    S101_M_총괄_CP_이상 AT %MW1009.7 : BOOL;
    S101_M_총괄_CT_이상 AT %MW1010.4 : BOOL;
    S101_M_총괄_EOCR_이상 AT %MW1009.8 : BOOL;
    S101_M_총괄_INV_이상 AT %MW1009.9 : BOOL;
    S101_M_총괄_LS_이상 AT %MW1009.15 : BOOL;
    S101_M_총괄_MATCH_이상 AT %MW1010.0 : BOOL;
    S101_M_총괄_MC_이상 AT %MW1009.13 : BOOL;
    S101_M_총괄_MOTOR_이상 AT %MW1010.3 : BOOL;
    S101_M_총괄_NFB_이상 AT %MW1009.11 : BOOL;
    S101_M_총괄_ROBOT_이상 AT %MW1010.1 : BOOL;
    S101_M_총괄_SAFETY_이상 AT %MW1009.2 : BOOL;
    S101_M_총괄_SRV_이상 AT %MW1009.10 : BOOL;
    S101_M_총괄_공기압_이상 AT %MW1009.3 : BOOL;
    S101_M_총괄_비상정지_이상 AT %MW1009.1 : BOOL;
    S101_M_총괄_사양_이상 AT %MW1009.6 : BOOL;
    S101_M_총괄_오버런_이상 AT %MW1009.12 : BOOL;
    S101_M_총괄_용점타점수_이상 AT %MW1010.2 : BOOL;
    S101_M_총괄_이상 AT %MW1009.0 : BOOL;
    S101_M_총괄_제품감지_이상 AT %MW1009.4 : BOOL;
    S101_M_총괄_차종_이상 AT %MW1009.5 : BOOL;
    S101_M_총괄_통신_이상 AT %MW1009.14 : BOOL;
    S101_M_핀클램프_전진_LAMP AT %MW11106 : WORD;
    S101_M_핀클램프_전진_LS_이상 AT %MW1106.5 : BOOL;
    S101_M_핀클램프_전진_보조 AT %MW1106.1 : BOOL;
    S101_M_핀클램프_전진단 AT %MW1106.3 : BOOL;
    S101_M_핀클램프_조건 AT %MW1106.0 : BOOL;
    S101_M_핀클램프_후진_LAMP AT %MW11107 : WORD;
    S101_M_핀클램프_후진_LS_이상 AT %MW1106.6 : BOOL;
    S101_M_핀클램프_후진_보조 AT %MW1106.2 : BOOL;
    S101_M_핀클램프_후진단 AT %MW1106.4 : BOOL;
    S101_OUT_3축_1_CONTROL AT %MB102000 : ARRAY[0..23] OF BYTE;
    S101_OUT_3축_1_EXPEN AT %MB102024 : ARRAY[0..31] OF BYTE;
    S101_OUT_3축_2_CONTROL AT %MB102200 : ARRAY[0..23] OF BYTE;
    S101_OUT_3축_2_EXPEN AT %MB102224 : ARRAY[0..31] OF BYTE;
    S101_OUT_3축_3_CONTROL AT %MB102400 : ARRAY[0..23] OF BYTE;
    S101_OUT_3축_3_EXPEN AT %MB102424 : ARRAY[0..31] OF BYTE;
    S101_PRS_AX_DASH_클램프_전진 AT %MW86100.13 : BOOL; (* 입력 접점 13 *)
    S101_PRS_AX_DASH_클램프_후진 AT %MW86100.12 : BOOL; (* 입력 접점 12 *)
    S101_PRS_AX_핀클램프_전진단1 AT %MW86101.0 : BOOL;
    S101_PRS_AX_핀클램프_전진단2 AT %MW86101.2 : BOOL;
    S101_PRS_AX_핀클램프_전진단3 AT %MW86101.4 : BOOL;
    S101_PRS_AX_핀클램프_전진단4 AT %MW86101.6 : BOOL;
    S101_PRS_AX_핀클램프_후진단1 AT %MW86101.1 : BOOL;
    S101_PRS_AX_핀클램프_후진단2 AT %MW86101.3 : BOOL;
    S101_PRS_AX_핀클램프_후진단3 AT %MW86101.5 : BOOL;
    S101_PRS_AX_핀클램프_후진단4 AT %MW86101.7 : BOOL;
    S101_PRS_I_3축_DASH_파트1_ON AT %MW86102.6 : BOOL; (* 입력 접점 06 *)
    S101_PRS_I_3축_DASH_파트2_ON AT %MW86102.7 : BOOL; (* 입력 접점 07 *)
    S101_PRS_I_3축_LH_파트_ON AT %MW86102.4 : BOOL; (* 입력 접점 04 *)
    S101_PRS_I_3축_RH_파트_ON AT %MW86102.5 : BOOL; (* 입력 접점 05 *)
    S101_PRS_I_AX_APRON_LHD_사양감지 AT %MW86102.8 : BOOL;
    S101_PRS_I_AX_APRON_RHD_사양감지 AT %MW86102.9 : BOOL;
    S101_PRS_I_AX_DASH_파트_ON AT %MW86102.2 : BOOL;
    S101_PRS_I_AX_LH_파트_ON AT %MW86102.0 : BOOL;
    S101_PRS_I_AX_RH_파트_ON AT %MW86102.1 : BOOL;
    S101_R102_2_CTYPE_MOVE : FB407_Car_Type_Move_Stn_v1;
    S101_R102_3_CTYPE_MOVE : FB407_Car_Type_Move_Stn_v1;
    S101_RH_M_APRON_PLT1_COUNT_RST AT %MW1250.15 : BOOL;
    S101_RH_M_APRON_PLT1_FAULT AT %MW1250.6 : BOOL;
    S101_RH_M_APRON_PLT1_MATCH_OK AT %MW1250.5 : BOOL;
    S101_RH_M_APRON_PLT1_PART_ERR AT %MW1250.9 : BOOL;
    S101_RH_M_APRON_PLT1_PLT_NONE AT %MW1250.2 : BOOL;
    S101_RH_M_APRON_PLT1_PLT_ON AT %MW1250.1 : BOOL;
    S101_RH_M_APRON_PLT1_PROG_OK AT %MW1250.0 : BOOL;
    S101_RH_M_APRON_PLT1_P파트무 AT %MW1250.4 : BOOL;
    S101_RH_M_APRON_PLT1_UNMAT_ERR AT %MW1250.7 : BOOL;
    S101_RH_M_APRON_PLT1_로딩완료 AT %MW1250.10 : BOOL;
    S101_RH_M_APRON_PLT1_제품수량 AT %MW1274 : WORD;
    S101_RH_M_APRON_PLT1_차종100 AT %MW1250.11 : BOOL;
    S101_RH_M_APRON_PLT1_차종200 AT %MW1250.12 : BOOL;
    S101_RH_M_APRON_PLT1_차종300 AT %MW1250.13 : BOOL;
    S101_RH_M_APRON_PLT1_차종400 AT %MW1250.14 : BOOL;
    S101_RH_M_APRON_PLT1_차종유 AT %MW1250.8 : BOOL;
    S101_RH_M_APRON_PLT1_차종코드 AT %MW1266 : WORD;
    S101_RH_M_APRON_PLT1_파트무 : BOOL;
    S101_RH_M_APRON_PLT1_파트유 AT %MW1250.3 : BOOL;
    S101_RH_M_APRON_PLT2_COUNT_RST AT %MW1251.15 : BOOL;
    S101_RH_M_APRON_PLT2_FAULT AT %MW1251.6 : BOOL;
    S101_RH_M_APRON_PLT2_MATCH_OK AT %MW1251.5 : BOOL;
    S101_RH_M_APRON_PLT2_PART_ERR AT %MW1251.9 : BOOL;
    S101_RH_M_APRON_PLT2_PLT_NONE AT %MW1251.2 : BOOL;
    S101_RH_M_APRON_PLT2_PLT_ON AT %MW1251.1 : BOOL;
    S101_RH_M_APRON_PLT2_PROG_OK AT %MW1251.0 : BOOL;
    S101_RH_M_APRON_PLT2_UNMAT_ERR AT %MW1251.7 : BOOL;
    S101_RH_M_APRON_PLT2_로딩완료 AT %MW1251.10 : BOOL;
    S101_RH_M_APRON_PLT2_제품수량 AT %MW1275 : WORD;
    S101_RH_M_APRON_PLT2_차종100 AT %MW1251.11 : BOOL;
    S101_RH_M_APRON_PLT2_차종200 AT %MW1251.12 : BOOL;
    S101_RH_M_APRON_PLT2_차종300 AT %MW1251.13 : BOOL;
    S101_RH_M_APRON_PLT2_차종400 AT %MW1251.14 : BOOL;
    S101_RH_M_APRON_PLT2_차종유 AT %MW1251.8 : BOOL;
    S101_RH_M_APRON_PLT2_차종코드 AT %MW1267 : WORD;
    S101_RH_M_APRON_PLT2_파트무 AT %MW1251.4 : BOOL;
    S101_RH_M_APRON_PLT2_파트유 AT %MW1251.3 : BOOL;
    S101_RH_M_APRON_PLT3_제품수량 AT %MW1276 : WORD;
    S101_RH_M_APRON_PLT3_차종코드 AT %MW1268 : WORD;
    S101_RH_M_APRON_PLT4_제품수량 AT %MW1277 : WORD;
    S101_RH_M_APRON_PLT4_차종코드 AT %MW1269 : WORD;
    S101_RH_M_APRON_PLT5_제품수량 AT %MW1278 : WORD;
    S101_RH_M_APRON_PLT5_차종코드 AT %MW1270 : WORD;
    S101_RH_M_APRON_PLT6_제품수량 AT %MW1279 : WORD;
    S101_RH_M_APRON_PLT6_차종코드 AT %MW1271 : WORD;
    S101_RH_M_APRON_PLT7_제품수량 AT %MW1280 : WORD;
    S101_RH_M_APRON_PLT7_차종코드 AT %MW1272 : WORD;
    S101_RH_M_APRON_PLT8_제품수량 AT %MW1281 : WORD;
    S101_RH_M_APRON_PLT8_차종코드 AT %MW1273 : WORD;
    S101_RH_M_APRON_PLT_PRIORITY1 AT %MW1258 : WORD;
    S101_RH_M_APRON_PLT_PRIORITY2 AT %MW1259 : WORD;
    S101_RH_M_APRON_PLT_PRIORITY3 AT %MW1260 : WORD;
    S101_RH_M_APRON_PLT_PRIORITY4 AT %MW1261 : WORD;
    S101_RH_M_APRON_PLT_PRIORITY5 AT %MW1262 : WORD;
    S101_RH_M_APRON_PLT_PRIORITY6 AT %MW1263 : WORD;
    S101_RH_M_APRON_PLT_PRIORITY7 AT %MW1264 : WORD;
    S101_RH_M_APRON_PLT_PRIORITY8 AT %MW1265 : WORD;
    S101_RS_AX_SFT_전진1 AT %MW86100.8 : BOOL; (* 입력 접점 08 *)
    S101_RS_AX_SFT_전진2 AT %MW86100.10 : BOOL; (* 입력 접점 10 *)
    S101_RS_AX_SFT_후진1 AT %MW86100.9 : BOOL; (* 입력 접점 09 *)
    S101_RS_AX_SFT_후진2 AT %MW86100.11 : BOOL; (* 입력 접점 11 *)
    S101_RS_AX_래치_전진1 AT %MW86100.0 : BOOL; (* 입력 접점 00 *)
    S101_RS_AX_래치_전진2 AT %MW86100.2 : BOOL; (* 입력 접점 02 *)
    S101_RS_AX_래치_후진1 AT %MW86100.1 : BOOL; (* 입력 접점 01 *)
    S101_RS_AX_래치_후진2 AT %MW86100.3 : BOOL; (* 입력 접점 03 *)
    S101_SHIFT : ACT_6_CYL;
    S101_SOL_AX_DASH_클램프_전진 AT %MW96103.4 : BOOL; (* 출력 접점 04 *)
    S101_SOL_AX_DASH_클램프_후진 AT %MW96103.5 : BOOL; (* 출력 접점 05 *)
    S101_SOL_AX_SHIFT_전진 AT %MW96103.2 : BOOL; (* 출력 접점 02 *)
    S101_SOL_AX_SHIFT_후진 AT %MW96103.3 : BOOL; (* 출력 접점 03 *)
    S101_SOL_AX_래치_전진 AT %MW96103.0 : BOOL; (* 출력 접점 00 *)
    S101_SOL_AX_래치_후진 AT %MW96103.1 : BOOL; (* 출력 접점 01 *)
    S101_SOL_AX_핀클램프_전진출력 AT %MW96103.6 : BOOL;
    S101_SOL_AX_핀클램프_후진출력 AT %MW96103.7 : BOOL;
    S101_공기압_AIR_CHECK AT %MW86102.14 : BOOL; (* 입력 접점 14 *)
    S101_운전준비 : TON;
    S101_전진_ON AT %MW1048.1 : BOOL;
    S101_후진_ON AT %MW1048.2 : BOOL;
    S102_6_20_PLC_BOX_CP_TRIP AT %MW86202.15 : BOOL; (* 입력 접점 15 *)
    S102_DASH_클램프 : ACT_6_CYL;
    S102_HOME AT %MW1548.0 : BOOL;
    S102_M_ACT_선택_1 AT %MW1540.0 : BOOL;
    S102_M_ACT_선택_10 AT %MW1540.9 : BOOL;
    S102_M_ACT_선택_11 AT %MW1540.10 : BOOL;
    S102_M_ACT_선택_12 AT %MW1540.11 : BOOL;
    S102_M_ACT_선택_13 AT %MW1540.12 : BOOL;
    S102_M_ACT_선택_14 AT %MW1540.13 : BOOL;
    S102_M_ACT_선택_15 AT %MW1540.14 : BOOL;
    S102_M_ACT_선택_16 AT %MW1540.15 : BOOL;
    S102_M_ACT_선택_17 AT %MW1541.0 : BOOL;
    S102_M_ACT_선택_18 AT %MW1541.1 : BOOL;
    S102_M_ACT_선택_19 AT %MW1541.2 : BOOL;
    S102_M_ACT_선택_2 AT %MW1540.1 : BOOL;
    S102_M_ACT_선택_20 AT %MW1541.3 : BOOL;
    S102_M_ACT_선택_21 AT %MW1541.4 : BOOL;
    S102_M_ACT_선택_22 AT %MW1541.5 : BOOL;
    S102_M_ACT_선택_23 AT %MW1541.6 : BOOL;
    S102_M_ACT_선택_24 AT %MW1541.7 : BOOL;
    S102_M_ACT_선택_25 AT %MW1541.8 : BOOL;
    S102_M_ACT_선택_26 AT %MW1541.9 : BOOL;
    S102_M_ACT_선택_27 AT %MW1541.10 : BOOL;
    S102_M_ACT_선택_28 AT %MW1541.11 : BOOL;
    S102_M_ACT_선택_29 AT %MW1541.12 : BOOL;
    S102_M_ACT_선택_3 AT %MW1540.2 : BOOL;
    S102_M_ACT_선택_30 AT %MW1541.13 : BOOL;
    S102_M_ACT_선택_31 AT %MW1541.14 : BOOL;
    S102_M_ACT_선택_32 AT %MW1541.15 : BOOL;
    S102_M_ACT_선택_4 AT %MW1540.3 : BOOL;
    S102_M_ACT_선택_5 AT %MW1540.4 : BOOL;
    S102_M_ACT_선택_6 AT %MW1540.5 : BOOL;
    S102_M_ACT_선택_7 AT %MW1540.6 : BOOL;
    S102_M_ACT_선택_8 AT %MW1540.7 : BOOL;
    S102_M_ACT_선택_9 AT %MW1540.8 : BOOL;
    S102_M_CTIME_OVER_ALRAM AT %MW1506.14 : BOOL;
    S102_M_CTIME_OVER_MUTE AT %MW1506.13 : BOOL;
    S102_M_DASH_PLT1_COUNT_RST AT %MW1700.15 : BOOL;
    S102_M_DASH_PLT1_FAULT AT %MW1700.6 : BOOL;
    S102_M_DASH_PLT1_MATCH_OK AT %MW1700.5 : BOOL;
    S102_M_DASH_PLT1_PART_ERR AT %MW1700.9 : BOOL;
    S102_M_DASH_PLT1_PLT_NONE AT %MW1700.2 : BOOL;
    S102_M_DASH_PLT1_PLT_ON AT %MW1700.1 : BOOL;
    S102_M_DASH_PLT1_PROG_OK AT %MW1700.0 : BOOL;
    S102_M_DASH_PLT1_UNMAT_ERR AT %MW1700.7 : BOOL;
    S102_M_DASH_PLT1_로딩완료 AT %MW1700.10 : BOOL;
    S102_M_DASH_PLT1_제품수량 AT %MW1724 : WORD;
    S102_M_DASH_PLT1_차종100 AT %MW1700.11 : BOOL;
    S102_M_DASH_PLT1_차종200 AT %MW1700.12 : BOOL;
    S102_M_DASH_PLT1_차종300 AT %MW1700.13 : BOOL;
    S102_M_DASH_PLT1_차종400 AT %MW1700.14 : BOOL;
    S102_M_DASH_PLT1_차종유 AT %MW1700.8 : BOOL;
    S102_M_DASH_PLT1_차종코드 AT %MW1716 : WORD;
    S102_M_DASH_PLT1_파트무 AT %MW1700.4 : BOOL;
    S102_M_DASH_PLT1_파트유 AT %MW1700.3 : BOOL;
    S102_M_DASH_PLT2_COUNT_RST AT %MW1701.15 : BOOL;
    S102_M_DASH_PLT2_FAULT AT %MW1701.6 : BOOL;
    S102_M_DASH_PLT2_MATCH_OK AT %MW1701.5 : BOOL;
    S102_M_DASH_PLT2_PART_ERR AT %MW1701.9 : BOOL;
    S102_M_DASH_PLT2_PLT_NONE AT %MW1701.2 : BOOL;
    S102_M_DASH_PLT2_PLT_ON AT %MW1701.1 : BOOL;
    S102_M_DASH_PLT2_PROG_OK AT %MW1701.0 : BOOL;
    S102_M_DASH_PLT2_UNMAT_ERR AT %MW1701.7 : BOOL;
    S102_M_DASH_PLT2_로딩완료 AT %MW1701.10 : BOOL;
    S102_M_DASH_PLT2_제품수량 AT %MW1725 : WORD;
    S102_M_DASH_PLT2_차종100 AT %MW1701.11 : BOOL;
    S102_M_DASH_PLT2_차종200 AT %MW1701.12 : BOOL;
    S102_M_DASH_PLT2_차종300 AT %MW1701.13 : BOOL;
    S102_M_DASH_PLT2_차종400 AT %MW1701.14 : BOOL;
    S102_M_DASH_PLT2_차종유 AT %MW1701.8 : BOOL;
    S102_M_DASH_PLT2_차종코드 AT %MW1717 : WORD;
    S102_M_DASH_PLT2_파트무 AT %MW1701.4 : BOOL;
    S102_M_DASH_PLT2_파트유 AT %MW1701.3 : BOOL;
    S102_M_DASH_PLT3_COUNT_RST AT %MW1702.15 : BOOL;
    S102_M_DASH_PLT3_FAULT AT %MW1702.6 : BOOL;
    S102_M_DASH_PLT3_MATCH_OK AT %MW1702.5 : BOOL;
    S102_M_DASH_PLT3_PART_ERR AT %MW1702.9 : BOOL;
    S102_M_DASH_PLT3_PLT_NONE AT %MW1702.2 : BOOL;
    S102_M_DASH_PLT3_PLT_ON AT %MW1702.1 : BOOL;
    S102_M_DASH_PLT3_PROG_OK AT %MW1702.0 : BOOL;
    S102_M_DASH_PLT3_UNMAT_ERR AT %MW1702.7 : BOOL;
    S102_M_DASH_PLT3_로딩완료 AT %MW1702.10 : BOOL;
    S102_M_DASH_PLT3_제품수량 AT %MW1726 : WORD;
    S102_M_DASH_PLT3_차종100 AT %MW1702.11 : BOOL;
    S102_M_DASH_PLT3_차종200 AT %MW1702.12 : BOOL;
    S102_M_DASH_PLT3_차종300 AT %MW1702.13 : BOOL;
    S102_M_DASH_PLT3_차종400 AT %MW1702.14 : BOOL;
    S102_M_DASH_PLT3_차종유 AT %MW1702.8 : BOOL;
    S102_M_DASH_PLT3_차종코드 AT %MW1718 : WORD;
    S102_M_DASH_PLT3_파트무 AT %MW1702.4 : BOOL;
    S102_M_DASH_PLT3_파트유 AT %MW1702.3 : BOOL;
    S102_M_DASH_PLT4_COUNT_RST AT %MW1703.15 : BOOL;
    S102_M_DASH_PLT4_FAULT AT %MW1703.6 : BOOL;
    S102_M_DASH_PLT4_MATCH_OK AT %MW1703.5 : BOOL;
    S102_M_DASH_PLT4_PART_ERR AT %MW1703.9 : BOOL;
    S102_M_DASH_PLT4_PLT_NONE AT %MW1703.2 : BOOL;
    S102_M_DASH_PLT4_PLT_ON AT %MW1703.1 : BOOL;
    S102_M_DASH_PLT4_PROG_OK AT %MW1703.0 : BOOL;
    S102_M_DASH_PLT4_UNMAT_ERR AT %MW1703.7 : BOOL;
    S102_M_DASH_PLT4_로딩완료 AT %MW1703.10 : BOOL;
    S102_M_DASH_PLT4_제품수량 AT %MW1727 : WORD;
    S102_M_DASH_PLT4_차종100 AT %MW1703.11 : BOOL;
    S102_M_DASH_PLT4_차종200 AT %MW1703.12 : BOOL;
    S102_M_DASH_PLT4_차종300 AT %MW1703.13 : BOOL;
    S102_M_DASH_PLT4_차종400 AT %MW1703.14 : BOOL;
    S102_M_DASH_PLT4_차종유 AT %MW1703.8 : BOOL;
    S102_M_DASH_PLT4_차종코드 AT %MW1719 : WORD;
    S102_M_DASH_PLT4_파트무 AT %MW1703.4 : BOOL;
    S102_M_DASH_PLT4_파트유 AT %MW1703.3 : BOOL;
    S102_M_DASH_PLT5_제품수량 AT %MW1728 : WORD;
    S102_M_DASH_PLT5_차종코드 AT %MW1720 : WORD;
    S102_M_DASH_PLT6_제품수량 AT %MW1729 : WORD;
    S102_M_DASH_PLT6_차종코드 AT %MW1721 : WORD;
    S102_M_DASH_PLT7_제품수량 AT %MW1730 : WORD;
    S102_M_DASH_PLT7_차종코드 AT %MW1722 : WORD;
    S102_M_DASH_PLT8_제품수량 AT %MW1731 : WORD;
    S102_M_DASH_PLT8_차종코드 AT %MW1723 : WORD;
    S102_M_DASH_PLT_PRIORITY1 AT %MW1708 : WORD;
    S102_M_DASH_PLT_PRIORITY2 AT %MW1709 : WORD;
    S102_M_DASH_PLT_PRIORITY3 AT %MW1710 : WORD;
    S102_M_DASH_PLT_PRIORITY4 AT %MW1711 : WORD;
    S102_M_DASH_PLT_PRIORITY5 AT %MW1712 : WORD;
    S102_M_DASH_PLT_PRIORITY6 AT %MW1713 : WORD;
    S102_M_DASH_PLT_PRIORITY7 AT %MW1714 : WORD;
    S102_M_DASH_PLT_PRIORITY8 AT %MW1715 : WORD;
    S102_M_DASH_랙방1_2_통신이상 AT %MW1524.1 : BOOL;
    S102_M_DASH_랙방3_4_통신이상 AT %MW1524.2 : BOOL;
    S102_M_DATA_삭제_PLS AT %MW9003.0 : BOOL; (* S102_M_DATA_삭제_PLS *)
    S102_M_DATA_삭제_SIGN AT %MW9003.1 : BOOL; (* S102_M_DATA_삭제_SIGN *)
    S102_M_DATA_삭제_완료 AT %MW9003.2 : BOOL; (* S102_M_DATA_삭제_완료 *)
    S102_M_DATA_전송_MEMO AT %MW9003.8 : BOOL; (* S102_M_DATA_전송_MEMO *)
    S102_M_DATA_전송_PLS AT %MW9003.9 : BOOL; (* S102_M_DATA_전송_PLS *)
    S102_M_DATA_전송_SIGN AT %MW9003.10 : BOOL; (* S102_M_DATA_전송_SIGN *)
    S102_M_DATA_전송_완료 AT %MW9003.11 : BOOL; (* S102_M_DATA_전송_완료 *)
    S102_M_GATE_DOOR_NORMAL AT %MW1506.4 : BOOL;
    S102_M_GATE_ESTOP_NORMAR AT %MW1506.3 : BOOL;
    S102_M_OP_ESTOP_NORMAL AT %MW1506.1 : BOOL;
    S102_M_R102_1_CN_MATCH_OK AT %MW1505.0 : BOOL;
    S102_M_R102_1_CT_MATCH_OK AT %MW1505.1 : BOOL;
    S102_M_RB_ESTOP_NORMAL AT %MW1506.2 : BOOL;
    S102_M_SAFTY_NO_INT AT %MW1504.4 : BOOL;
    S102_M_SEMI_자동_모드 AT %MW1500.2 : BOOL;
    S102_M_SEQ AT %MW10060 : WORD; (* S102_M_SEQ *)
    S102_M_STN_DASH_로딩완료 AT %MW1501.8 : BOOL;
    S102_M_STN_차종_NONE AT %MW1502.1 : BOOL;
    S102_M_STN_차종_ON AT %MW1502.0 : BOOL;
    S102_M_VIN_NO_1_2 AT %MW10071 : WORD; (* S102_M_VIN_NO_1_2 *)
    S102_M_VIN_NO_3_4 AT %MW10072 : WORD; (* S102_M_VIN_NO_3_4 *)
    S102_M_VIN_NO_5_6 AT %MW10073 : WORD; (* S102_M_VIN_NO_5_6 *)
    S102_M_VIN_NO_7_8 AT %MW10074 : WORD; (* S102_M_VIN_NO_7_8 *)
    S102_M_VIN_NO_9_10 AT %MW10075 : WORD; (* S102_M_VIN_NO_9_10 *)
    S102_M_공정_HOME_POSI AT %MW1504.0 : BOOL;
    S102_M_공정_SAFETY_NORMAL AT %MW1506.7 : BOOL;
    S102_M_공정_간섭무 AT %MW1504.1 : BOOL;
    S102_M_공정_사양감지_OK AT %MW1501.5 : BOOL;
    S102_M_공정_제품감지_OFF AT %MW1501.4 : BOOL;
    S102_M_공정_제품감지_ON AT %MW1501.3 : BOOL;
    S102_M_공정_통신이상 AT %MW1524.0 : BOOL;
    S102_M_부저_정지_보조 AT %MW1500.11 : BOOL;
    S102_M_사양_이상 AT %MW1516.0 : BOOL;
    S102_M_수동_모드 AT %MW1500.3 : BOOL;
    S102_M_운전준비_ON AT %MW1500.0 : BOOL;
    S102_M_이상_리셋_보조 AT %MW1500.10 : BOOL;
    S102_M_자동_START AT %MW1500.5 : BOOL;
    S102_M_자동_모드 AT %MW1500.1 : BOOL;
    S102_M_자동_운전중 AT %MW1500.4 : BOOL;
    S102_M_작업_완료 AT %MW1501.0 : BOOL;
    S102_M_작업_완료_보조 AT %MW1500.9 : BOOL;
    S102_M_제품감지_이상 AT %MW1514.0 : BOOL;
    S102_M_차종1_AX AT %MW10061.0 : BOOL; (* S102_M_차종1_AX *)
    S102_M_차종1_B AT %MW10061.1 : BOOL; (* S102_M_차종1_B *)
    S102_M_차종1_C AT %MW10061.2 : BOOL; (* S102_M_차종1_C *)
    S102_M_차종1_D AT %MW10061.3 : BOOL; (* S102_M_차종1_D *)
    S102_M_차종1_E AT %MW10061.4 : BOOL; (* S102_M_차종1_E *)
    S102_M_차종1_F AT %MW10061.5 : BOOL; (* S102_M_차종1_F *)
    S102_M_차종1_G AT %MW10061.6 : BOOL; (* S102_M_차종1_G *)
    S102_M_차종1_H AT %MW10061.7 : BOOL; (* S102_M_차종1_H *)
    S102_M_차종2_3DR AT %MW10061.8 : BOOL; (* S102_M_차종2_3DR *)
    S102_M_차종2_4DR AT %MW10061.9 : BOOL; (* S102_M_차종2_4DR *)
    S102_M_차종2_5DR AT %MW10061.10 : BOOL; (* S102_M_차종2_5DR *)
    S102_M_차종2_SP1 AT %MW10061.12 : BOOL; (* S102_M_차종2_SP1 *)
    S102_M_차종2_SP2 AT %MW10061.13 : BOOL; (* S102_M_차종2_SP2 *)
    S102_M_차종2_WGN AT %MW10061.11 : BOOL; (* S102_M_차종2_WGN *)
    S102_M_차종3_LHD AT %MW10061.14 : BOOL; (* S102_M_차종3_LHD *)
    S102_M_차종3_RHD AT %MW10061.15 : BOOL; (* S102_M_차종3_RHD *)
    S102_M_차종4_EEC AT %MW10062.3 : BOOL; (* S102_M_차종4_EEC *)
    S102_M_차종4_SP1 AT %MW10062.8 : BOOL; (* S102_M_차종4_SP1 *)
    S102_M_차종4_SP2 AT %MW10062.9 : BOOL; (* S102_M_차종4_SP2 *)
    S102_M_차종4_SP3 AT %MW10062.11 : BOOL; (* S102_M_차종4_SP3 *)
    S102_M_차종4_SP4 AT %MW10062.12 : BOOL; (* S102_M_차종4_SP4 *)
    S102_M_차종4_SP5 AT %MW10062.13 : BOOL; (* S102_M_차종4_SP5 *)
    S102_M_차종4_SP6 AT %MW10062.14 : BOOL; (* S102_M_차종4_SP6 *)
    S102_M_차종4_SP7 AT %MW10062.15 : BOOL; (* S102_M_차종4_SP7 *)
    S102_M_차종4_내수 AT %MW10062.0 : BOOL; (* S102_M_차종4_내수 *)
    S102_M_차종4_러시아 AT %MW10062.10 : BOOL; (* S102_M_차종4_러시아 *)
    S102_M_차종4_북미 AT %MW10062.2 : BOOL; (* S102_M_차종4_북미 *)
    S102_M_차종4_브라질 AT %MW10062.7 : BOOL; (* S102_M_차종4_브라질 *)
    S102_M_차종4_수출 AT %MW10062.1 : BOOL; (* S102_M_차종4_수출 *)
    S102_M_차종4_중국 AT %MW10062.6 : BOOL; (* S102_M_차종4_중국 *)
    S102_M_차종4_중동 AT %MW10062.5 : BOOL; (* S102_M_차종4_중동 *)
    S102_M_차종4_호주 AT %MW10062.4 : BOOL; (* S102_M_차종4_호주 *)
    S102_M_차종5_AT AT %MW10063.1 : BOOL; (* S102_M_차종5_AT *)
    S102_M_차종5_MT AT %MW10063.0 : BOOL; (* S102_M_차종5_MT *)
    S102_M_차종5_SP1 AT %MW10063.2 : BOOL; (* S102_M_차종5_SP1 *)
    S102_M_차종6_DSROOF AT %MW10063.6 : BOOL; (* S102_M_차종6_DSROOF *)
    S102_M_차종6_SP1 AT %MW10063.7 : BOOL; (* S102_M_차종6_SP1 *)
    S102_M_차종6_썬루프 AT %MW10063.4 : BOOL; (* S102_M_차종6_썬루프 *)
    S102_M_차종6_일반루프 AT %MW10063.3 : BOOL; (* S102_M_차종6_일반루프 *)
    S102_M_차종6_파노라마루프 AT %MW10063.5 : BOOL; (* S102_M_차종6_파노라마루프 *)
    S102_M_차종7_DSL AT %MW10063.9 : BOOL; (* S102_M_차종7_DSL *)
    S102_M_차종7_GSL AT %MW10063.8 : BOOL; (* S102_M_차종7_GSL *)
    S102_M_차종7_SP1 AT %MW10063.10 : BOOL; (* S102_M_차종7_SP1 *)
    S102_M_차종7_SP2 AT %MW10063.11 : BOOL; (* S102_M_차종7_SP2 *)
    S102_M_차종7_SP3 AT %MW10063.12 : BOOL; (* S102_M_차종7_SP3 *)
    S102_M_차종7_SP4 AT %MW10063.13 : BOOL; (* S102_M_차종7_SP4 *)
    S102_M_차종7_SP5 AT %MW10063.14 : BOOL; (* S102_M_차종7_SP5 *)
    S102_M_차종7_SP6 AT %MW10063.15 : BOOL; (* S102_M_차종7_SP6 *)
    S102_M_차종8_2WD AT %MW10064.0 : BOOL; (* S102_M_차종8_2WD *)
    S102_M_차종8_4WD AT %MW10064.1 : BOOL; (* S102_M_차종8_4WD *)
    S102_M_차종8_SP1 AT %MW10064.2 : BOOL; (* S102_M_차종8_SP1 *)
    S102_M_차종9_MPI AT %MW10064.3 : BOOL; (* S102_M_차종9_MPI *)
    S102_M_차종9_SP1 AT %MW10064.5 : BOOL; (* S102_M_차종9_SP1 *)
    S102_M_차종9_SP10 AT %MW10064.14 : BOOL; (* S102_M_차종9_SP10 *)
    S102_M_차종9_SP11 AT %MW10064.15 : BOOL; (* S102_M_차종9_SP11 *)
    S102_M_차종9_SP2 AT %MW10064.6 : BOOL; (* S102_M_차종9_SP2 *)
    S102_M_차종9_SP3 AT %MW10064.7 : BOOL; (* S102_M_차종9_SP3 *)
    S102_M_차종9_SP4 AT %MW10064.8 : BOOL; (* S102_M_차종9_SP4 *)
    S102_M_차종9_SP5 AT %MW10064.9 : BOOL; (* S102_M_차종9_SP5 *)
    S102_M_차종9_SP6 AT %MW10064.10 : BOOL; (* S102_M_차종9_SP6 *)
    S102_M_차종9_SP7 AT %MW10064.11 : BOOL; (* S102_M_차종9_SP7 *)
    S102_M_차종9_SP8 AT %MW10064.12 : BOOL; (* S102_M_차종9_SP8 *)
    S102_M_차종9_SP9 AT %MW10064.13 : BOOL; (* S102_M_차종9_SP9 *)
    S102_M_차종9_T_GDI AT %MW10064.4 : BOOL; (* S102_M_차종9_T_GDI *)
    S102_M_차종_AS AT %MW10070.9 : BOOL; (* S102_M_차종_AS *)
    S102_M_차종_OPT1_R_RACK_무 AT %MW10065.3 : BOOL; (* S102_M_차종_OPT1_R_RACK_무 *)
    S102_M_차종_OPT1_R_RACK_유 AT %MW10065.2 : BOOL; (* S102_M_차종_OPT1_R_RACK_유 *)
    S102_M_차종_OPT1_SP1 AT %MW10065.10 : BOOL; (* S102_M_차종_OPT1_SP1 *)
    S102_M_차종_OPT1_SP2 AT %MW10065.11 : BOOL; (* S102_M_차종_OPT1_SP2 *)
    S102_M_차종_OPT1_SP3 AT %MW10065.12 : BOOL; (* S102_M_차종_OPT1_SP3 *)
    S102_M_차종_OPT1_SP4 AT %MW10065.13 : BOOL; (* S102_M_차종_OPT1_SP4 *)
    S102_M_차종_OPT1_SP5 AT %MW10065.14 : BOOL; (* S102_M_차종_OPT1_SP5 *)
    S102_M_차종_OPT1_SP6 AT %MW10065.15 : BOOL; (* S102_M_차종_OPT1_SP6 *)
    S102_M_차종_OPT1_S_REP_EATER_무 AT %MW10065.7 : BOOL; (* S102_M_차종_OPT1_S_REP_EATER_무 *)
    S102_M_차종_OPT1_S_REP_EATER_유 AT %MW10065.6 : BOOL; (* S102_M_차종_OPT1_S_REP_EATER_유 *)
    S102_M_차종_OPT1_VAN_무 AT %MW10065.9 : BOOL; (* S102_M_차종_OPT1_VAN_무 *)
    S102_M_차종_OPT1_VAN_유 AT %MW10065.8 : BOOL; (* S102_M_차종_OPT1_VAN_유 *)
    S102_M_차종_OPT1_슬라이딩_무 AT %MW10065.1 : BOOL; (* S102_M_차종_OPT1_슬라이딩_무 *)
    S102_M_차종_OPT1_슬라이딩_유 AT %MW10065.0 : BOOL; (* S102_M_차종_OPT1_슬라이딩_유 *)
    S102_M_차종_OPT1_폴딩_무 AT %MW10065.5 : BOOL; (* S102_M_차종_OPT1_폴딩_무 *)
    S102_M_차종_OPT1_폴딩_유 AT %MW10065.4 : BOOL; (* S102_M_차종_OPT1_폴딩_유 *)
    S102_M_차종_OPT2_SP_WORD1 AT %MW10066 : WORD; (* S102_M_차종_OPT2_SP_WORD1 *)
    S102_M_차종_OPT3_SP_WORD2 AT %MW10067 : WORD; (* S102_M_차종_OPT3_SP_WORD2 *)
    S102_M_차종_OPT4_SP_WORD3 AT %MW10068 : WORD; (* S102_M_차종_OPT4_SP_WORD3 *)
    S102_M_차종_OPT5_SP_WORD4 AT %MW10069 : WORD; (* S102_M_차종_OPT5_SP_WORD4 *)
    S102_M_차종_SP1 AT %MW10070.0 : BOOL; (* S102_M_차종_SP1 *)
    S102_M_차종_SP2 AT %MW10070.1 : BOOL; (* S102_M_차종_SP2 *)
    S102_M_차종_SP3 AT %MW10070.2 : BOOL; (* S102_M_차종_SP3 *)
    S102_M_차종_SP4 AT %MW10070.3 : BOOL; (* S102_M_차종_SP4 *)
    S102_M_차종_SP5 AT %MW10070.4 : BOOL; (* S102_M_차종_SP5 *)
    S102_M_차종_SP6 AT %MW10070.5 : BOOL; (* S102_M_차종_SP6 *)
    S102_M_차종_SP7 AT %MW10070.6 : BOOL; (* S102_M_차종_SP7 *)
    S102_M_차종_SP8 AT %MW10070.7 : BOOL; (* S102_M_차종_SP8 *)
    S102_M_차종_SP9 AT %MW10070.15 : BOOL; (* S102_M_차종_SP9 *)
    S102_M_차종_공대차 AT %MW10070.12 : BOOL; (* S102_M_차종_공대차 *)
    S102_M_차종_공차 AT %MW10070.10 : BOOL; (* S102_M_차종_공차 *)
    S102_M_차종_불량대차 AT %MW10070.13 : BOOL; (* S102_M_차종_불량대차 *)
    S102_M_차종_불량차 AT %MW10070.11 : BOOL; (* S102_M_차종_불량차 *)
    S102_M_차종_비축 AT %MW10070.8 : BOOL; (* S102_M_차종_비축 *)
    S102_M_차종_취출대차 AT %MW10070.14 : BOOL; (* S102_M_차종_취출대차 *)
    S102_M_총괄_CP_이상 AT %MW1509.7 : BOOL;
    S102_M_총괄_CT_이상 AT %MW1510.4 : BOOL;
    S102_M_총괄_EOCR_이상 AT %MW1509.8 : BOOL;
    S102_M_총괄_INV_이상 AT %MW1509.9 : BOOL;
    S102_M_총괄_LS_이상 AT %MW1509.15 : BOOL;
    S102_M_총괄_MATCH_이상 AT %MW1510.0 : BOOL;
    S102_M_총괄_MC_이상 AT %MW1509.13 : BOOL;
    S102_M_총괄_MOTOR_이상 AT %MW1510.3 : BOOL;
    S102_M_총괄_NFB_이상 AT %MW1509.11 : BOOL;
    S102_M_총괄_ROBOT_이상 AT %MW1510.1 : BOOL;
    S102_M_총괄_SAFETY_이상 AT %MW1509.2 : BOOL;
    S102_M_총괄_SRV_이상 AT %MW1509.10 : BOOL;
    S102_M_총괄_공기압_이상 AT %MW1509.3 : BOOL;
    S102_M_총괄_비상정지_이상 AT %MW1509.1 : BOOL;
    S102_M_총괄_사양_이상 AT %MW1509.6 : BOOL;
    S102_M_총괄_오버런_이상 AT %MW1509.12 : BOOL;
    S102_M_총괄_용점타점수_이상 AT %MW1510.2 : BOOL;
    S102_M_총괄_이상 AT %MW1509.0 : BOOL;
    S102_M_총괄_제품감지_이상 AT %MW1509.4 : BOOL;
    S102_M_총괄_차종_이상 AT %MW1509.5 : BOOL;
    S102_M_총괄_통신_이상 AT %MW1509.14 : BOOL;
    S102_PRS_I_AT_감지 AT %MW86201.8 : BOOL;
    S102_PRS_I_AX_파트_ON AT %MW86200.1 : BOOL;
    S102_PRS_I_LHD_감지 AT %MW86201.0 : BOOL;
    S102_PRS_I_MT_감지 AT %MW86201.9 : BOOL;
    S102_PRS_I_RHD_감지 AT %MW86201.1 : BOOL;
    S102_PRS_I_공용_파트_ON AT %MW86200.0 : BOOL;
    S102_R102_1_CTYPE_MOVE : FB407_Car_Type_Move_Stn_v1;
    S102_R102_2_CTYPE_MOVE : FB407_Car_Type_Move_Stn_v1;
    S102_SHIFT : ACT_6_CYL;
    S102_운전준비 : TON;
    S102_전진_ON AT %MW1548.1 : BOOL;
    S102_후진_ON AT %MW1548.2 : BOOL;
    S103_6_30_PLC_BOX_CP_TRIP AT %MW86302.15 : BOOL; (* 입력 접점 15 *)
    S103_AX_래치 : ACT_6_CYL;
    S103_DASH_클램프 : ACT_6_CYL;
    S103_HOME AT %MW2048.0 : BOOL;
    S103_M_ACT_선택_1 AT %MW2040.0 : BOOL;
    S103_M_ACT_선택_10 AT %MW2040.9 : BOOL;
    S103_M_ACT_선택_11 AT %MW2040.10 : BOOL;
    S103_M_ACT_선택_12 AT %MW2040.11 : BOOL;
    S103_M_ACT_선택_13 AT %MW2040.12 : BOOL;
    S103_M_ACT_선택_14 AT %MW2040.13 : BOOL;
    S103_M_ACT_선택_15 AT %MW2040.14 : BOOL;
    S103_M_ACT_선택_16 AT %MW2040.15 : BOOL;
    S103_M_ACT_선택_17 AT %MW2041.0 : BOOL;
    S103_M_ACT_선택_18 AT %MW2041.1 : BOOL;
    S103_M_ACT_선택_19 AT %MW2041.2 : BOOL;
    S103_M_ACT_선택_2 AT %MW2040.1 : BOOL;
    S103_M_ACT_선택_20 AT %MW2041.3 : BOOL;
    S103_M_ACT_선택_21 AT %MW2041.4 : BOOL;
    S103_M_ACT_선택_22 AT %MW2041.5 : BOOL;
    S103_M_ACT_선택_23 AT %MW2041.6 : BOOL;
    S103_M_ACT_선택_24 AT %MW2041.7 : BOOL;
    S103_M_ACT_선택_25 AT %MW2041.8 : BOOL;
    S103_M_ACT_선택_26 AT %MW2041.9 : BOOL;
    S103_M_ACT_선택_27 AT %MW2041.10 : BOOL;
    S103_M_ACT_선택_28 AT %MW2041.11 : BOOL;
    S103_M_ACT_선택_29 AT %MW2041.12 : BOOL;
    S103_M_ACT_선택_3 AT %MW2040.2 : BOOL;
    S103_M_ACT_선택_30 AT %MW2041.13 : BOOL;
    S103_M_ACT_선택_31 AT %MW2041.14 : BOOL;
    S103_M_ACT_선택_32 AT %MW2041.15 : BOOL;
    S103_M_ACT_선택_4 AT %MW2040.3 : BOOL;
    S103_M_ACT_선택_5 AT %MW2040.4 : BOOL;
    S103_M_ACT_선택_6 AT %MW2040.5 : BOOL;
    S103_M_ACT_선택_7 AT %MW2040.6 : BOOL;
    S103_M_ACT_선택_8 AT %MW2040.7 : BOOL;
    S103_M_ACT_선택_9 AT %MW2040.8 : BOOL;
    S103_M_AX_래치_전진_LAMP AT %MW12100 : WORD;
    S103_M_AX_래치_전진_LS_이상 AT %MW2100.5 : BOOL;
    S103_M_AX_래치_전진_보조 AT %MW2100.1 : BOOL;
    S103_M_AX_래치_전진단 AT %MW2100.3 : BOOL;
    S103_M_AX_래치_조건 AT %MW2100.0 : BOOL;
    S103_M_AX_래치_후진_LAMP AT %MW12101 : WORD;
    S103_M_AX_래치_후진_LS_이상 AT %MW2100.6 : BOOL;
    S103_M_AX_래치_후진_보조 AT %MW2100.2 : BOOL;
    S103_M_AX_래치_후진단 AT %MW2100.4 : BOOL;
    S103_M_CTIME_OVER_ALRAM AT %MW2006.14 : BOOL;
    S103_M_CTIME_OVER_MUTE AT %MW2006.13 : BOOL;
    S103_M_DATA_삭제_PLS AT %MW9005.0 : BOOL; (* S103_M_DATA_삭제_PLS *)
    S103_M_DATA_삭제_SIGN AT %MW9005.1 : BOOL; (* S103_M_DATA_삭제_SIGN *)
    S103_M_DATA_삭제_완료 AT %MW9005.2 : BOOL; (* S103_M_DATA_삭제_완료 *)
    S103_M_DATA_전송_MEMO AT %MW9005.8 : BOOL; (* S103_M_DATA_전송_MEMO *)
    S103_M_DATA_전송_PLS AT %MW9005.9 : BOOL; (* S103_M_DATA_전송_PLS *)
    S103_M_DATA_전송_SIGN AT %MW9005.10 : BOOL; (* S103_M_DATA_전송_SIGN *)
    S103_M_DATA_전송_완료 AT %MW9005.11 : BOOL; (* S103_M_DATA_전송_완료 *)
    S103_M_FRT_안착OK_POS AT %MW2004.8 : BOOL;
    S103_M_FRT_취출OK_POS AT %MW2004.9 : BOOL;
    S103_M_GATE_DOOR_NORMAL AT %MW2006.4 : BOOL;
    S103_M_GATE_ESTOP_NORMAR AT %MW2006.3 : BOOL;
    S103_M_OP_ESTOP_NORMAL AT %MW2006.1 : BOOL;
    S103_M_RB_ESTOP_NORMAL AT %MW2006.2 : BOOL;
    S103_M_SAFTY_NO_INT AT %MW2004.4 : BOOL;
    S103_M_SEMI_자동_모드 AT %MW2000.2 : BOOL;
    S103_M_SEQ AT %MW10100 : WORD; (* S103_M_SEQ *)
    S103_M_STN_FRT_FLR_로딩완료 AT %MW2001.8 : BOOL;
    S103_M_STN_차종_NONE AT %MW2002.1 : BOOL;
    S103_M_STN_차종_ON AT %MW2002.0 : BOOL;
    S103_M_VIN_NO_1_2 AT %MW10111 : WORD; (* S103_M_VIN_NO_1_2 *)
    S103_M_VIN_NO_3_4 AT %MW10112 : WORD; (* S103_M_VIN_NO_3_4 *)
    S103_M_VIN_NO_5_6 AT %MW10113 : WORD; (* S103_M_VIN_NO_5_6 *)
    S103_M_VIN_NO_7_8 AT %MW10114 : WORD; (* S103_M_VIN_NO_7_8 *)
    S103_M_VIN_NO_9_10 AT %MW10115 : WORD; (* S103_M_VIN_NO_9_10 *)
    S103_M_공정_HOME_POSI AT %MW2004.0 : BOOL;
    S103_M_공정_SAFETY_NORMAL AT %MW2006.7 : BOOL;
    S103_M_공정_간섭무 AT %MW2004.1 : BOOL;
    S103_M_공정_제품감지_OFF AT %MW2001.4 : BOOL;
    S103_M_공정_제품감지_ON AT %MW2001.3 : BOOL;
    S103_M_공정_통신이상 AT %MW2024.0 : BOOL;
    S103_M_부저_정지_보조 AT %MW2000.11 : BOOL;
    S103_M_수동_모드 AT %MW2000.3 : BOOL;
    S103_M_운전준비_ON AT %MW2000.0 : BOOL;
    S103_M_이상_리셋_보조 AT %MW2000.10 : BOOL;
    S103_M_자동_START AT %MW2000.5 : BOOL;
    S103_M_자동_모드 AT %MW2000.1 : BOOL;
    S103_M_자동_운전중 AT %MW2000.4 : BOOL;
    S103_M_작업_완료 AT %MW2001.0 : BOOL;
    S103_M_작업_완료_보조 AT %MW2000.9 : BOOL;
    S103_M_제품감지_이상 AT %MW2014.0 : BOOL;
    S103_M_차종1_AX AT %MW10101.0 : BOOL; (* S103_M_차종1_AX *)
    S103_M_차종1_B AT %MW10101.1 : BOOL; (* S103_M_차종1_B *)
    S103_M_차종1_C AT %MW10101.2 : BOOL; (* S103_M_차종1_C *)
    S103_M_차종1_D AT %MW10101.3 : BOOL; (* S103_M_차종1_D *)
    S103_M_차종1_E AT %MW10101.4 : BOOL; (* S103_M_차종1_E *)
    S103_M_차종1_F AT %MW10101.5 : BOOL; (* S103_M_차종1_F *)
    S103_M_차종1_G AT %MW10101.6 : BOOL; (* S103_M_차종1_G *)
    S103_M_차종1_H AT %MW10101.7 : BOOL; (* S103_M_차종1_H *)
    S103_M_차종2_3DR AT %MW10101.8 : BOOL; (* S103_M_차종2_3DR *)
    S103_M_차종2_4DR AT %MW10101.9 : BOOL; (* S103_M_차종2_4DR *)
    S103_M_차종2_5DR AT %MW10101.10 : BOOL; (* S103_M_차종2_5DR *)
    S103_M_차종2_SP1 AT %MW10101.12 : BOOL; (* S103_M_차종2_SP1 *)
    S103_M_차종2_SP2 AT %MW10101.13 : BOOL; (* S103_M_차종2_SP2 *)
    S103_M_차종2_WGN AT %MW10101.11 : BOOL; (* S103_M_차종2_WGN *)
    S103_M_차종3_LHD AT %MW10101.14 : BOOL; (* S103_M_차종3_LHD *)
    S103_M_차종3_RHD AT %MW10101.15 : BOOL; (* S103_M_차종3_RHD *)
    S103_M_차종4_EEC AT %MW10102.3 : BOOL; (* S103_M_차종4_EEC *)
    S103_M_차종4_SP1 AT %MW10102.8 : BOOL; (* S103_M_차종4_SP1 *)
    S103_M_차종4_SP2 AT %MW10102.9 : BOOL; (* S103_M_차종4_SP2 *)
    S103_M_차종4_SP3 AT %MW10102.11 : BOOL; (* S103_M_차종4_SP3 *)
    S103_M_차종4_SP4 AT %MW10102.12 : BOOL; (* S103_M_차종4_SP4 *)
    S103_M_차종4_SP5 AT %MW10102.13 : BOOL; (* S103_M_차종4_SP5 *)
    S103_M_차종4_SP6 AT %MW10102.14 : BOOL; (* S103_M_차종4_SP6 *)
    S103_M_차종4_SP7 AT %MW10102.15 : BOOL; (* S103_M_차종4_SP7 *)
    S103_M_차종4_내수 AT %MW10102.0 : BOOL; (* S103_M_차종4_내수 *)
    S103_M_차종4_러시아 AT %MW10102.10 : BOOL; (* S103_M_차종4_러시아 *)
    S103_M_차종4_북미 AT %MW10102.2 : BOOL; (* S103_M_차종4_북미 *)
    S103_M_차종4_브라질 AT %MW10102.7 : BOOL; (* S103_M_차종4_브라질 *)
    S103_M_차종4_수출 AT %MW10102.1 : BOOL; (* S103_M_차종4_수출 *)
    S103_M_차종4_중국 AT %MW10102.6 : BOOL; (* S103_M_차종4_중국 *)
    S103_M_차종4_중동 AT %MW10102.5 : BOOL; (* S103_M_차종4_중동 *)
    S103_M_차종4_호주 AT %MW10102.4 : BOOL; (* S103_M_차종4_호주 *)
    S103_M_차종5_AT AT %MW10103.1 : BOOL; (* S103_M_차종5_AT *)
    S103_M_차종5_MT AT %MW10103.0 : BOOL; (* S103_M_차종5_MT *)
    S103_M_차종5_SP1 AT %MW10103.2 : BOOL; (* S103_M_차종5_SP1 *)
    S103_M_차종6_DSROOF AT %MW10103.6 : BOOL; (* S103_M_차종6_DSROOF *)
    S103_M_차종6_SP1 AT %MW10103.7 : BOOL; (* S103_M_차종6_SP1 *)
    S103_M_차종6_썬루프 AT %MW10103.4 : BOOL; (* S103_M_차종6_썬루프 *)
    S103_M_차종6_일반루프 AT %MW10103.3 : BOOL; (* S103_M_차종6_일반루프 *)
    S103_M_차종6_파노라마루프 AT %MW10103.5 : BOOL; (* S103_M_차종6_파노라마루프 *)
    S103_M_차종7_DSL AT %MW10103.9 : BOOL; (* S103_M_차종7_DSL *)
    S103_M_차종7_GSL AT %MW10103.8 : BOOL; (* S103_M_차종7_GSL *)
    S103_M_차종7_SP1 AT %MW10103.10 : BOOL; (* S103_M_차종7_SP1 *)
    S103_M_차종7_SP2 AT %MW10103.11 : BOOL; (* S103_M_차종7_SP2 *)
    S103_M_차종7_SP3 AT %MW10103.12 : BOOL; (* S103_M_차종7_SP3 *)
    S103_M_차종7_SP4 AT %MW10103.13 : BOOL; (* S103_M_차종7_SP4 *)
    S103_M_차종7_SP5 AT %MW10103.14 : BOOL; (* S103_M_차종7_SP5 *)
    S103_M_차종7_SP6 AT %MW10103.15 : BOOL; (* S103_M_차종7_SP6 *)
    S103_M_차종8_2WD AT %MW10104.0 : BOOL; (* S103_M_차종8_2WD *)
    S103_M_차종8_4WD AT %MW10104.1 : BOOL; (* S103_M_차종8_4WD *)
    S103_M_차종8_SP1 AT %MW10104.2 : BOOL; (* S103_M_차종8_SP1 *)
    S103_M_차종9_MPI AT %MW10104.3 : BOOL; (* S103_M_차종9_MPI *)
    S103_M_차종9_SP1 AT %MW10104.5 : BOOL; (* S103_M_차종9_SP1 *)
    S103_M_차종9_SP10 AT %MW10104.14 : BOOL; (* S103_M_차종9_SP10 *)
    S103_M_차종9_SP11 AT %MW10104.15 : BOOL; (* S103_M_차종9_SP11 *)
    S103_M_차종9_SP2 AT %MW10104.6 : BOOL; (* S103_M_차종9_SP2 *)
    S103_M_차종9_SP3 AT %MW10104.7 : BOOL; (* S103_M_차종9_SP3 *)
    S103_M_차종9_SP4 AT %MW10104.8 : BOOL; (* S103_M_차종9_SP4 *)
    S103_M_차종9_SP5 AT %MW10104.9 : BOOL; (* S103_M_차종9_SP5 *)
    S103_M_차종9_SP6 AT %MW10104.10 : BOOL; (* S103_M_차종9_SP6 *)
    S103_M_차종9_SP7 AT %MW10104.11 : BOOL; (* S103_M_차종9_SP7 *)
    S103_M_차종9_SP8 AT %MW10104.12 : BOOL; (* S103_M_차종9_SP8 *)
    S103_M_차종9_SP9 AT %MW10104.13 : BOOL; (* S103_M_차종9_SP9 *)
    S103_M_차종9_T_GDI AT %MW10104.4 : BOOL; (* S103_M_차종9_T_GDI *)
    S103_M_차종_AS AT %MW10110.9 : BOOL; (* S103_M_차종_AS *)
    S103_M_차종_OPT1_R_RACK_무 AT %MW10105.3 : BOOL; (* S103_M_차종_OPT1_R_RACK_무 *)
    S103_M_차종_OPT1_R_RACK_유 AT %MW10105.2 : BOOL; (* S103_M_차종_OPT1_R_RACK_유 *)
    S103_M_차종_OPT1_SP1 AT %MW10105.10 : BOOL; (* S103_M_차종_OPT1_SP1 *)
    S103_M_차종_OPT1_SP2 AT %MW10105.11 : BOOL; (* S103_M_차종_OPT1_SP2 *)
    S103_M_차종_OPT1_SP3 AT %MW10105.12 : BOOL; (* S103_M_차종_OPT1_SP3 *)
    S103_M_차종_OPT1_SP4 AT %MW10105.13 : BOOL; (* S103_M_차종_OPT1_SP4 *)
    S103_M_차종_OPT1_SP5 AT %MW10105.14 : BOOL; (* S103_M_차종_OPT1_SP5 *)
    S103_M_차종_OPT1_SP6 AT %MW10105.15 : BOOL; (* S103_M_차종_OPT1_SP6 *)
    S103_M_차종_OPT1_S_REP_EATER_무 AT %MW10105.7 : BOOL; (* S103_M_차종_OPT1_S_REP_EATER_무 *)
    S103_M_차종_OPT1_S_REP_EATER_유 AT %MW10105.6 : BOOL; (* S103_M_차종_OPT1_S_REP_EATER_유 *)
    S103_M_차종_OPT1_VAN_무 AT %MW10105.9 : BOOL; (* S103_M_차종_OPT1_VAN_무 *)
    S103_M_차종_OPT1_VAN_유 AT %MW10105.8 : BOOL; (* S103_M_차종_OPT1_VAN_유 *)
    S103_M_차종_OPT1_슬라이딩_무 AT %MW10105.1 : BOOL; (* S103_M_차종_OPT1_슬라이딩_무 *)
    S103_M_차종_OPT1_슬라이딩_유 AT %MW10105.0 : BOOL; (* S103_M_차종_OPT1_슬라이딩_유 *)
    S103_M_차종_OPT1_폴딩_무 AT %MW10105.5 : BOOL; (* S103_M_차종_OPT1_폴딩_무 *)
    S103_M_차종_OPT1_폴딩_유 AT %MW10105.4 : BOOL; (* S103_M_차종_OPT1_폴딩_유 *)
    S103_M_차종_OPT2_SP_WORD1 AT %MW10106 : WORD; (* S103_M_차종_OPT2_SP_WORD1 *)
    S103_M_차종_OPT3_SP_WORD2 AT %MW10107 : WORD; (* S103_M_차종_OPT3_SP_WORD2 *)
    S103_M_차종_OPT4_SP_WORD3 AT %MW10108 : WORD; (* S103_M_차종_OPT4_SP_WORD3 *)
    S103_M_차종_OPT5_SP_WORD4 AT %MW10109 : WORD; (* S103_M_차종_OPT5_SP_WORD4 *)
    S103_M_차종_SP1 AT %MW10110.0 : BOOL; (* S103_M_차종_SP1 *)
    S103_M_차종_SP2 AT %MW10110.1 : BOOL; (* S103_M_차종_SP2 *)
    S103_M_차종_SP3 AT %MW10110.2 : BOOL; (* S103_M_차종_SP3 *)
    S103_M_차종_SP4 AT %MW10110.3 : BOOL; (* S103_M_차종_SP4 *)
    S103_M_차종_SP5 AT %MW10110.4 : BOOL; (* S103_M_차종_SP5 *)
    S103_M_차종_SP6 AT %MW10110.5 : BOOL; (* S103_M_차종_SP6 *)
    S103_M_차종_SP7 AT %MW10110.6 : BOOL; (* S103_M_차종_SP7 *)
    S103_M_차종_SP8 AT %MW10110.7 : BOOL; (* S103_M_차종_SP8 *)
    S103_M_차종_SP9 AT %MW10110.15 : BOOL; (* S103_M_차종_SP9 *)
    S103_M_차종_공대차 AT %MW10110.12 : BOOL; (* S103_M_차종_공대차 *)
    S103_M_차종_공차 AT %MW10110.10 : BOOL; (* S103_M_차종_공차 *)
    S103_M_차종_불량대차 AT %MW10110.13 : BOOL; (* S103_M_차종_불량대차 *)
    S103_M_차종_불량차 AT %MW10110.11 : BOOL; (* S103_M_차종_불량차 *)
    S103_M_차종_비축 AT %MW10110.8 : BOOL; (* S103_M_차종_비축 *)
    S103_M_차종_취출대차 AT %MW10110.14 : BOOL; (* S103_M_차종_취출대차 *)
    S103_M_총괄_CP_이상 AT %MW2009.7 : BOOL;
    S103_M_총괄_CT_이상 AT %MW2010.4 : BOOL;
    S103_M_총괄_EOCR_이상 AT %MW2009.8 : BOOL;
    S103_M_총괄_INV_이상 AT %MW2009.9 : BOOL;
    S103_M_총괄_LS_이상 AT %MW2009.15 : BOOL;
    S103_M_총괄_MATCH_이상 AT %MW2010.0 : BOOL;
    S103_M_총괄_MC_이상 AT %MW2009.13 : BOOL;
    S103_M_총괄_MOTOR_이상 AT %MW2010.3 : BOOL;
    S103_M_총괄_NFB_이상 AT %MW2009.11 : BOOL;
    S103_M_총괄_ROBOT_이상 AT %MW2010.1 : BOOL;
    S103_M_총괄_SAFETY_이상 AT %MW2009.2 : BOOL;
    S103_M_총괄_SRV_이상 AT %MW2009.10 : BOOL;
    S103_M_총괄_공기압_이상 AT %MW2009.3 : BOOL;
    S103_M_총괄_비상정지_이상 AT %MW2009.1 : BOOL;
    S103_M_총괄_사양_이상 AT %MW2009.6 : BOOL;
    S103_M_총괄_오버런_이상 AT %MW2009.12 : BOOL;
    S103_M_총괄_용점타점수_이상 AT %MW2010.2 : BOOL;
    S103_M_총괄_이상 AT %MW2009.0 : BOOL;
    S103_M_총괄_제품감지_이상 AT %MW2009.4 : BOOL;
    S103_M_총괄_차종_이상 AT %MW2009.5 : BOOL;
    S103_M_총괄_통신_이상 AT %MW2009.14 : BOOL;
    S103_PRS_AX_제품감지_CHECK1 AT %MW86301.0 : BOOL; (* 입력 접점 00 *)
    S103_PRS_AX_제품감지_CHECK2 AT %MW86301.1 : BOOL; (* 입력 접점 01 *)
    S103_R103_1_CTYPE_MOVE : FB407_Car_Type_Move_Stn_v1;
    S103_R103_2_CTYPE_MOVE : FB407_Car_Type_Move_Stn_v1;
    S103_RS_AX_래치_전진1 AT %MW86300.0 : BOOL; (* 입력 접점 00 *)
    S103_RS_AX_래치_전진2 AT %MW86300.2 : BOOL; (* 입력 접점 02 *)
    S103_RS_AX_래치_전진3 AT %MW86300.4 : BOOL; (* 입력 접점 04 *)
    S103_RS_AX_래치_전진4 AT %MW86300.6 : BOOL; (* 입력 접점 06 *)
    S103_RS_AX_래치_후진1 AT %MW86300.1 : BOOL; (* 입력 접점 01 *)
    S103_RS_AX_래치_후진2 AT %MW86300.3 : BOOL; (* 입력 접점 03 *)
    S103_RS_AX_래치_후진3 AT %MW86300.5 : BOOL; (* 입력 접점 05 *)
    S103_RS_AX_래치_후진4 AT %MW86300.7 : BOOL; (* 입력 접점 07 *)
    S103_SOL_AX_래치_전진 AT %MW96303.0 : BOOL; (* 출력 접점 00 *)
    S103_SOL_AX_래치_후진 AT %MW96303.1 : BOOL; (* 출력 접점 01 *)
    S103_공기압_AIR_CHECK AT %MW86302.14 : BOOL; (* 입력 접점 14 *)
    S103_운전준비 : TON;
    S103_전진_ON AT %MW2048.1 : BOOL;
    S103_후진_ON AT %MW2048.2 : BOOL;
    S104_HOME AT %MW2548.0 : BOOL;
    S104_M_ACT_선택_1 AT %MW2540.0 : BOOL;
    S104_M_ACT_선택_10 AT %MW2540.9 : BOOL;
    S104_M_ACT_선택_11 AT %MW2540.10 : BOOL;
    S104_M_ACT_선택_12 AT %MW2540.11 : BOOL;
    S104_M_ACT_선택_13 AT %MW2540.12 : BOOL;
    S104_M_ACT_선택_14 AT %MW2540.13 : BOOL;
    S104_M_ACT_선택_15 AT %MW2540.14 : BOOL;
    S104_M_ACT_선택_16 AT %MW2540.15 : BOOL;
    S104_M_ACT_선택_17 AT %MW2541.0 : BOOL;
    S104_M_ACT_선택_18 AT %MW2541.1 : BOOL;
    S104_M_ACT_선택_19 AT %MW2541.2 : BOOL;
    S104_M_ACT_선택_2 AT %MW2540.1 : BOOL;
    S104_M_ACT_선택_20 AT %MW2541.3 : BOOL;
    S104_M_ACT_선택_21 AT %MW2541.4 : BOOL;
    S104_M_ACT_선택_22 AT %MW2541.5 : BOOL;
    S104_M_ACT_선택_23 AT %MW2541.6 : BOOL;
    S104_M_ACT_선택_24 AT %MW2541.7 : BOOL;
    S104_M_ACT_선택_25 AT %MW2541.8 : BOOL;
    S104_M_ACT_선택_26 AT %MW2541.9 : BOOL;
    S104_M_ACT_선택_27 AT %MW2541.10 : BOOL;
    S104_M_ACT_선택_28 AT %MW2541.11 : BOOL;
    S104_M_ACT_선택_29 AT %MW2541.12 : BOOL;
    S104_M_ACT_선택_3 AT %MW2540.2 : BOOL;
    S104_M_ACT_선택_30 AT %MW2541.13 : BOOL;
    S104_M_ACT_선택_31 AT %MW2541.14 : BOOL;
    S104_M_ACT_선택_32 AT %MW2541.15 : BOOL;
    S104_M_ACT_선택_4 AT %MW2540.3 : BOOL;
    S104_M_ACT_선택_5 AT %MW2540.4 : BOOL;
    S104_M_ACT_선택_6 AT %MW2540.5 : BOOL;
    S104_M_ACT_선택_7 AT %MW2540.6 : BOOL;
    S104_M_ACT_선택_8 AT %MW2540.7 : BOOL;
    S104_M_ACT_선택_9 AT %MW2540.8 : BOOL;
    S104_M_CTIME_OVER_ALRAM AT %MW2506.14 : BOOL;
    S104_M_CTIME_OVER_MUTE AT %MW2506.13 : BOOL;
    S104_M_GATE_DOOR_NORMAL AT %MW2506.4 : BOOL;
    S104_M_GATE_ESTOP_NORMAR AT %MW2506.3 : BOOL;
    S104_M_LC_NORMAL AT %MW2506.5 : BOOL;
    S104_M_MAT_NORMAL AT %MW2506.6 : BOOL;
    S104_M_OP_ESTOP_NORMAL AT %MW2506.1 : BOOL;
    S104_M_RB_ESTOP_NORMAL AT %MW2506.2 : BOOL;
    S104_M_S326_CN_MATCH_OK AT %MW2501.14 : BOOL;
    S104_M_S326_CT_MATCH_OK AT %MW2501.15 : BOOL;
    S104_M_SAFTY_NO_INT AT %MW2504.4 : BOOL;
    S104_M_SEMI_자동_모드 AT %MW2500.2 : BOOL;
    S104_M_SKID_OFF AT %MW2501.6 : BOOL;
    S104_M_SKID_ON AT %MW2501.5 : BOOL;
    S104_M_공정_HOME_POSI AT %MW2504.0 : BOOL;
    S104_M_공정_SAFETY_NORMAL AT %MW2506.7 : BOOL;
    S104_M_공정_간섭무 AT %MW2504.1 : BOOL;
    S104_M_공정_제품감지_OFF AT %MW2501.4 : BOOL;
    S104_M_공정_제품감지_ON AT %MW2501.3 : BOOL;
    S104_M_공정_차종_NONE AT %MW2502.1 : BOOL;
    S104_M_공정_차종_ON AT %MW2502.0 : BOOL;
    S104_M_공정_차종_보조 AT %MW2502.2 : BOOL;
    S104_M_공정_통신이상 AT %MW2524.0 : BOOL;
    S104_M_부저_정지_보조 AT %MW2500.11 : BOOL;
    S104_M_수동_모드 AT %MW2500.3 : BOOL;
    S104_M_운전준비_ON AT %MW2500.0 : BOOL;
    S104_M_이상_리셋_보조 AT %MW2500.10 : BOOL;
    S104_M_자동_START AT %MW2500.5 : BOOL;
    S104_M_자동_모드 AT %MW2500.1 : BOOL;
    S104_M_자동_운전중 AT %MW2500.4 : BOOL;
    S104_M_작업_완료 AT %MW2501.0 : BOOL;
    S104_M_총괄_CP_이상 AT %MW2509.7 : BOOL;
    S104_M_총괄_CT_이상 AT %MW2510.4 : BOOL;
    S104_M_총괄_EOCR_이상 AT %MW2509.8 : BOOL;
    S104_M_총괄_INV_이상 AT %MW2509.9 : BOOL;
    S104_M_총괄_LS_이상 AT %MW2509.15 : BOOL;
    S104_M_총괄_MATCH_이상 AT %MW2510.0 : BOOL;
    S104_M_총괄_MC_이상 AT %MW2509.13 : BOOL;
    S104_M_총괄_MOTOR_이상 AT %MW2510.3 : BOOL;
    S104_M_총괄_NFB_이상 AT %MW2509.11 : BOOL;
    S104_M_총괄_ROBOT_이상 AT %MW2510.1 : BOOL;
    S104_M_총괄_SAFETY_이상 AT %MW2509.2 : BOOL;
    S104_M_총괄_SRV_이상 AT %MW2509.10 : BOOL;
    S104_M_총괄_공기압_이상 AT %MW2509.3 : BOOL;
    S104_M_총괄_비상정지_이상 AT %MW2509.1 : BOOL;
    S104_M_총괄_사양_이상 AT %MW2509.6 : BOOL;
    S104_M_총괄_오버런_이상 AT %MW2509.12 : BOOL;
    S104_M_총괄_용점타점수_이상 AT %MW2510.2 : BOOL;
    S104_M_총괄_이상 AT %MW2509.0 : BOOL;
    S104_M_총괄_제품감지_이상 AT %MW2509.4 : BOOL;
    S104_M_총괄_차종_이상 AT %MW2509.5 : BOOL;
    S104_M_총괄_통신_이상 AT %MW2509.14 : BOOL;
    S104_운전준비 : TON;
    S104_전진_ON AT %MW2548.1 : BOOL;
    S104_후진_ON AT %MW2548.2 : BOOL;
    S161_M_공정_차종_AX AT %MW3002.3 : BOOL;
    S161_M_수동_모드 AT %MW3000.3 : BOOL;
    S161_M_자동_START AT %MW3000.5 : BOOL;
    S161_M_자동_운전중 AT %MW3000.4 : BOOL;
    S161_M_작업완료 AT %MW3001.0 : BOOL;
    S161_M_전체_3축_로봇1차_작업완료 AT %MW3001.1 : BOOL;
    S161_M_전체_용접로보트_1차_작업완료 AT %MW3001.8 : BOOL;
    S161_M_전체_용접로보트_최종_작업완료 AT %MW3001.9 : BOOL;
    S161_M_총괄_이상 AT %MW3009.0 : BOOL;
    SB_APR_RACK2_P_BOX_CP_TRIP AT %MW87211.15 : BOOL;
    SB_DASH_RACK1_P_BOX_CP_TRIP AT %MW87301.15 : BOOL;
    SRV1_M_PS1_DC_LOW AT %MW357.2 : BOOL;
    SRV1_M_PS2_DC_LOW AT %MW357.3 : BOOL;
    SRV1_M_SPD_이상 AT %MW357.1 : BOOL;
    SRV1_M_총괄_이상 AT %MW357.0 : BOOL;
    SRV1_M_통신_이상 AT %MW356.4 : BOOL;
    SRV_PNL_CP_ON AT %MW85363.15 : BOOL;
    SRV_PNL_PS_NOMAL AT %MW85363.12 : BOOL;
    SRV_PNL_SPD_NOMAL AT %MW85203.9 : BOOL;
    SW6 : BOOL;
    T101_자동 : TON;
    T102_자동 : TON;
    T103_자동 : TON;
    T104_자동 : TON;
    TEST : BOOL;
    TEST1 : BOOL;
    TON_GATE10_OPEN : TON;
    TON_GATE11_OPEN : TON;
    TON_GATE12_OPEN : TON;
    TON_부저_정지 : TON;
    TON_부저_정지1 : TON;
    T_GB10_CP_OFF_DELAY : TON;
    T_GB10_통신_이상_DELAY : TON;
    T_GB11_CP_OFF_DELAY : TON;
    T_GB11_통신_이상_DELAY : TON;
    T_GB12_CP_OFF_DELAY : TON;
    T_GB12_통신_이상_DELAY : TON;
    _0004_EB01_CFG_ER AT %MX59360 : BOOL; (* EB 구성 에러 *)
    _0004_EB01_DEER AT %MX59361 : BOOL; (* EB 운전 중 탈락 *)
    _0004_EB04_CFG_ER AT %MX59400 : BOOL; (* EB 구성 에러 *)
    _0004_EB04_DEER AT %MX59401 : BOOL; (* EB 운전 중 탈락 *)
    _0004_EB05_CFG_ER AT %MX59440 : BOOL; (* EB 구성 에러 *)
    _0004_EB05_DEER AT %MX59441 : BOOL; (* EB 운전 중 탈락 *)
    _0004_EB06_CFG_ER AT %MX59480 : BOOL; (* EB 구성 에러 *)
    _0004_EB06_DEER AT %MX59481 : BOOL; (* EB 운전 중 탈락 *)
    _0004_EB07_CFG_ER AT %MX59520 : BOOL; (* EB 구성 에러 *)
    _0004_EB07_DEER AT %MX59521 : BOOL; (* EB 운전 중 탈락 *)
    _0004_EB08_CFG_ER AT %MX59560 : BOOL; (* EB 구성 에러 *)
    _0004_EB08_DEER AT %MX59561 : BOOL; (* EB 운전 중 탈락 *)
    _0004_EB09_CFG_ER AT %MX59600 : BOOL; (* EB 구성 에러 *)
    _0004_EB09_DEER AT %MX59601 : BOOL; (* EB 운전 중 탈락 *)
    _0004_EB10_CFG_ER AT %MX59640 : BOOL; (* EB 구성 에러 *)
    _0004_EB10_DEER AT %MX59641 : BOOL; (* EB 운전 중 탈락 *)
    _0005_EB11_S00_SVC_ER AT %MW185024.7 : BOOL; (* 통신 서비스 에러 *)
    _0005_EB11_S01_SVC_ER AT %MW185024.15 : BOOL; (* 통신 서비스 에러 *)
    _0005_EB12_S00_SVC_ER AT %MW185058.7 : BOOL; (* 통신 서비스 에러 *)
    _0005_EB12_S01_SVC_ER AT %MW185058.15 : BOOL; (* 통신 서비스 에러 *)
    _0005_EB13_S00_SVC_ER AT %MW185092.7 : BOOL; (* 통신 서비스 에러 *)
    _0005_EB13_S01_SVC_ER AT %MW185092.15 : BOOL; (* 통신 서비스 에러 *)
    _0005_EB20_CFG_ER AT %MW185124.0 : BOOL; (* EB 구성 에러 *)
    _0005_EB20_DEER AT %MW185124.1 : BOOL; (* EB 운전 중 탈락 *)
    _0005_EB20_IO_DEER AT %MW185125.2 : BOOL; (* EB IO 탈락 에러 *)
    _0005_EB20_IO_TYER AT %MW185125.1 : BOOL; (* EB IO 타입 에러 *)
    _0006_EB10_CFG_ER AT %MW186022.0 : BOOL; (* EB 구성 에러 *)
    _0006_EB10_DEER AT %MW186022.1 : BOOL; (* EB 운전 중 탈락 *)
    _0006_EB10_IO_DEER AT %MW186023.2 : BOOL; (* EB IO 탈락 에러 *)
    _0006_EB10_IO_TYER AT %MW186023.1 : BOOL; (* EB IO 타입 에러 *)
    _0006_EB20_CFG_ER AT %MW186028.0 : BOOL; (* EB 구성 에러 *)
    _0006_EB20_DEER AT %MW186028.1 : BOOL; (* EB 운전 중 탈락 *)
    _0006_EB20_IO_DEER AT %MW186029.2 : BOOL; (* EB IO 탈락 에러 *)
    _0006_EB20_IO_TYER AT %MW186029.1 : BOOL; (* EB IO 타입 에러 *)
    _0006_EB30_CFG_ER AT %MW186034.0 : BOOL; (* EB 구성 에러 *)
    _0006_EB30_DEER AT %MW186034.1 : BOOL; (* EB 운전 중 탈락 *)
    _0006_EB30_IO_DEER AT %MW186035.2 : BOOL; (* EB IO 탈락 에러 *)
    _0006_EB30_IO_TYER AT %MW186035.1 : BOOL; (* EB IO 타입 에러 *)
    _0007_EB10_CFG_ER AT %MW187022.0 : BOOL; (* EB 구성 에러 *)
    _0007_EB10_DEER AT %MW187022.1 : BOOL; (* EB 운전 중 탈락 *)
    _0007_EB10_IO_DEER AT %MW187023.2 : BOOL; (* EB IO 탈락 에러 *)
    _0007_EB10_IO_TYER AT %MW187023.1 : BOOL; (* EB IO 타입 에러 *)
    _0007_EB21_CFG_ER AT %MW187028.0 : BOOL; (* EB 구성 에러 *)
    _0007_EB21_DEER AT %MW187028.1 : BOOL; (* EB 운전 중 탈락 *)
    _0007_EB21_IO_DEER AT %MW187029.2 : BOOL; (* EB IO 탈락 에러 *)
    _0007_EB21_IO_TYER AT %MW187029.1 : BOOL; (* EB IO 타입 에러 *)
    _0007_EB30_CFG_ER AT %MW187034.0 : BOOL; (* EB 구성 에러 *)
    _0007_EB30_DEER AT %MW187034.1 : BOOL; (* EB 운전 중 탈락 *)
    _0007_EB30_IO_DEER AT %MW187035.2 : BOOL; (* EB IO 탈락 에러 *)
    _0007_EB30_IO_TYER AT %MW187035.1 : BOOL; (* EB IO 타입 에러 *)
    _0007_EB63_CFG_ER AT %MW187040.0 : BOOL; (* EB 구성 에러 *)
    _0007_EB63_DEER AT %MW187040.1 : BOOL; (* EB 운전 중 탈락 *)
    _0007_EB63_IO_DEER AT %MW187041.2 : BOOL; (* EB IO 탈락 에러 *)
    _0007_EB63_IO_TYER AT %MW187041.1 : BOOL; (* EB IO 타입 에러 *)
    로보트제외 : BOOL;
    셔틀_M_MOVE_전진_보조 AT %MW504.1 : BOOL;
    셔틀_M_MOVE_전진단 AT %MW504.3 : BOOL;
    셔틀_M_MOVE_후진단 AT %MW504.4 : BOOL;
    셔틀_M_작업완료 AT %MW501.0 : BOOL;
    전체_M_GATE_CYCLE_정지 AT %MW308.0 : BOOL; (* 전체 M GATE CYCLE STOP *)
    전체_M_GATE_비상정지_정상 AT %MW308.4 : BOOL;
    전체_M_GATE_열림_조건 AT %MW308.3 : BOOL; (* 전체 M GATE 열림 조건 *)
    전체_M_GATE_자동기동 AT %MW308.1 : BOOL; (* 전체 M GATE 자동기동 *)
    전체_M_운전준비_보조 AT %MW308.5 : BOOL;
    전체_M_이상_리셋 AT %MW308.2 : BOOL; (* 전체 M 이상 리셋 *)
    전체_OP_M_총괄_비상정지_정상 AT %MW304.2 : BOOL; (* 전체 OP M 총괄 비상정지 정상 *)
    전체_공정_M_총괄_비상정지_정상 AT %MW304.1 : BOOL; (* 전체 공정 M 총괄 비상정지 정상 *)
    전체_라인_M_총괄_CP_OFF AT %MW300.7 : BOOL;
    전체_라인_M_총괄_CT_이상 AT %MW301.4 : BOOL;
    전체_라인_M_총괄_EOCR_이상 AT %MW300.8 : BOOL;
    전체_라인_M_총괄_GATE_OPEN_이상 AT %MW301.5 : BOOL;
    전체_라인_M_총괄_INV_이상 AT %MW300.9 : BOOL;
    전체_라인_M_총괄_LS_이상 AT %MW300.15 : BOOL;
    전체_라인_M_총괄_MATCH_이상 AT %MW301.0 : BOOL;
    전체_라인_M_총괄_MC_이상 AT %MW300.13 : BOOL;
    전체_라인_M_총괄_MOTOR_이상 AT %MW301.3 : BOOL;
    전체_라인_M_총괄_NFB_이상 AT %MW300.11 : BOOL;
    전체_라인_M_총괄_PS_DC_LOW AT %MW301.7 : BOOL;
    전체_라인_M_총괄_ROBOT_이상 AT %MW301.1 : BOOL;
    전체_라인_M_총괄_SAFETY_이상 AT %MW300.2 : BOOL;
    전체_라인_M_총괄_SAG_이상 AT %MW301.6 : BOOL;
    전체_라인_M_총괄_SPD_이상 AT %MW301.8 : BOOL;
    전체_라인_M_총괄_SRV_이상 AT %MW300.10 : BOOL;
    전체_라인_M_총괄_공기압_이상 AT %MW300.3 : BOOL;
    전체_라인_M_총괄_비상정지_이상 AT %MW300.1 : BOOL;
    전체_라인_M_총괄_비상정지_정상 AT %MW304.0 : BOOL; (* 전체 라인 M 총괄 비상정지 정상 *)
    전체_라인_M_총괄_사양_이상 AT %MW300.6 : BOOL;
    전체_라인_M_총괄_오버런_이상 AT %MW300.12 : BOOL;
    전체_라인_M_총괄_용점타점수_이상 AT %MW301.2 : BOOL;
    전체_라인_M_총괄_이상 AT %MW300.0 : BOOL;
    전체_라인_M_총괄_제품감지_이상 AT %MW300.4 : BOOL;
    전체_라인_M_총괄_차종_이상 AT %MW300.5 : BOOL;
    전체_라인_M_총괄_통신_이상 AT %MW300.14 : BOOL;
END_VAR

TYPE S101_3AXIS_OUTPUT :
STRUCT
END_STRUCT;
END_TYPE

TYPE S101_3AXIS_INPUT :
STRUCT
END_STRUCT;
END_TYPE

FUNCTION_BLOCK FB406_Car_Type_Move_Line_v1
VAR_INPUT RETAIN
    FWD_Pulse : BOOL;
    RET_Pulse : BOOL;
END_VAR
VAR_IN_OUT
    Source_DB : ARRAY[0..499] OF WORD;
END_VAR
VAR_INPUT
    Start_Add : INT;
    Stn_AMTG : INT;
    Word_per_Stn : INT;
    Cpu_Run_Pulse : BOOL;
END_VAR
VAR_OUTPUT
    Complete : BOOL;
END_VAR
VAR
    END : INT;
    Number_of_Array : INT;
    Temp1 : INT;
END_VAR

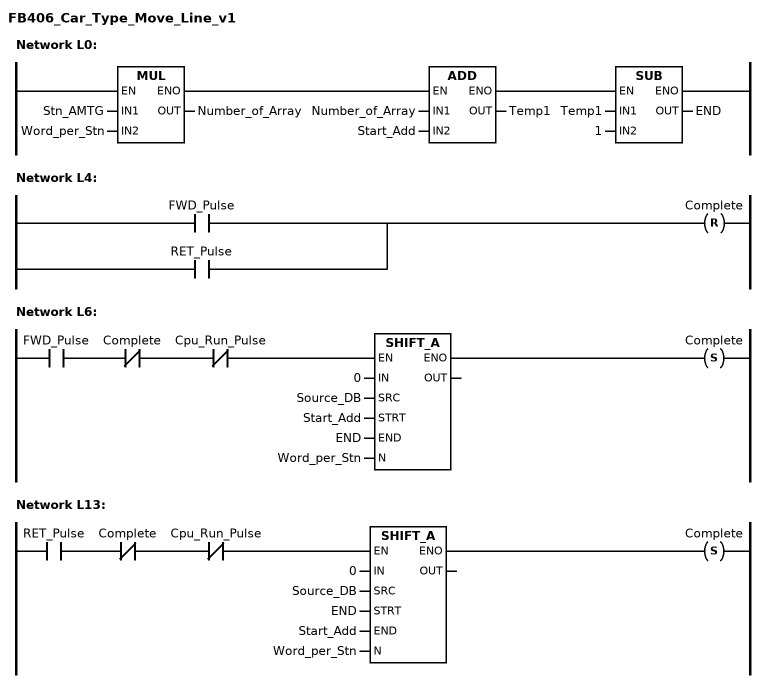
(* Rung L0 *)
Number_of_Array := Stn_AMTG * Word_per_Stn;
Temp1 := Number_of_Array + Start_Add;
END := Temp1 - 1;
(* Rung L4 *)
IF FWD_Pulse OR RET_Pulse THEN Complete := FALSE; END_IF;
(* Rung L6 *)
IF FWD_Pulse AND NOT Complete AND NOT Cpu_Run_Pulse THEN
    SHIFT_A(IN := 0, SRC := Source_DB, STRT := Start_Add, END := END, N := Word_per_Stn);
    Complete := TRUE;
END_IF;
(* Rung L13 *)
IF RET_Pulse AND NOT Complete AND NOT Cpu_Run_Pulse THEN
    SHIFT_A(IN := 0, SRC := Source_DB, STRT := END, END := Start_Add, N := Word_per_Stn);
    Complete := TRUE;
END_IF;
END_FUNCTION_BLOCK

FUNCTION_BLOCK FB407_Car_Type_Move_Stn_v1
VAR_INPUT RETAIN
    FWD_Pulse : BOOL;
    RET_Pulse : BOOL;
END_VAR
VAR_IN_OUT
    Source_DB : ARRAY[0..999] OF WORD;
    Dest_DB : ARRAY[0..999] OF WORD;
END_VAR
VAR_INPUT
    Source_Add : INT;
    Dest_Add : INT;
    Word_per_Stn : INT;
    Cpu_Run_Pulse : BOOL;
END_VAR
VAR_OUTPUT
    Complete : BOOL;
END_VAR
VAR
    _t1 : DINT;
    _t2 : DINT;
END_VAR

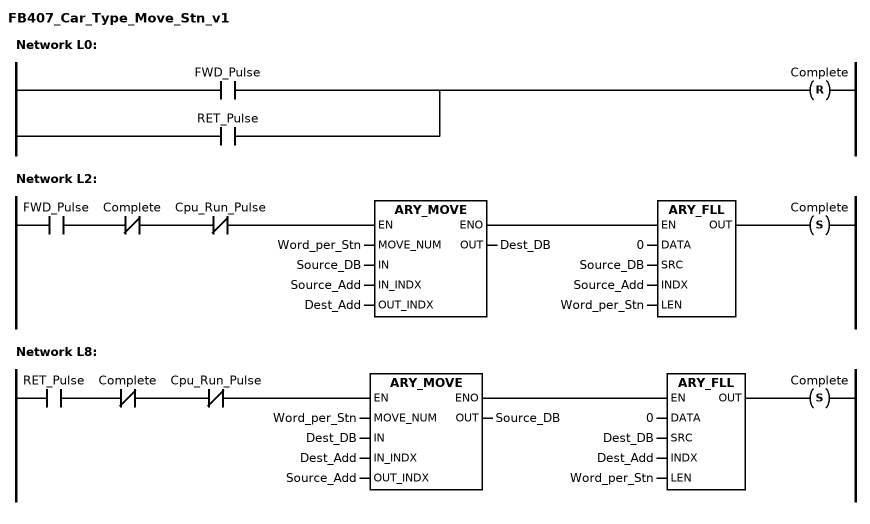
(* Rung L0 *)
IF FWD_Pulse OR RET_Pulse THEN Complete := FALSE; END_IF;
(* Rung L2 *)
IF FWD_Pulse AND NOT Complete AND NOT Cpu_Run_Pulse THEN
    Dest_DB := ARY_MOVE(MOVE_NUM := Word_per_Stn, IN := Source_DB, IN_INDX := Source_Add, OUT_INDX := Dest_Add);
    _t1 := ARY_FLL(DATA := 0, SRC := Source_DB, INDX := Source_Add, LEN := Word_per_Stn);
END_IF;
IF _t1 THEN Complete := TRUE; END_IF;
(* Rung L8 *)
IF RET_Pulse AND NOT Complete AND NOT Cpu_Run_Pulse THEN
    Source_DB := ARY_MOVE(MOVE_NUM := Word_per_Stn, IN := Dest_DB, IN_INDX := Dest_Add, OUT_INDX := Source_Add);
    _t2 := ARY_FLL(DATA := 0, SRC := Dest_DB, INDX := Dest_Add, LEN := Word_per_Stn);
END_IF;
IF _t2 THEN Complete := TRUE; END_IF;
END_FUNCTION_BLOCK

FUNCTION_BLOCK FB409_Car_Type_Clear_v1
VAR_INPUT RETAIN
    Clear_Pulse : BOOL;
END_VAR
VAR_IN_OUT
    Dest_DB : ARRAY[0..999] OF WORD;
END_VAR
VAR_INPUT
    Dest_Add : INT;
    Len_per_Stn_Word : INT;
    Cpu_Run_Pulse : BOOL;
END_VAR
VAR_OUTPUT
    Complete : BOOL;
END_VAR
VAR
    _t1 : DINT;
END_VAR

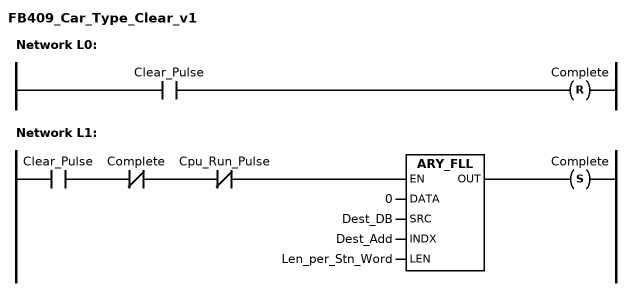
(* Rung L0 *)
IF Clear_Pulse THEN Complete := FALSE; END_IF;
(* Rung L1 *)
IF Clear_Pulse AND NOT Complete AND NOT Cpu_Run_Pulse THEN
    _t1 := ARY_FLL(DATA := 0, SRC := Dest_DB, INDX := Dest_Add, LEN := Len_per_Stn_Word);
END_IF;
IF _t1 THEN Complete := TRUE; END_IF;
END_FUNCTION_BLOCK

FUNCTION_BLOCK FB470_HMI_BType_Modify_LS
VAR_INPUT
    CCR_ON : BOOL;
    BT_Modify_ON : BOOL;
    BT_Combi_OK : BOOL;
    STN_SEL : UINT;
    Word_per_Stn : UINT;
    SET : BOOL;
    RST : BOOL;
END_VAR
VAR_IN_OUT
    HMI_Disp_DB : ARRAY[0..19] OF WORD;
    Modify_DB : ARRAY[0..19] OF WORD;
    CType_DB : ARRAY[0..999] OF WORD;
END_VAR
VAR_OUTPUT
    LP_CCR_On : BOOL;
    LP_Modify_On : BOOL;
END_VAR
VAR
    INDEX : INT;
    JMP : BOOL;
    NE : BOOL;
    RST_Delay : BOOL;
    SET_Delay : BOOL;
    STN_SEL_Temp : UINT;
    STN_SEL_Temp2 : UINT;
    T1 : TON;
    T2 : TON;
    Temp : WORD;
END_VAR
VAR
    _t1 : BOOL;
    _t2 : BOOL;
    _p3 : BOOL;
    _e4 : R_TRIG;
    _e5 : R_TRIG;
    _t6 : BOOL;
    _e7 : R_TRIG;
    _t8 : BOOL;
    _e9 : R_TRIG;
    _t10 : BOOL;
END_VAR

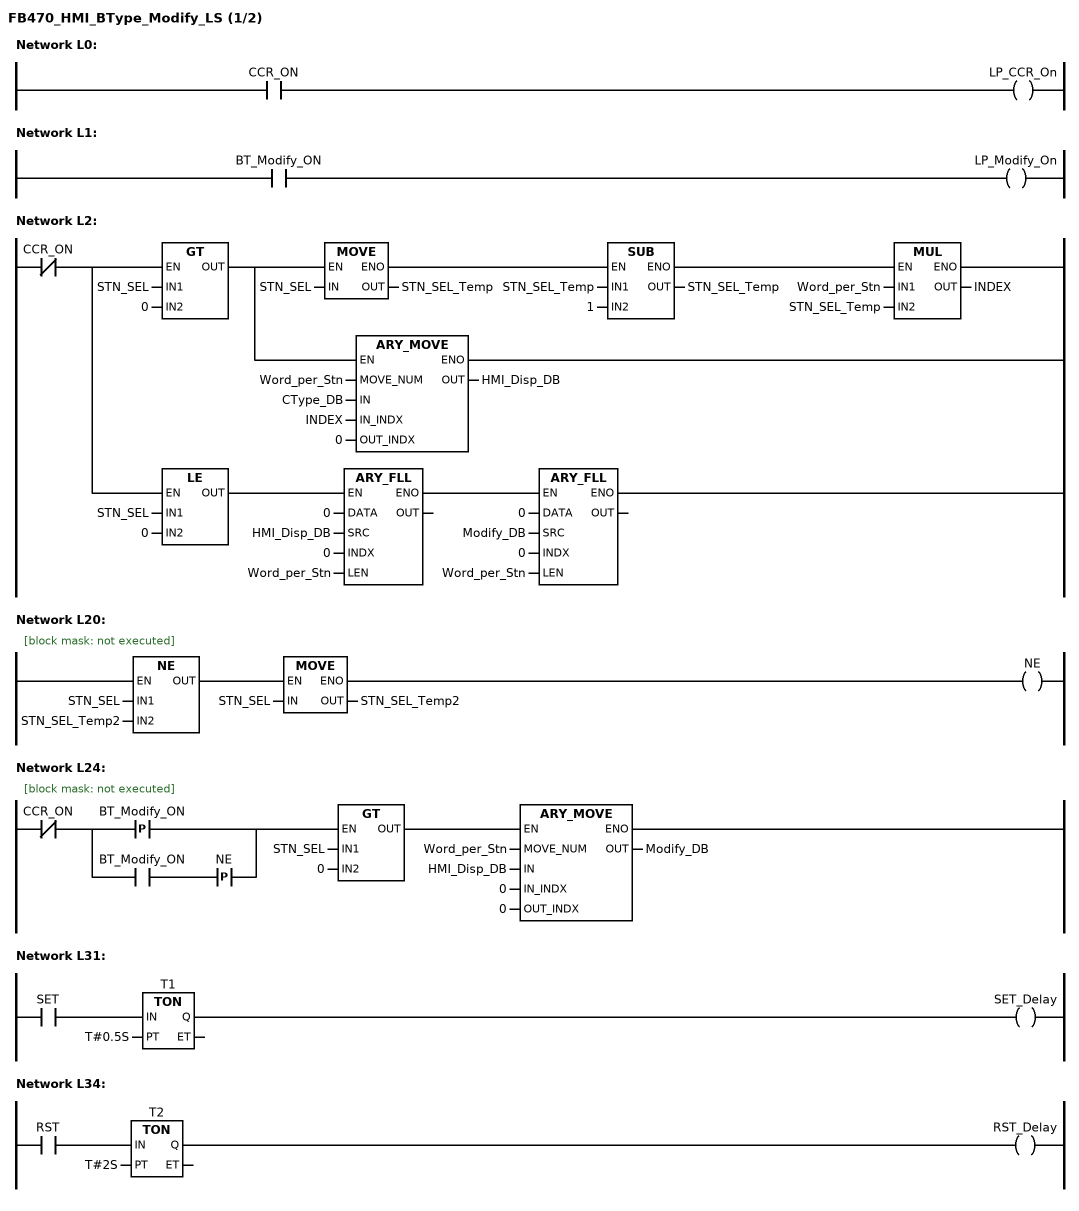
(* Rung L0 *)
LP_CCR_On := CCR_ON;
(* Rung L1 *)
LP_Modify_On := BT_Modify_ON;
(* Rung L2 *)
IF NOT CCR_ON THEN _t1 := STN_SEL > 0; END_IF;
IF _t1 THEN
    STN_SEL_Temp := STN_SEL;
    STN_SEL_Temp := STN_SEL_Temp - 1;
    INDEX := Word_per_Stn * STN_SEL_Temp;
    HMI_Disp_DB := ARY_MOVE(MOVE_NUM := Word_per_Stn, IN := CType_DB, IN_INDX := INDEX, OUT_INDX := 0);
END_IF;
IF NOT CCR_ON THEN _t2 := STN_SEL <= 0; END_IF;
IF _t2 THEN
    ARY_FLL(DATA := 0, SRC := HMI_Disp_DB, INDX := 0, LEN := Word_per_Stn);
    ARY_FLL(DATA := 0, SRC := Modify_DB, INDX := 0, LEN := Word_per_Stn);
END_IF;
(* Rung L20 is block-masked: not executed *)
// _p3 := STN_SEL <> STN_SEL_Temp2;
// IF _p3 THEN STN_SEL_Temp2 := STN_SEL; END_IF;
// NE := _p3;
(* Rung L24 is block-masked: not executed *)
// _e4(CLK := BT_Modify_ON);
// _e5(CLK := NE);
// IF NOT CCR_ON AND (_e4.Q OR (BT_Modify_ON AND _e5.Q)) THEN _t6 := STN_SEL > 0; END_IF;
// IF _t6 THEN
//     Modify_DB := ARY_MOVE(MOVE_NUM := Word_per_Stn, IN := HMI_Disp_DB, IN_INDX := 0, OUT_INDX := 0);
// END_IF;
(* Rung L31 *)
T1(IN := SET, PT := T#0.5S);
SET_Delay := T1.Q;
(* Rung L34 *)
T2(IN := RST, PT := T#2S);
RST_Delay := T2.Q;

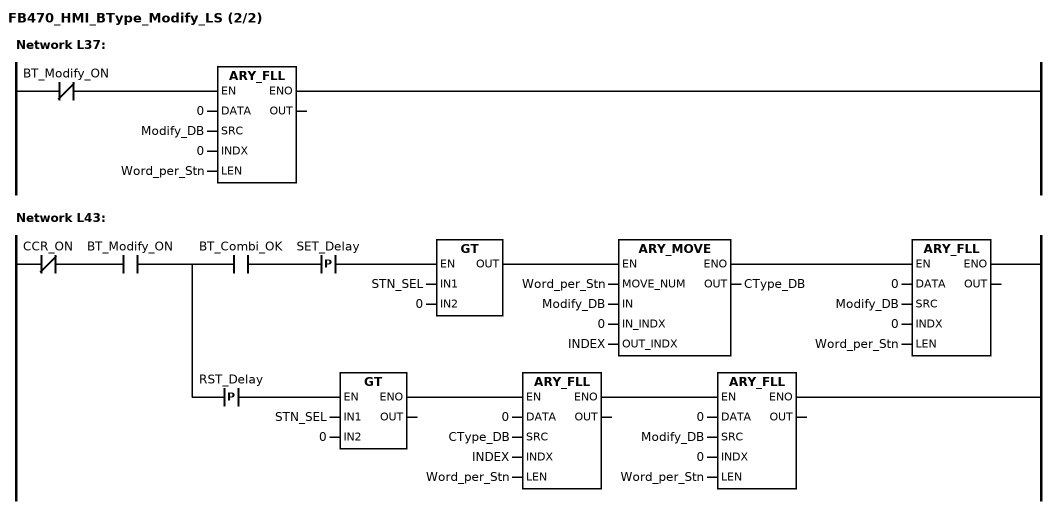
(* Rung L37 *)
IF NOT BT_Modify_ON THEN ARY_FLL(DATA := 0, SRC := Modify_DB, INDX := 0, LEN := Word_per_Stn); END_IF;
(* Rung L43 *)
_e7(CLK := SET_Delay);
IF NOT CCR_ON AND BT_Modify_ON AND BT_Combi_OK AND _e7.Q THEN _t8 := STN_SEL > 0; END_IF;
IF _t8 THEN
    CType_DB := ARY_MOVE(MOVE_NUM := Word_per_Stn, IN := Modify_DB, IN_INDX := 0, OUT_INDX := INDEX);
    ARY_FLL(DATA := 0, SRC := Modify_DB, INDX := 0, LEN := Word_per_Stn);
END_IF;
_e9(CLK := RST_Delay);
IF NOT CCR_ON AND BT_Modify_ON AND _e9.Q THEN
    _t10 := STN_SEL > 0;
    ARY_FLL(DATA := 0, SRC := CType_DB, INDX := INDEX, LEN := Word_per_Stn);
    ARY_FLL(DATA := 0, SRC := Modify_DB, INDX := 0, LEN := Word_per_Stn);
END_IF;
END_FUNCTION_BLOCK

FUNCTION_BLOCK FB494_Robot_Hyundai_HMMI_v1
VAR_INPUT
    IN_START_Add : ARRAY[0..3] OF WORD;
    RBT_Prog_No : INT;
    X_Ready_On : BOOL;
    M_Auto : BOOL;
    T_START : TIME;
    M_START_OK : BOOL;
    M_Prog_OK : BOOL;
    M_RESTART_OK : BOOL;
    M_Stn_Fault : BOOL;
    M_Error_Rst : BOOL;
    M_Cycle_Set : BOOL;
    M_LAST_WK_COMP_RST : BOOL;
    M_ATD_OK : BOOL;
    M_TIP_CHANGE_START : BOOL;
    M_TIP_CHANGE_COMPL : BOOL;
    M_WATER_CUT_OFF : BOOL;
    M_BUZZ_STOP_AUX : BOOL;
    M_PLT_COUNT_RST_AUX : BOOL;
    M_GATE_CLOSED : BOOL;
    M_EM_STOP : BOOL;
    M_VIP_MODE : BOOL;
    M_TEST : BOOL;
    M_A_In_Ok : BOOL;
    M_B_In_Ok : BOOL;
    M_C_In_Ok : BOOL;
    M_D_In_Ok : BOOL;
    M_E_In_Ok : BOOL;
    M_F_In_Ok : BOOL;
    M_G_In_Ok : BOOL;
    M_H_In_Ok : BOOL;
    M_2nd_In_Ok : BOOL;
    M_3rd_In_Ok : BOOL;
    M_4th_In_Ok : BOOL;
    M_5th_In_Ok : BOOL;
    M_6th_In_Ok : BOOL;
    M_7th_In_Ok : BOOL;
    M_1st_Comp_Rst : BOOL;
    M_2nd_Comp_Rst : BOOL;
    M_3rd_Comp_Rst : BOOL;
    M_4th_Comp_Rst : BOOL;
    M_5th_Comp_Rst : BOOL;
    M_6th_Comp_Rst : BOOL;
    M_7th_Comp_Rst : BOOL;
    Mutual_Int1 : BOOL;
    Mutual_Int2 : BOOL;
    Mutual_Int3 : BOOL;
    Mutual_Int4 : BOOL;
    Mutual_Int5 : BOOL;
    Mutual_Int6 : BOOL;
    Mutual_Int7 : BOOL;
    Mutual_Int8 : BOOL;
    M_PLT1_In_Ok : BOOL;
    M_PLT2_In_Ok : BOOL;
    M_PLT3_In_Ok : BOOL;
    M_PLT4_In_Ok : BOOL;
    M_PLT5_In_Ok : BOOL;
    M_PLT6_In_Ok : BOOL;
    M_PLT7_In_Ok : BOOL;
    M_PLT8_In_Ok : BOOL;
    M_PLT9_In_Ok : BOOL;
    M_PLT10_In_Ok : BOOL;
    M_PLT11_In_Ok : BOOL;
    M_PLT12_In_Ok : BOOL;
END_VAR
VAR_OUTPUT
    OUT_Start_Add : ARRAY[0..3] OF WORD;
    M_RBT_Ready : BOOL;
    M_RBT_Auto : BOOL;
    M_RBT_Fault : BOOL;
    M_RBT_Home : BOOL;
    M_RBT_EM_Stop : BOOL;
    M_RBT_PAUSE : BOOL;
    M_RBT_PROGRAM_ERR : BOOL;
    M_RBT_PLC_RUN_CHK_ERR : BOOL;
    M_Last_Comp : BOOL;
    M_1st_Comp : BOOL;
    M_2nd_Comp : BOOL;
    M_3rd_Comp : BOOL;
    M_4th_Comp : BOOL;
    M_5th_Comp : BOOL;
    M_6th_Comp : BOOL;
    M_7th_Comp : BOOL;
    M_NO_INTF1 : BOOL;
    M_NO_INTF2 : BOOL;
    M_NO_INTF3 : BOOL;
    M_NO_INTF4 : BOOL;
    M_NO_INTF5 : BOOL;
    M_NO_INTF6 : BOOL;
    M_NO_INTF7 : BOOL;
    M_NO_INTF8 : BOOL;
    M_NO_INTF9 : BOOL;
    M_NO_INTF10 : BOOL;
    M_NO_INTF11 : BOOL;
    M_NO_INTF12 : BOOL;
END_VAR
VAR
    EM_STOP_DELAY : TOF;
    GATE_CLOSED_DELAY : TOF;
    Home_Delay : TON;
    IN_Add : ARRAY[0..3] OF WORD;
    M_RBT_Home_Aux : BOOL;
    OUT_Add : ARRAY[0..3] OF WORD;
    RBT_PLC_RUN_CHK_TIMER1 : TON;
    RBT_PLC_RUN_CHK_TIMER2 : TON;
    RBT_PRG_ARR : WORD;
    RBT_PRG_ECHO : INT;
    RBT_PRG_ECHO_ARR : WORD;
    RBT_PRG_Match_Ok : BOOL;
    RBT_RESTART : BOOL;
    RBT_START_Aux : BOOL;
    RBT_Start_Delay : TON;
    RBT_START_Off_DT : BOOL;
    RBT_Work_Rst_Aux : BOOL;
    RBT_X00_Home : BOOL;
    RBT_X01_LAST_WK_COMP : BOOL;
    RBT_X02_TOTAL_ERR : BOOL;
    RBT_X03_Ready_ON : BOOL;
    RBT_X04_Auto : BOOL;
    RBT_X05_Running : BOOL;
    RBT_X06_ABNORMAL_SEL : BOOL;
    RBT_X07_Tip_Dressing : BOOL;
    RBT_X08_EM_STOP : BOOL;
    RBT_X09_1ST_WK_COMP : BOOL;
    RBT_X10_2ND_WK_COMP : BOOL;
    RBT_X11_3RD_WK_COMP : BOOL;
    RBT_X12_4TH_WK_COMP : BOOL;
    RBT_X13_5TH_WK_COMP : BOOL;
    RBT_X14_6TH_WK_COMP : BOOL;
    RBT_X15_7TH_WK_COMP : BOOL;
    RBT_X16_NON_INTF1 : BOOL;
    RBT_X17_NON_INTF2 : BOOL;
    RBT_X18_NON_INTF3 : BOOL;
    RBT_X19_NON_INTF4 : BOOL;
    RBT_X20_NON_INTF5 : BOOL;
    RBT_X21_NON_INTF6 : BOOL;
    RBT_X22_NON_INTF7 : BOOL;
    RBT_X23_NON_INTF8 : BOOL;
    RBT_X24_NON_INTF9 : BOOL;
    RBT_X25_NON_INTF10 : BOOL;
    RBT_X26_NON_INTF11 : BOOL;
    RBT_X27_NON_INTF12 : BOOL;
    RBT_X28_SP : BOOL;
    RBT_X29_SP : BOOL;
    RBT_X30_SP : BOOL;
    RBT_X31_SP : BOOL;
    RBT_X32_Prog_Echo1 : BOOL;
    RBT_X33_Prog_Echo2 : BOOL;
    RBT_X34_Prog_Echo4 : BOOL;
    RBT_X35_Prog_Echo8 : BOOL;
    RBT_X36_Prog_Echo16 : BOOL;
    RBT_X37_Prog_Echo32 : BOOL;
    RBT_X38_Prog_Echo64 : BOOL;
    RBT_X39_Prog_Echo128 : BOOL;
    RBT_X40_TC_ERR : BOOL;
    RBT_X41_AIR_ERR : BOOL;
    RBT_X42_WATER_ERR : BOOL;
    RBT_X43_LS_ERR : BOOL;
    RBT_X44_COMM_ERR : BOOL;
    RBT_X45_SEALER_ERR : BOOL;
    RBT_X46_VISION_ERR : BOOL;
    RBT_X47_WELD_COUNT_ERR : BOOL;
    RBT_X48_MUTUAL_INT1 : BOOL;
    RBT_X49_MUTUAL_INT2 : BOOL;
    RBT_X50_MUTUAL_INT3 : BOOL;
    RBT_X51_MUTUAL_INT4 : BOOL;
    RBT_X52_MUTUAL_INT5 : BOOL;
    RBT_X53_MUTUAL_INT6 : BOOL;
    RBT_X54_MUTUAL_INT7 : BOOL;
    RBT_X55_MUTUAL_INT8 : BOOL;
    RBT_X56_SP : BOOL;
    RBT_X57_SP : BOOL;
    RBT_X58_PLT_COUNT_RST_COMPL : BOOL;
    RBT_X59_PLT_UNLOAD_COMPL : BOOL;
    RBT_X60_PLT_LAST_UNLOAD_COMPL : BOOL;
    RBT_X61_TIP_CHANGE : BOOL;
    RBT_X62_FLICKER_COMM_CHK : BOOL;
    RBT_X63_MOTOR_MC_ON : BOOL;
    RBT_Y00_Prog_SEL1 : BOOL;
    RBT_Y01_Prog_SEL2 : BOOL;
    RBT_Y02_Prog_SEL4 : BOOL;
    RBT_Y03_Prog_SEL8 : BOOL;
    RBT_Y04_Prog_SEL16 : BOOL;
    RBT_Y05_Prog_SEL32 : BOOL;
    RBT_Y06_Prog_SEL64 : BOOL;
    RBT_Y07_Prog_SEL128 : BOOL;
    RBT_Y08_WK_COMP_RST : BOOL;
    RBT_Y09_START : BOOL;
    RBT_Y10_Error_Rst : BOOL;
    RBT_Y11_EXT_READY : BOOL;
    RBT_Y12_ATD_START : BOOL;
    RBT_Y13_Pause : BOOL;
    RBT_Y14_EACH_WORK_COMPL_RST : BOOL;
    RBT_Y15_WATER_CUT_OFF : BOOL;
    RBT_Y16_A_1ST_IN_Ok : BOOL;
    RBT_Y17_B_1ST_IN_Ok : BOOL;
    RBT_Y18_C_1ST_IN_Ok : BOOL;
    RBT_Y19_D_1ST_IN_Ok : BOOL;
    RBT_Y20_E_1ST_IN_Ok : BOOL;
    RBT_Y21_F_1ST_IN_Ok : BOOL;
    RBT_Y22_G_1ST_IN_Ok : BOOL;
    RBT_Y23_H_1ST_IN_Ok : BOOL;
    RBT_Y24_2ND_IN_OK : BOOL;
    RBT_Y25_3RD_IN_OK : BOOL;
    RBT_Y26_4TH_IN_OK : BOOL;
    RBT_Y27_5TH_IN_OK : BOOL;
    RBT_Y28_6TH_IN_OK : BOOL;
    RBT_Y29_7TH_IN_OK : BOOL;
    RBT_Y30_SP : BOOL;
    RBT_Y31_SP : BOOL;
    RBT_Y32_PLT1_IN_OK : BOOL;
    RBT_Y33_PLT2_IN_OK : BOOL;
    RBT_Y34_PLT3_IN_OK : BOOL;
    RBT_Y35_PLT4_IN_OK : BOOL;
    RBT_Y36_PLT5_IN_OK : BOOL;
    RBT_Y37_PLT6_IN_OK : BOOL;
    RBT_Y38_PLT7_IN_OK : BOOL;
    RBT_Y39_PLT8_IN_OK : BOOL;
    RBT_Y40_PLT9_IN_OK : BOOL;
    RBT_Y41_PLT10_IN_OK : BOOL;
    RBT_Y42_PLT11_IN_OK : BOOL;
    RBT_Y43_PLT12_IN_OK : BOOL;
    RBT_Y44_SP : BOOL;
    RBT_Y45_SP : BOOL;
    RBT_Y46_SP : BOOL;
    RBT_Y47_TEST : BOOL;
    RBT_Y48_MUTUAL_INT1 : BOOL;
    RBT_Y49_MUTUAL_INT2 : BOOL;
    RBT_Y50_MUTUAL_INT3 : BOOL;
    RBT_Y51_MUTUAL_INT4 : BOOL;
    RBT_Y52_MUTUAL_INT5 : BOOL;
    RBT_Y53_MUTUAL_INT6 : BOOL;
    RBT_Y54_MUTUAL_INT7 : BOOL;
    RBT_Y55_MUTUAL_INT8 : BOOL;
    RBT_Y56_TIP_CHANGE_START : BOOL;
    RBT_Y57_TIP_CHANGE_END : BOOL;
    RBT_Y58_PLT_COUNT_RST : BOOL;
    RBT_Y59_GATE_CLOSED : BOOL;
    RBT_Y60_EM_STOP : BOOL;
    RBT_Y61_BUZZ_STOP : BOOL;
    RBT_Y62_FLICKER_COMM_CHK : BOOL;
    RBT_Y63_VIP_MODE : BOOL;
    Start_off_Delay : TON;
END_VAR
VAR
    _t1 : BOOL;
    _t2 : BOOL;
    _t3 : BOOL;
    _t4 : BOOL;
    _t5 : BOOL;
    _t6 : BOOL;
    _t7 : BOOL;
    _t8 : BOOL;
END_VAR

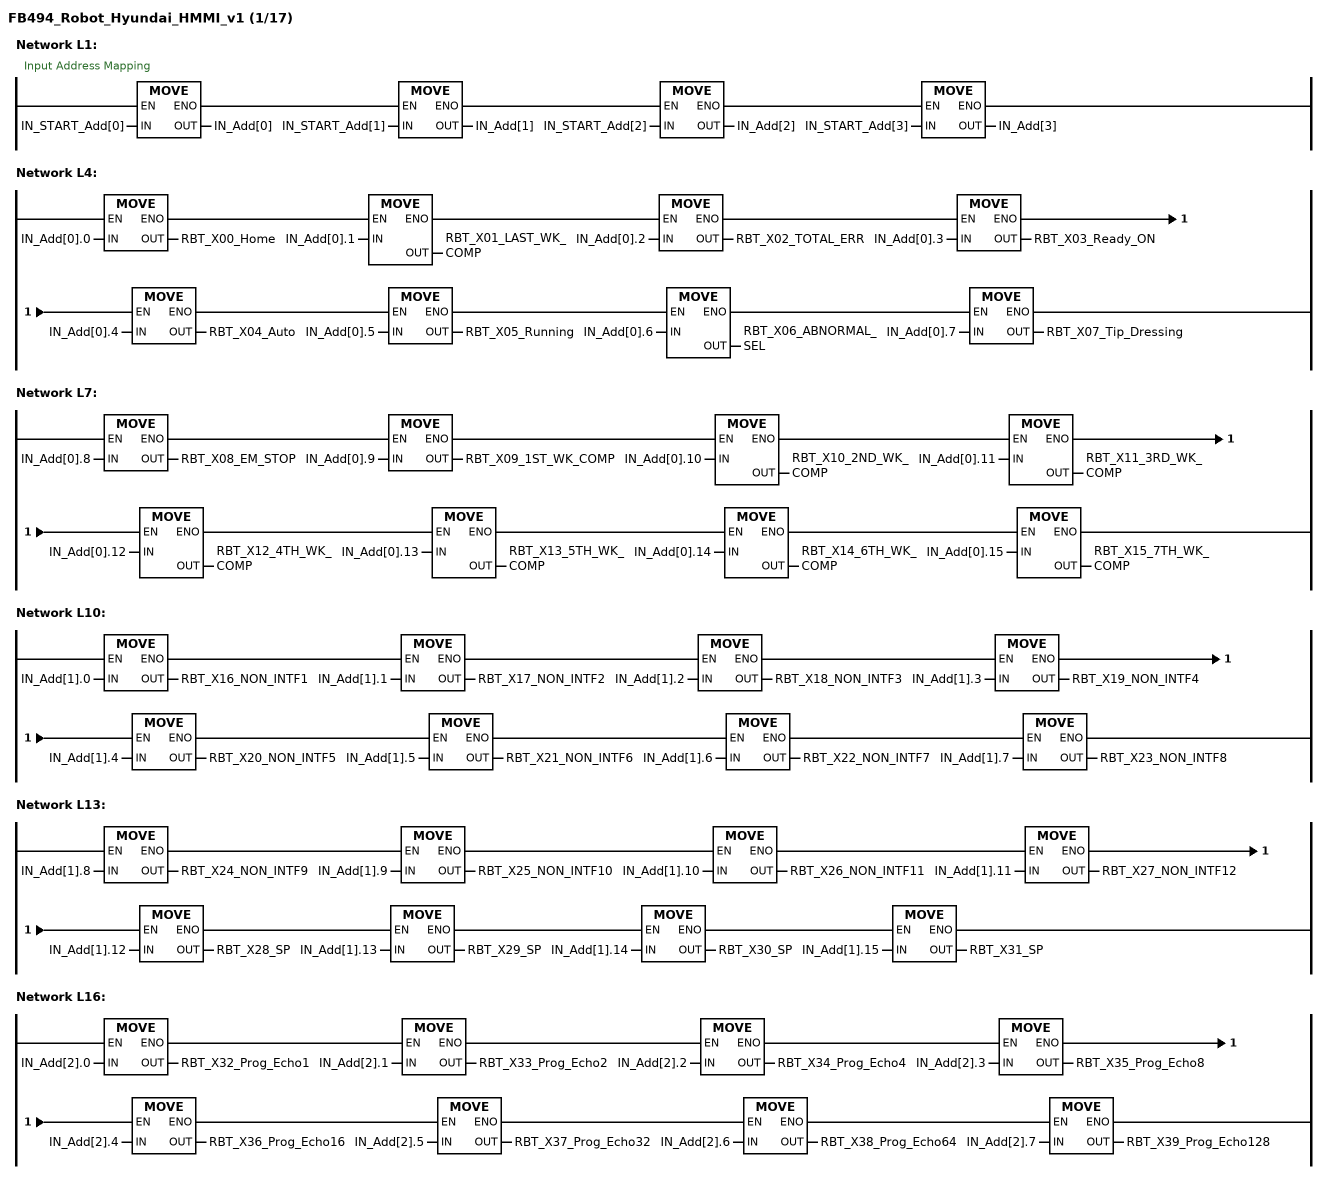
(* Input Address Mapping *)
(* Rung L1 *)
IN_Add[0] := IN_START_Add[0];
IN_Add[1] := IN_START_Add[1];
IN_Add[2] := IN_START_Add[2];
IN_Add[3] := IN_START_Add[3];
(* Rung L4 *)
RBT_X00_Home := IN_Add[0].0;
RBT_X01_LAST_WK_COMP := IN_Add[0].1;
RBT_X02_TOTAL_ERR := IN_Add[0].2;
RBT_X03_Ready_ON := IN_Add[0].3;
RBT_X04_Auto := IN_Add[0].4;
RBT_X05_Running := IN_Add[0].5;
RBT_X06_ABNORMAL_SEL := IN_Add[0].6;
RBT_X07_Tip_Dressing := IN_Add[0].7;
(* Rung L7 *)
RBT_X08_EM_STOP := IN_Add[0].8;
RBT_X09_1ST_WK_COMP := IN_Add[0].9;
RBT_X10_2ND_WK_COMP := IN_Add[0].10;
RBT_X11_3RD_WK_COMP := IN_Add[0].11;
RBT_X12_4TH_WK_COMP := IN_Add[0].12;
RBT_X13_5TH_WK_COMP := IN_Add[0].13;
RBT_X14_6TH_WK_COMP := IN_Add[0].14;
RBT_X15_7TH_WK_COMP := IN_Add[0].15;
(* Rung L10 *)
RBT_X16_NON_INTF1 := IN_Add[1].0;
RBT_X17_NON_INTF2 := IN_Add[1].1;
RBT_X18_NON_INTF3 := IN_Add[1].2;
RBT_X19_NON_INTF4 := IN_Add[1].3;
RBT_X20_NON_INTF5 := IN_Add[1].4;
RBT_X21_NON_INTF6 := IN_Add[1].5;
RBT_X22_NON_INTF7 := IN_Add[1].6;
RBT_X23_NON_INTF8 := IN_Add[1].7;
(* Rung L13 *)
RBT_X24_NON_INTF9 := IN_Add[1].8;
RBT_X25_NON_INTF10 := IN_Add[1].9;
RBT_X26_NON_INTF11 := IN_Add[1].10;
RBT_X27_NON_INTF12 := IN_Add[1].11;
RBT_X28_SP := IN_Add[1].12;
RBT_X29_SP := IN_Add[1].13;
RBT_X30_SP := IN_Add[1].14;
RBT_X31_SP := IN_Add[1].15;
(* Rung L16 *)
RBT_X32_Prog_Echo1 := IN_Add[2].0;
RBT_X33_Prog_Echo2 := IN_Add[2].1;
RBT_X34_Prog_Echo4 := IN_Add[2].2;
RBT_X35_Prog_Echo8 := IN_Add[2].3;
RBT_X36_Prog_Echo16 := IN_Add[2].4;
RBT_X37_Prog_Echo32 := IN_Add[2].5;
RBT_X38_Prog_Echo64 := IN_Add[2].6;
RBT_X39_Prog_Echo128 := IN_Add[2].7;

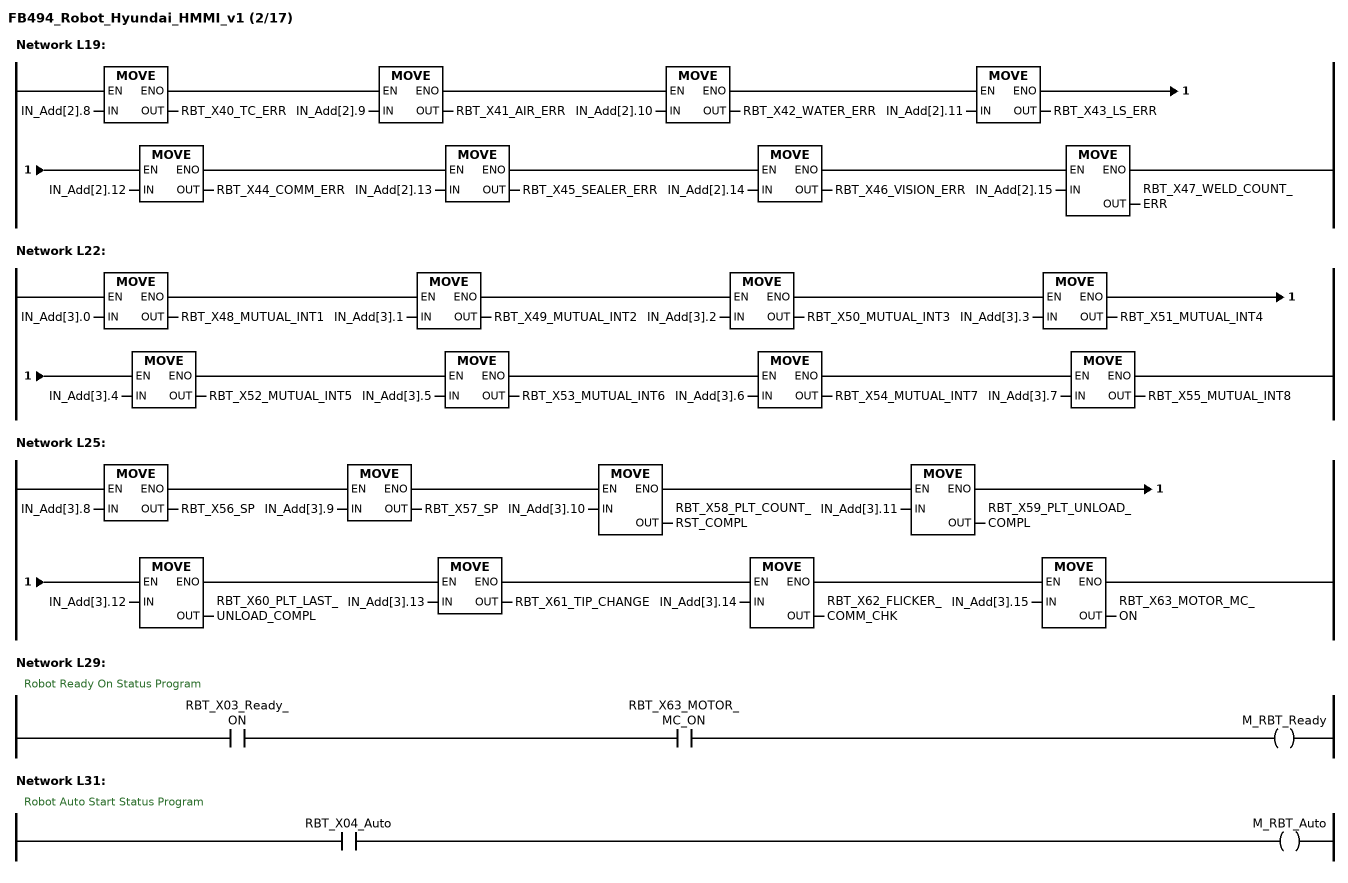
(* Rung L19 *)
RBT_X40_TC_ERR := IN_Add[2].8;
RBT_X41_AIR_ERR := IN_Add[2].9;
RBT_X42_WATER_ERR := IN_Add[2].10;
RBT_X43_LS_ERR := IN_Add[2].11;
RBT_X44_COMM_ERR := IN_Add[2].12;
RBT_X45_SEALER_ERR := IN_Add[2].13;
RBT_X46_VISION_ERR := IN_Add[2].14;
RBT_X47_WELD_COUNT_ERR := IN_Add[2].15;
(* Rung L22 *)
RBT_X48_MUTUAL_INT1 := IN_Add[3].0;
RBT_X49_MUTUAL_INT2 := IN_Add[3].1;
RBT_X50_MUTUAL_INT3 := IN_Add[3].2;
RBT_X51_MUTUAL_INT4 := IN_Add[3].3;
RBT_X52_MUTUAL_INT5 := IN_Add[3].4;
RBT_X53_MUTUAL_INT6 := IN_Add[3].5;
RBT_X54_MUTUAL_INT7 := IN_Add[3].6;
RBT_X55_MUTUAL_INT8 := IN_Add[3].7;
(* Rung L25 *)
RBT_X56_SP := IN_Add[3].8;
RBT_X57_SP := IN_Add[3].9;
RBT_X58_PLT_COUNT_RST_COMPL := IN_Add[3].10;
RBT_X59_PLT_UNLOAD_COMPL := IN_Add[3].11;
RBT_X60_PLT_LAST_UNLOAD_COMPL := IN_Add[3].12;
RBT_X61_TIP_CHANGE := IN_Add[3].13;
RBT_X62_FLICKER_COMM_CHK := IN_Add[3].14;
RBT_X63_MOTOR_MC_ON := IN_Add[3].15;
(* Robot Ready On Status Program *)
(* Rung L29 *)
M_RBT_Ready := RBT_X03_Ready_ON AND RBT_X63_MOTOR_MC_ON;
(* Robot Auto Start Status Program *)
(* Rung L31 *)
M_RBT_Auto := RBT_X04_Auto;

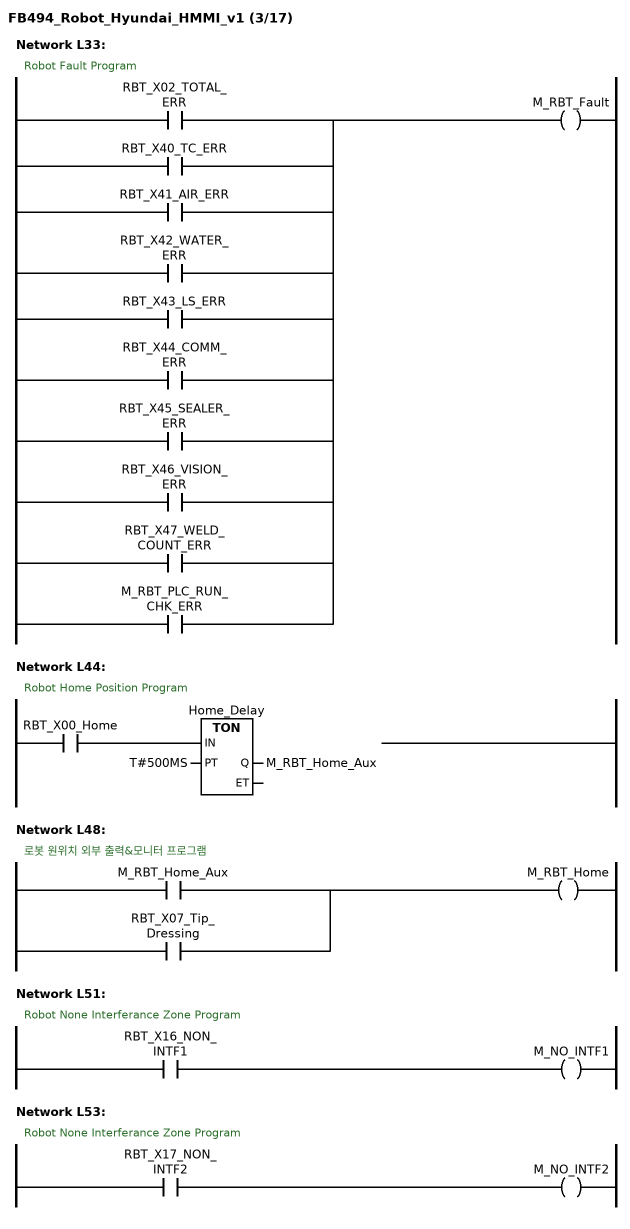
(* Robot Fault Program *)
(* Rung L33 *)
M_RBT_Fault := RBT_X02_TOTAL_ERR OR RBT_X40_TC_ERR OR RBT_X41_AIR_ERR OR RBT_X42_WATER_ERR OR RBT_X43_LS_ERR OR RBT_X44_COMM_ERR OR RBT_X45_SEALER_ERR OR RBT_X46_VISION_ERR OR RBT_X47_WELD_COUNT_ERR OR M_RBT_PLC_RUN_CHK_ERR;
(* Robot Home Position Program *)
(* Rung L44 *)
Home_Delay(IN := RBT_X00_Home, PT := T#500MS, Q => M_RBT_Home_Aux);
(* 로봇 원위치 외부 출력&모니터 프로그램 *)
(* Rung L48 *)
M_RBT_Home := M_RBT_Home_Aux OR RBT_X07_Tip_Dressing;
(* Robot None Interferance Zone Program *)
(* Rung L51 *)
M_NO_INTF1 := RBT_X16_NON_INTF1;
(* Robot None Interferance Zone Program *)
(* Rung L53 *)
M_NO_INTF2 := RBT_X17_NON_INTF2;

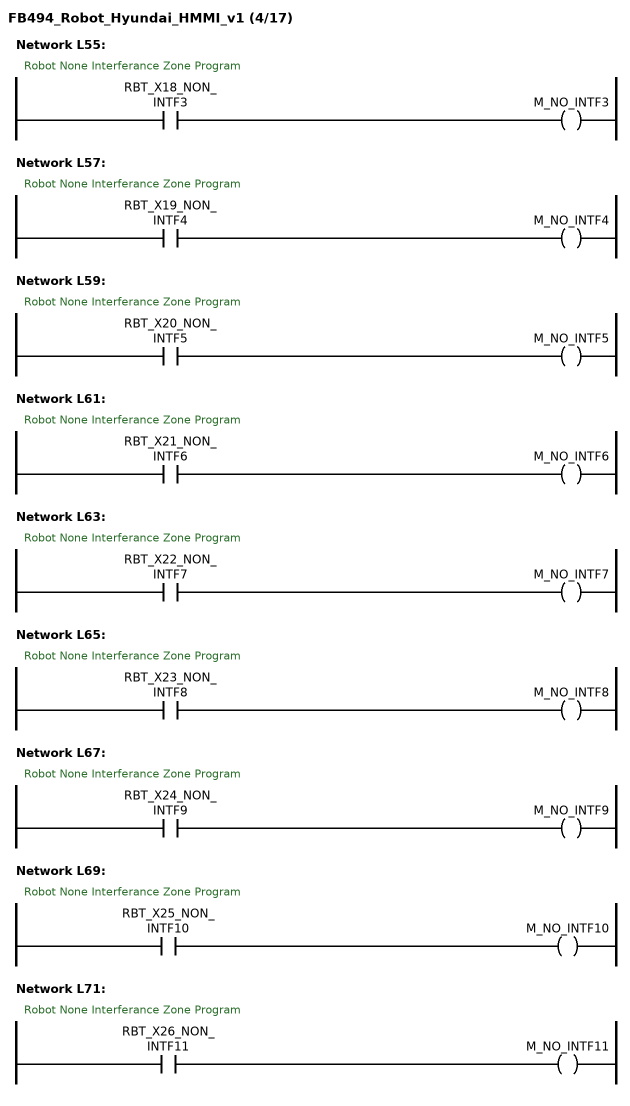
(* Robot None Interferance Zone Program *)
(* Rung L55 *)
M_NO_INTF3 := RBT_X18_NON_INTF3;
(* Robot None Interferance Zone Program *)
(* Rung L57 *)
M_NO_INTF4 := RBT_X19_NON_INTF4;
(* Robot None Interferance Zone Program *)
(* Rung L59 *)
M_NO_INTF5 := RBT_X20_NON_INTF5;
(* Robot None Interferance Zone Program *)
(* Rung L61 *)
M_NO_INTF6 := RBT_X21_NON_INTF6;
(* Robot None Interferance Zone Program *)
(* Rung L63 *)
M_NO_INTF7 := RBT_X22_NON_INTF7;
(* Robot None Interferance Zone Program *)
(* Rung L65 *)
M_NO_INTF8 := RBT_X23_NON_INTF8;
(* Robot None Interferance Zone Program *)
(* Rung L67 *)
M_NO_INTF9 := RBT_X24_NON_INTF9;
(* Robot None Interferance Zone Program *)
(* Rung L69 *)
M_NO_INTF10 := RBT_X25_NON_INTF10;
(* Robot None Interferance Zone Program *)
(* Rung L71 *)
M_NO_INTF11 := RBT_X26_NON_INTF11;

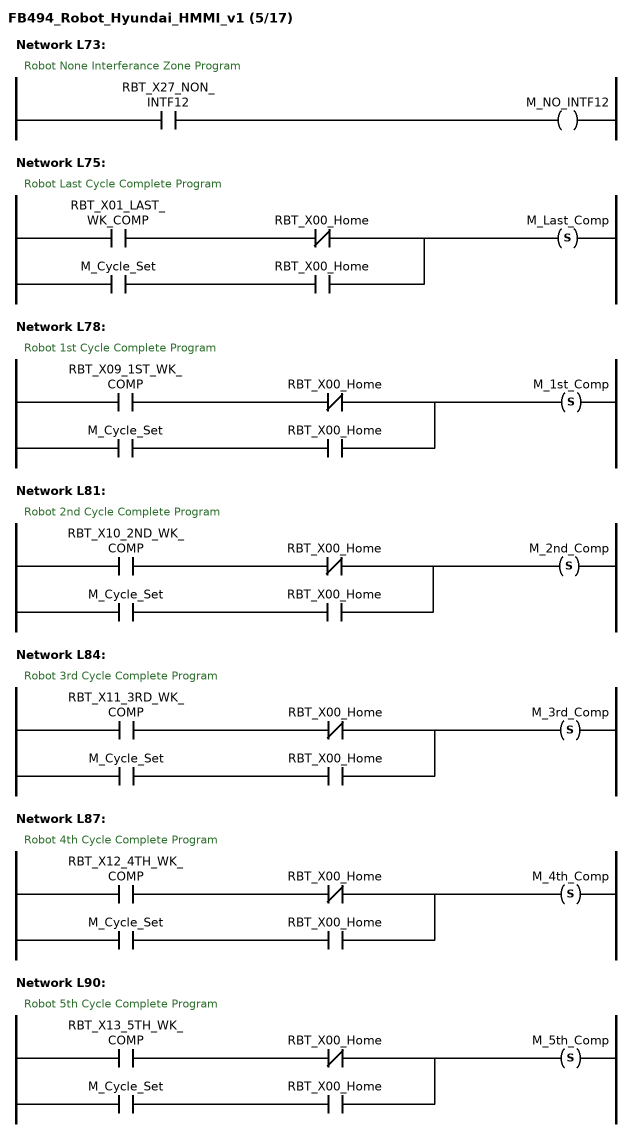
(* Robot None Interferance Zone Program *)
(* Rung L73 *)
M_NO_INTF12 := RBT_X27_NON_INTF12;
(* Robot Last Cycle Complete Program *)
(* Rung L75 *)
IF (RBT_X01_LAST_WK_COMP AND NOT RBT_X00_Home) OR (M_Cycle_Set AND RBT_X00_Home) THEN
    M_Last_Comp := TRUE;
END_IF;
(* Robot 1st Cycle Complete Program *)
(* Rung L78 *)
IF (RBT_X09_1ST_WK_COMP AND NOT RBT_X00_Home) OR (M_Cycle_Set AND RBT_X00_Home) THEN
    M_1st_Comp := TRUE;
END_IF;
(* Robot 2nd Cycle Complete Program *)
(* Rung L81 *)
IF (RBT_X10_2ND_WK_COMP AND NOT RBT_X00_Home) OR (M_Cycle_Set AND RBT_X00_Home) THEN
    M_2nd_Comp := TRUE;
END_IF;
(* Robot 3rd Cycle Complete Program *)
(* Rung L84 *)
IF (RBT_X11_3RD_WK_COMP AND NOT RBT_X00_Home) OR (M_Cycle_Set AND RBT_X00_Home) THEN
    M_3rd_Comp := TRUE;
END_IF;
(* Robot 4th Cycle Complete Program *)
(* Rung L87 *)
IF (RBT_X12_4TH_WK_COMP AND NOT RBT_X00_Home) OR (M_Cycle_Set AND RBT_X00_Home) THEN
    M_4th_Comp := TRUE;
END_IF;
(* Robot 5th Cycle Complete Program *)
(* Rung L90 *)
IF (RBT_X13_5TH_WK_COMP AND NOT RBT_X00_Home) OR (M_Cycle_Set AND RBT_X00_Home) THEN
    M_5th_Comp := TRUE;
END_IF;

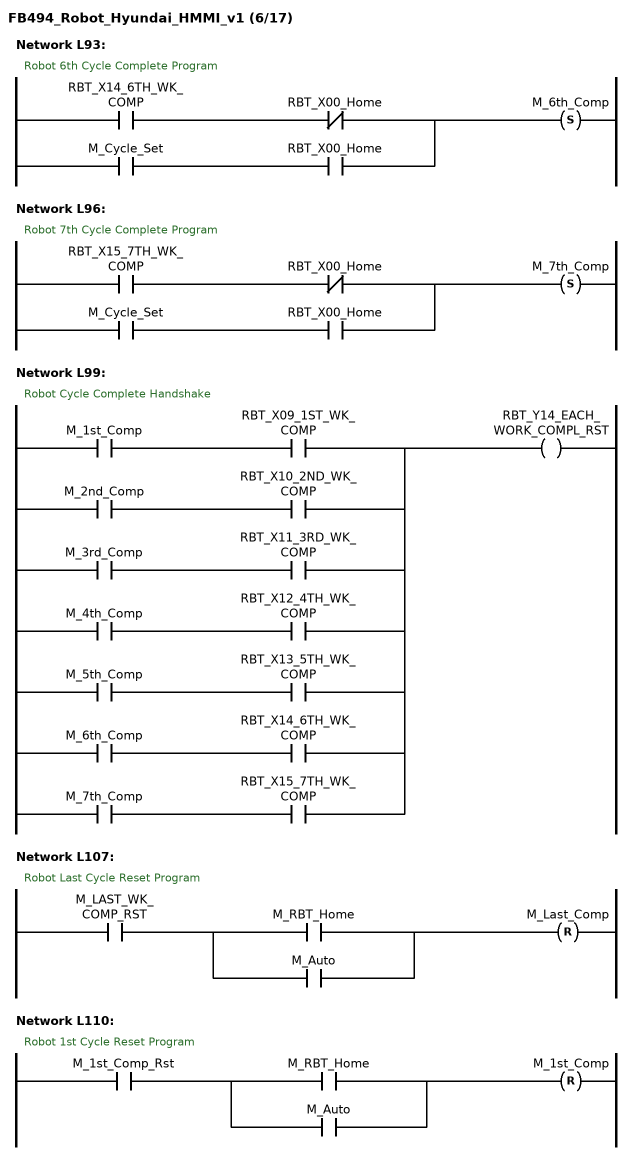
(* Robot 6th Cycle Complete Program *)
(* Rung L93 *)
IF (RBT_X14_6TH_WK_COMP AND NOT RBT_X00_Home) OR (M_Cycle_Set AND RBT_X00_Home) THEN
    M_6th_Comp := TRUE;
END_IF;
(* Robot 7th Cycle Complete Program *)
(* Rung L96 *)
IF (RBT_X15_7TH_WK_COMP AND NOT RBT_X00_Home) OR (M_Cycle_Set AND RBT_X00_Home) THEN
    M_7th_Comp := TRUE;
END_IF;
(* Robot Cycle Complete Handshake *)
(* Rung L99 *)
RBT_Y14_EACH_WORK_COMPL_RST := (M_1st_Comp AND RBT_X09_1ST_WK_COMP) OR (M_2nd_Comp AND RBT_X10_2ND_WK_COMP) OR (M_3rd_Comp AND RBT_X11_3RD_WK_COMP) OR (M_4th_Comp AND RBT_X12_4TH_WK_COMP) OR (M_5th_Comp AND RBT_X13_5TH_WK_COMP) OR (M_6th_Comp AND RBT_X14_6TH_WK_COMP) OR (M_7th_Comp AND RBT_X15_7TH_WK_COMP);
(* Robot Last Cycle Reset Program *)
(* Rung L107 *)
IF M_LAST_WK_COMP_RST AND (M_RBT_Home OR M_Auto) THEN M_Last_Comp := FALSE; END_IF;
(* Robot 1st Cycle Reset Program *)
(* Rung L110 *)
IF M_1st_Comp_Rst AND (M_RBT_Home OR M_Auto) THEN M_1st_Comp := FALSE; END_IF;

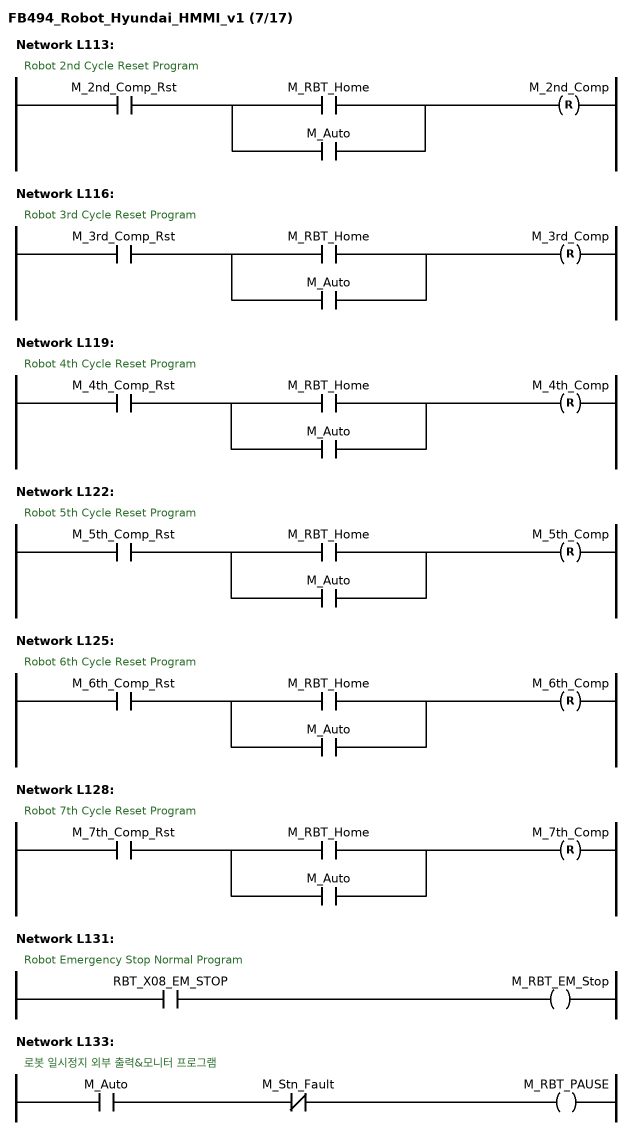
(* Robot 2nd Cycle Reset Program *)
(* Rung L113 *)
IF M_2nd_Comp_Rst AND (M_RBT_Home OR M_Auto) THEN M_2nd_Comp := FALSE; END_IF;
(* Robot 3rd Cycle Reset Program *)
(* Rung L116 *)
IF M_3rd_Comp_Rst AND (M_RBT_Home OR M_Auto) THEN M_3rd_Comp := FALSE; END_IF;
(* Robot 4th Cycle Reset Program *)
(* Rung L119 *)
IF M_4th_Comp_Rst AND (M_RBT_Home OR M_Auto) THEN M_4th_Comp := FALSE; END_IF;
(* Robot 5th Cycle Reset Program *)
(* Rung L122 *)
IF M_5th_Comp_Rst AND (M_RBT_Home OR M_Auto) THEN M_5th_Comp := FALSE; END_IF;
(* Robot 6th Cycle Reset Program *)
(* Rung L125 *)
IF M_6th_Comp_Rst AND (M_RBT_Home OR M_Auto) THEN M_6th_Comp := FALSE; END_IF;
(* Robot 7th Cycle Reset Program *)
(* Rung L128 *)
IF M_7th_Comp_Rst AND (M_RBT_Home OR M_Auto) THEN M_7th_Comp := FALSE; END_IF;
(* Robot Emergency Stop Normal Program *)
(* Rung L131 *)
M_RBT_EM_Stop := RBT_X08_EM_STOP;
(* 로봇 일시정지 외부 출력&모니터 프로그램 *)
(* Rung L133 *)
M_RBT_PAUSE := M_Auto AND NOT M_Stn_Fault;

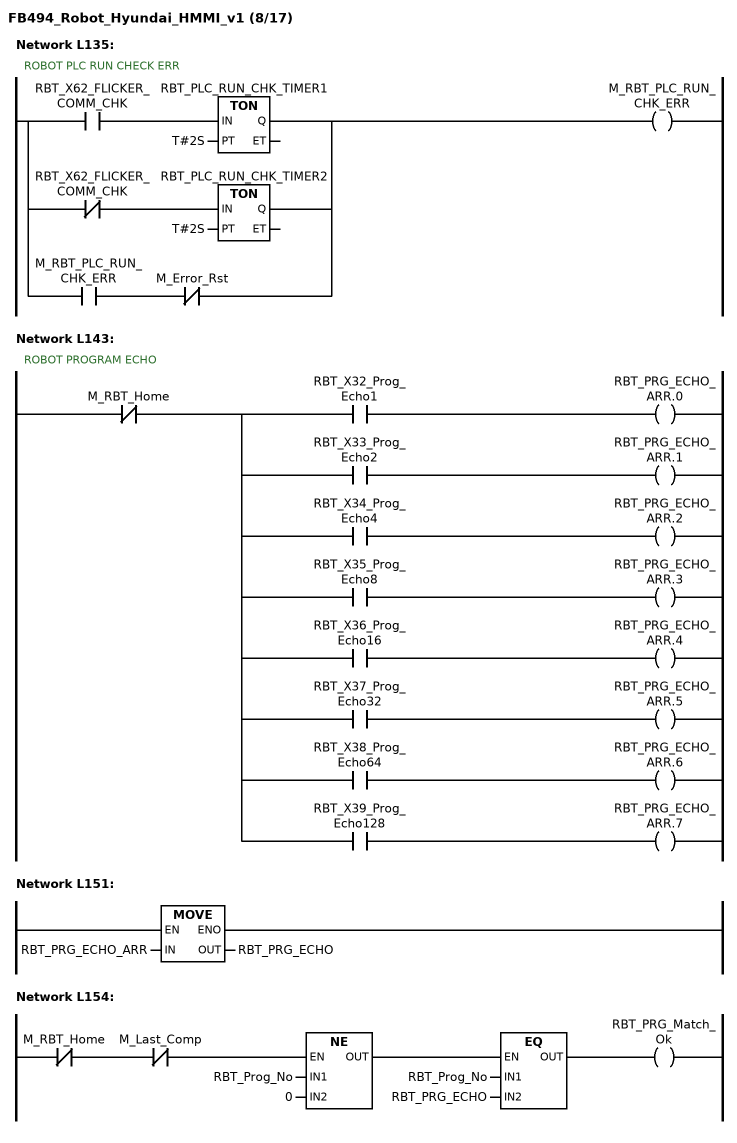
(* ROBOT PLC RUN CHECK ERR *)
(* Rung L135 *)
RBT_PLC_RUN_CHK_TIMER1(IN := RBT_X62_FLICKER_COMM_CHK, PT := T#2S);
RBT_PLC_RUN_CHK_TIMER2(IN := NOT RBT_X62_FLICKER_COMM_CHK, PT := T#2S);
M_RBT_PLC_RUN_CHK_ERR := RBT_PLC_RUN_CHK_TIMER1.Q OR RBT_PLC_RUN_CHK_TIMER2.Q OR (M_RBT_PLC_RUN_CHK_ERR AND NOT M_Error_Rst);
(* ROBOT PROGRAM ECHO *)
(* Rung L143 *)
RBT_PRG_ECHO_ARR.0 := NOT M_RBT_Home AND RBT_X32_Prog_Echo1;
RBT_PRG_ECHO_ARR.1 := NOT M_RBT_Home AND RBT_X33_Prog_Echo2;
RBT_PRG_ECHO_ARR.2 := NOT M_RBT_Home AND RBT_X34_Prog_Echo4;
RBT_PRG_ECHO_ARR.3 := NOT M_RBT_Home AND RBT_X35_Prog_Echo8;
RBT_PRG_ECHO_ARR.4 := NOT M_RBT_Home AND RBT_X36_Prog_Echo16;
RBT_PRG_ECHO_ARR.5 := NOT M_RBT_Home AND RBT_X37_Prog_Echo32;
RBT_PRG_ECHO_ARR.6 := NOT M_RBT_Home AND RBT_X38_Prog_Echo64;
RBT_PRG_ECHO_ARR.7 := NOT M_RBT_Home AND RBT_X39_Prog_Echo128;
(* Rung L151 *)
RBT_PRG_ECHO := RBT_PRG_ECHO_ARR;
(* Rung L154 *)
IF NOT M_RBT_Home AND NOT M_Last_Comp THEN _t1 := RBT_Prog_No <> 0; END_IF;
IF _t1 THEN _t2 := RBT_Prog_No = RBT_PRG_ECHO; END_IF;
RBT_PRG_Match_Ok := _t2;

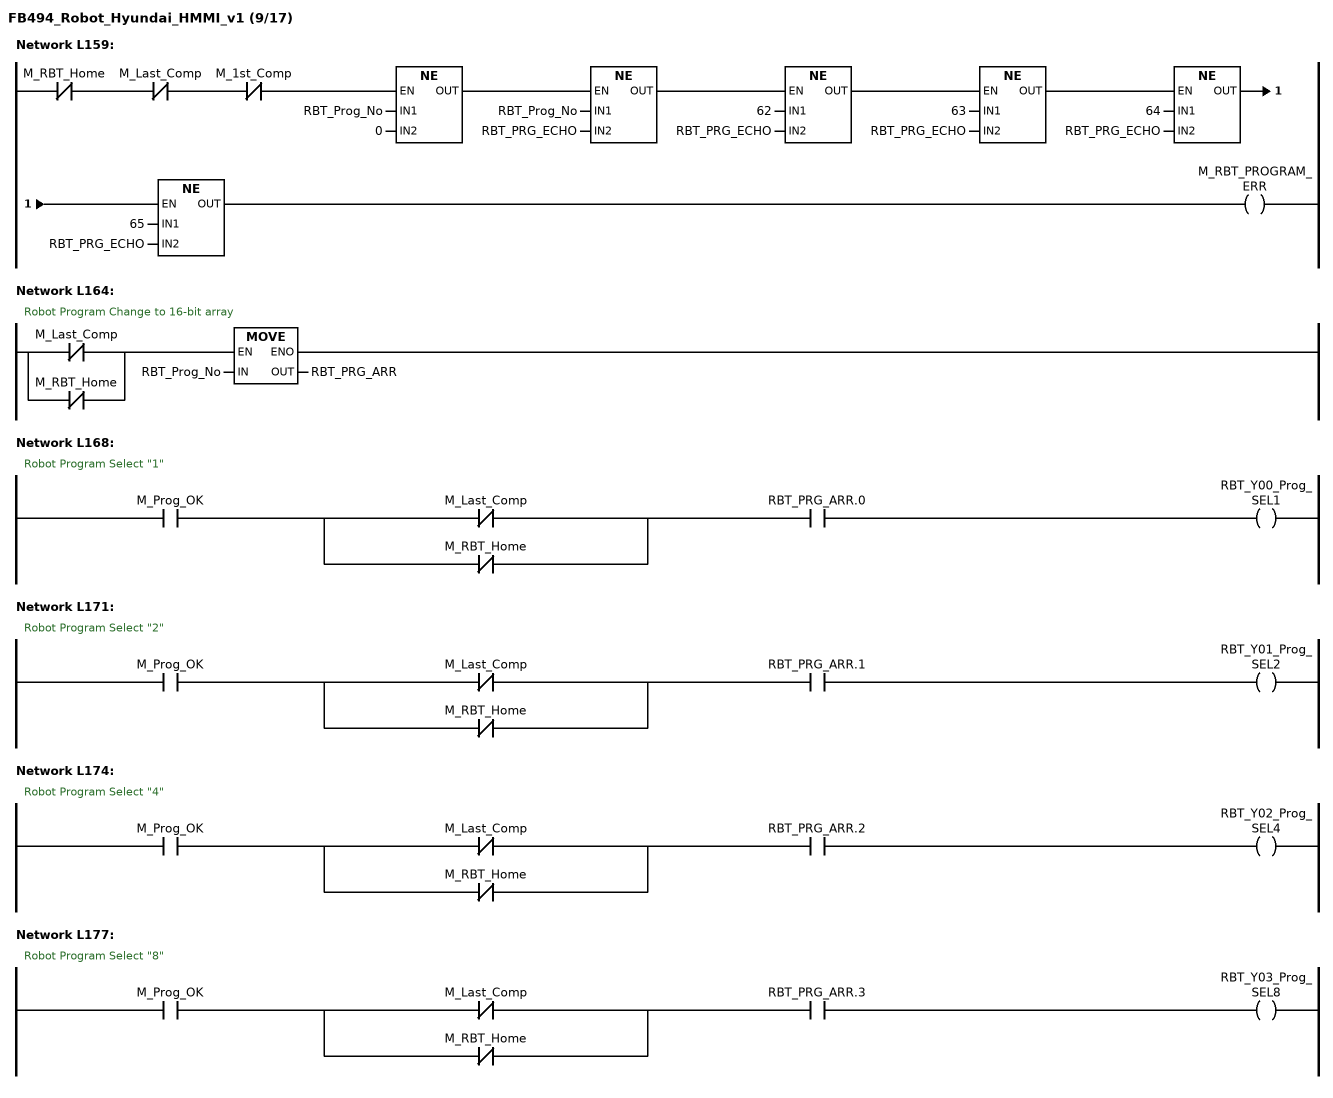
(* Rung L159 *)
IF NOT M_RBT_Home AND NOT M_Last_Comp AND NOT M_1st_Comp THEN _t3 := RBT_Prog_No <> 0; END_IF;
IF _t3 THEN _t4 := RBT_Prog_No <> RBT_PRG_ECHO; END_IF;
IF _t4 THEN _t5 := 62 <> RBT_PRG_ECHO; END_IF;
IF _t5 THEN _t6 := 63 <> RBT_PRG_ECHO; END_IF;
IF _t6 THEN _t7 := 64 <> RBT_PRG_ECHO; END_IF;
IF _t7 THEN _t8 := 65 <> RBT_PRG_ECHO; END_IF;
M_RBT_PROGRAM_ERR := _t8;
(* Robot Program Change to 16-bit array *)
(* Rung L164 *)
IF NOT M_Last_Comp OR NOT M_RBT_Home THEN RBT_PRG_ARR := RBT_Prog_No; END_IF;
(* Robot Program Select "1" *)
(* Rung L168 *)
RBT_Y00_Prog_SEL1 := M_Prog_OK AND (NOT M_Last_Comp OR NOT M_RBT_Home) AND RBT_PRG_ARR.0;
(* Robot Program Select "2" *)
(* Rung L171 *)
RBT_Y01_Prog_SEL2 := M_Prog_OK AND (NOT M_Last_Comp OR NOT M_RBT_Home) AND RBT_PRG_ARR.1;
(* Robot Program Select "4" *)
(* Rung L174 *)
RBT_Y02_Prog_SEL4 := M_Prog_OK AND (NOT M_Last_Comp OR NOT M_RBT_Home) AND RBT_PRG_ARR.2;
(* Robot Program Select "8" *)
(* Rung L177 *)
RBT_Y03_Prog_SEL8 := M_Prog_OK AND (NOT M_Last_Comp OR NOT M_RBT_Home) AND RBT_PRG_ARR.3;

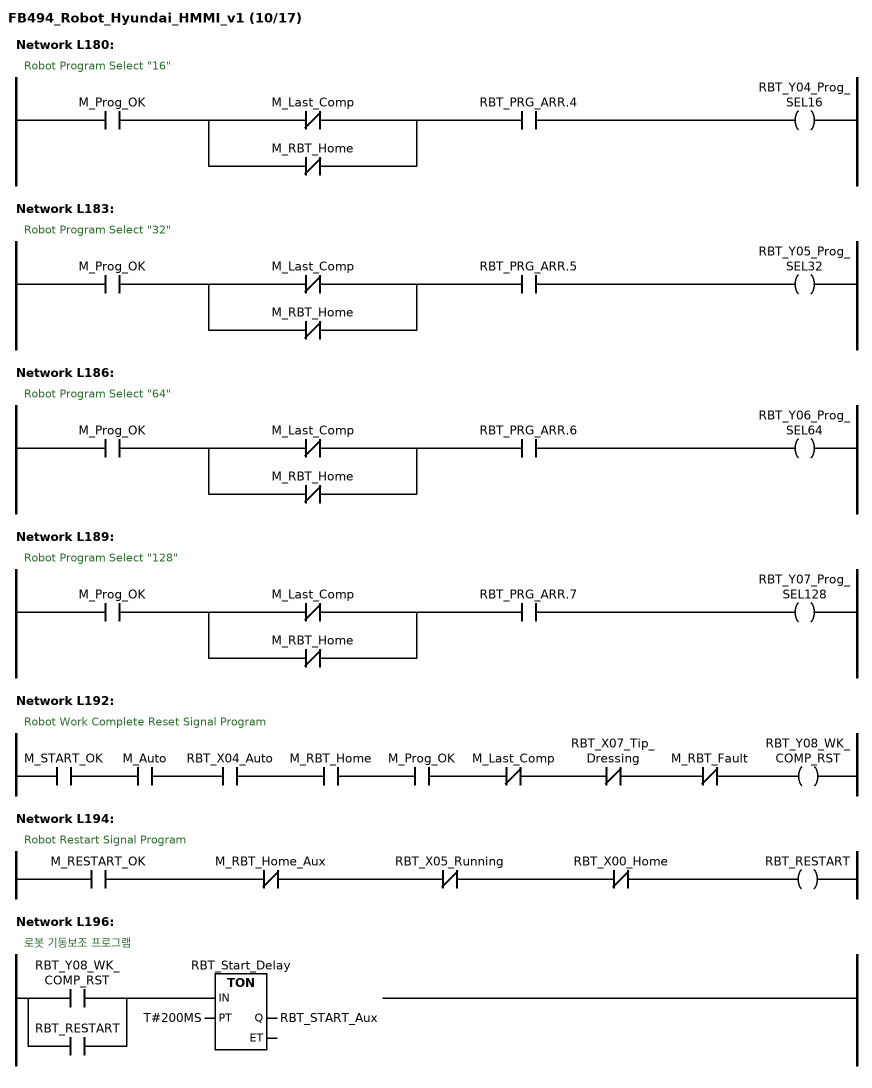
(* Robot Program Select "16" *)
(* Rung L180 *)
RBT_Y04_Prog_SEL16 := M_Prog_OK AND (NOT M_Last_Comp OR NOT M_RBT_Home) AND RBT_PRG_ARR.4;
(* Robot Program Select "32" *)
(* Rung L183 *)
RBT_Y05_Prog_SEL32 := M_Prog_OK AND (NOT M_Last_Comp OR NOT M_RBT_Home) AND RBT_PRG_ARR.5;
(* Robot Program Select "64" *)
(* Rung L186 *)
RBT_Y06_Prog_SEL64 := M_Prog_OK AND (NOT M_Last_Comp OR NOT M_RBT_Home) AND RBT_PRG_ARR.6;
(* Robot Program Select "128" *)
(* Rung L189 *)
RBT_Y07_Prog_SEL128 := M_Prog_OK AND (NOT M_Last_Comp OR NOT M_RBT_Home) AND RBT_PRG_ARR.7;
(* Robot Work Complete Reset Signal Program *)
(* Rung L192 *)
RBT_Y08_WK_COMP_RST := M_START_OK AND M_Auto AND RBT_X04_Auto AND M_RBT_Home AND M_Prog_OK AND NOT M_Last_Comp AND NOT RBT_X07_Tip_Dressing AND NOT M_RBT_Fault;
(* Robot Restart Signal Program *)
(* Rung L194 *)
RBT_RESTART := M_RESTART_OK AND NOT M_RBT_Home_Aux AND NOT RBT_X05_Running AND NOT RBT_X00_Home;
(* 로봇 기동보조 프로그램 *)
(* Rung L196 *)
RBT_Start_Delay(IN := RBT_Y08_WK_COMP_RST OR RBT_RESTART, PT := T#200MS, Q => RBT_START_Aux);

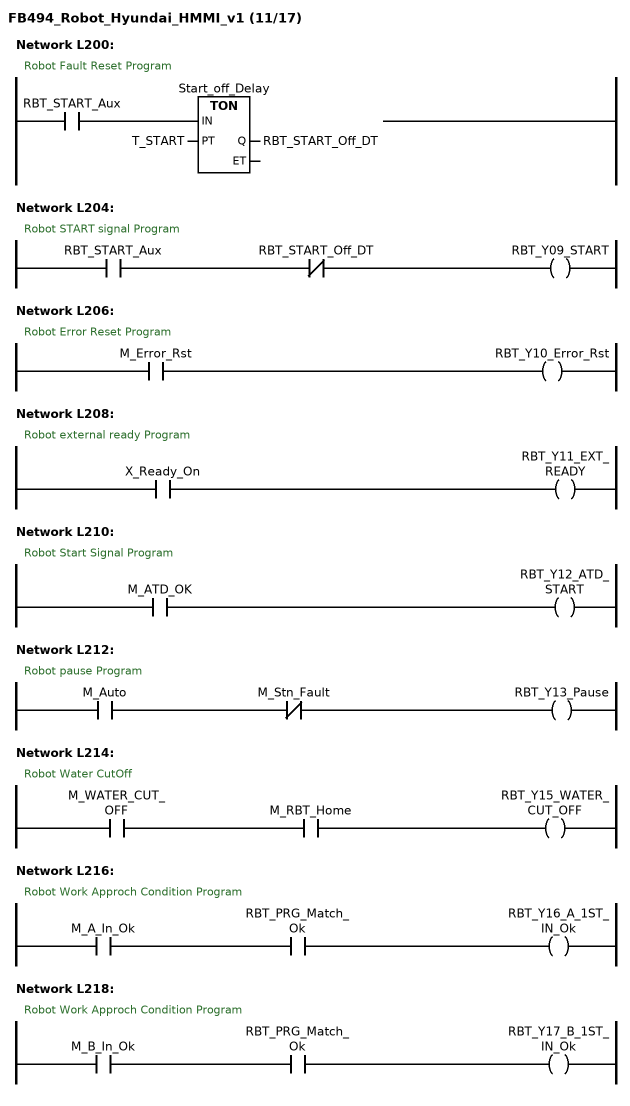
(* Robot Fault Reset Program *)
(* Rung L200 *)
Start_off_Delay(IN := RBT_START_Aux, PT := T_START, Q => RBT_START_Off_DT);
(* Robot START signal Program *)
(* Rung L204 *)
RBT_Y09_START := RBT_START_Aux AND NOT RBT_START_Off_DT;
(* Robot Error Reset Program *)
(* Rung L206 *)
RBT_Y10_Error_Rst := M_Error_Rst;
(* Robot external ready Program *)
(* Rung L208 *)
RBT_Y11_EXT_READY := X_Ready_On;
(* Robot Start Signal Program *)
(* Rung L210 *)
RBT_Y12_ATD_START := M_ATD_OK;
(* Robot pause Program *)
(* Rung L212 *)
RBT_Y13_Pause := M_Auto AND NOT M_Stn_Fault;
(* Robot Water CutOff *)
(* Rung L214 *)
RBT_Y15_WATER_CUT_OFF := M_WATER_CUT_OFF AND M_RBT_Home;
(* Robot Work Approch Condition Program *)
(* Rung L216 *)
RBT_Y16_A_1ST_IN_Ok := M_A_In_Ok AND RBT_PRG_Match_Ok;
(* Robot Work Approch Condition Program *)
(* Rung L218 *)
RBT_Y17_B_1ST_IN_Ok := M_B_In_Ok AND RBT_PRG_Match_Ok;

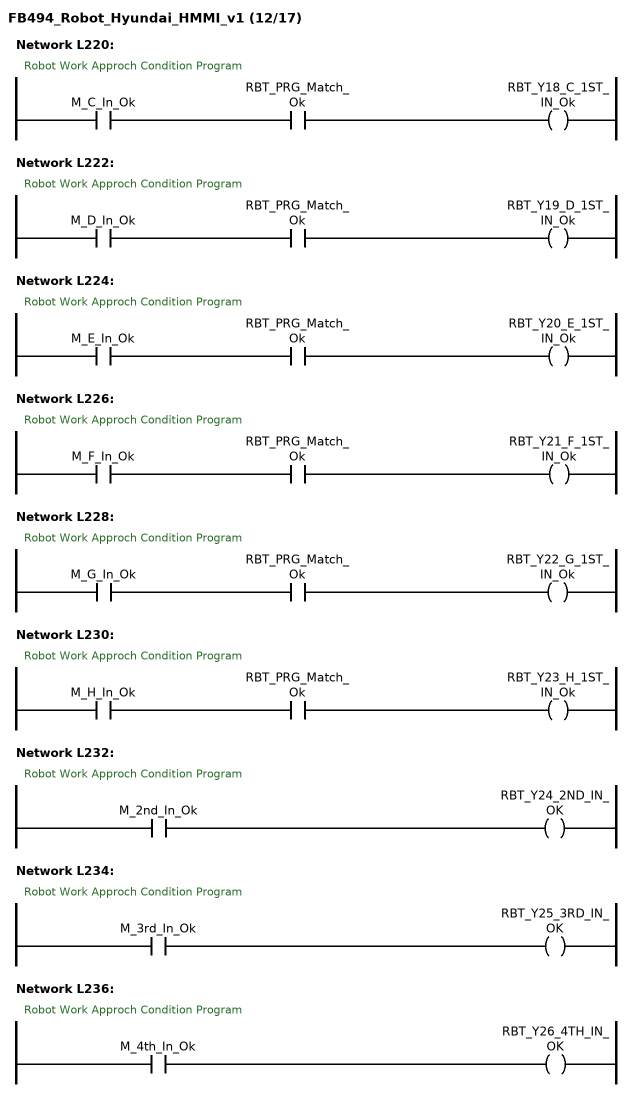
(* Robot Work Approch Condition Program *)
(* Rung L220 *)
RBT_Y18_C_1ST_IN_Ok := M_C_In_Ok AND RBT_PRG_Match_Ok;
(* Robot Work Approch Condition Program *)
(* Rung L222 *)
RBT_Y19_D_1ST_IN_Ok := M_D_In_Ok AND RBT_PRG_Match_Ok;
(* Robot Work Approch Condition Program *)
(* Rung L224 *)
RBT_Y20_E_1ST_IN_Ok := M_E_In_Ok AND RBT_PRG_Match_Ok;
(* Robot Work Approch Condition Program *)
(* Rung L226 *)
RBT_Y21_F_1ST_IN_Ok := M_F_In_Ok AND RBT_PRG_Match_Ok;
(* Robot Work Approch Condition Program *)
(* Rung L228 *)
RBT_Y22_G_1ST_IN_Ok := M_G_In_Ok AND RBT_PRG_Match_Ok;
(* Robot Work Approch Condition Program *)
(* Rung L230 *)
RBT_Y23_H_1ST_IN_Ok := M_H_In_Ok AND RBT_PRG_Match_Ok;
(* Robot Work Approch Condition Program *)
(* Rung L232 *)
RBT_Y24_2ND_IN_OK := M_2nd_In_Ok;
(* Robot Work Approch Condition Program *)
(* Rung L234 *)
RBT_Y25_3RD_IN_OK := M_3rd_In_Ok;
(* Robot Work Approch Condition Program *)
(* Rung L236 *)
RBT_Y26_4TH_IN_OK := M_4th_In_Ok;

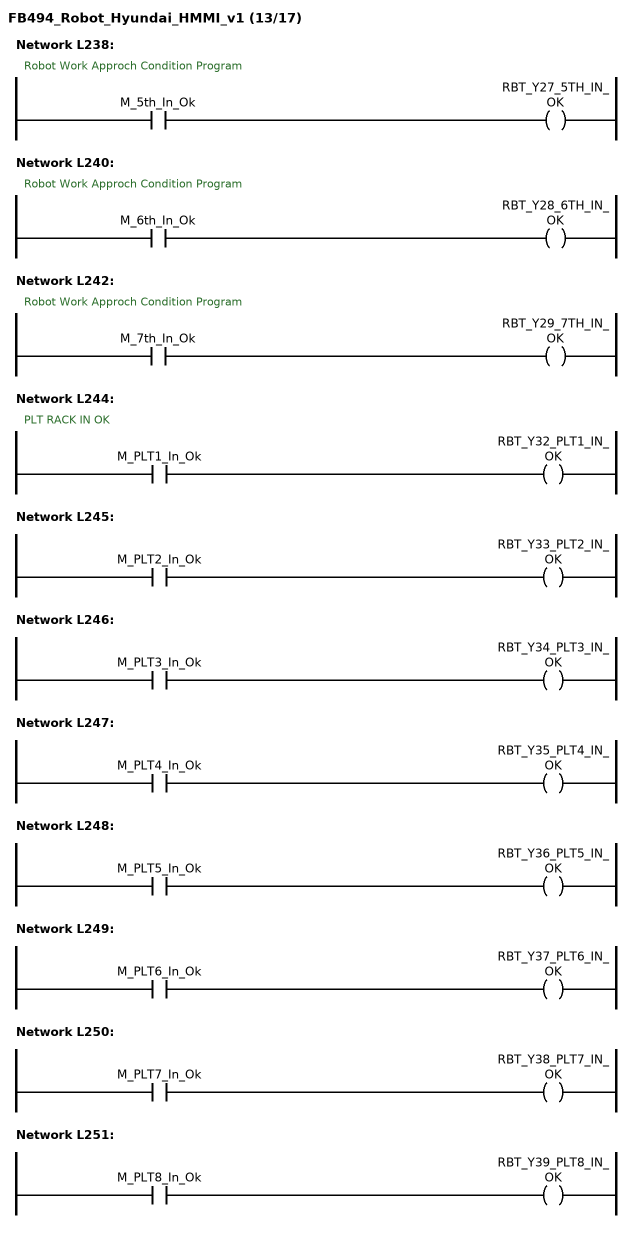
(* Robot Work Approch Condition Program *)
(* Rung L238 *)
RBT_Y27_5TH_IN_OK := M_5th_In_Ok;
(* Robot Work Approch Condition Program *)
(* Rung L240 *)
RBT_Y28_6TH_IN_OK := M_6th_In_Ok;
(* Robot Work Approch Condition Program *)
(* Rung L242 *)
RBT_Y29_7TH_IN_OK := M_7th_In_Ok;
(* PLT RACK IN OK *)
(* Rung L244 *)
RBT_Y32_PLT1_IN_OK := M_PLT1_In_Ok;
(* Rung L245 *)
RBT_Y33_PLT2_IN_OK := M_PLT2_In_Ok;
(* Rung L246 *)
RBT_Y34_PLT3_IN_OK := M_PLT3_In_Ok;
(* Rung L247 *)
RBT_Y35_PLT4_IN_OK := M_PLT4_In_Ok;
(* Rung L248 *)
RBT_Y36_PLT5_IN_OK := M_PLT5_In_Ok;
(* Rung L249 *)
RBT_Y37_PLT6_IN_OK := M_PLT6_In_Ok;
(* Rung L250 *)
RBT_Y38_PLT7_IN_OK := M_PLT7_In_Ok;
(* Rung L251 *)
RBT_Y39_PLT8_IN_OK := M_PLT8_In_Ok;

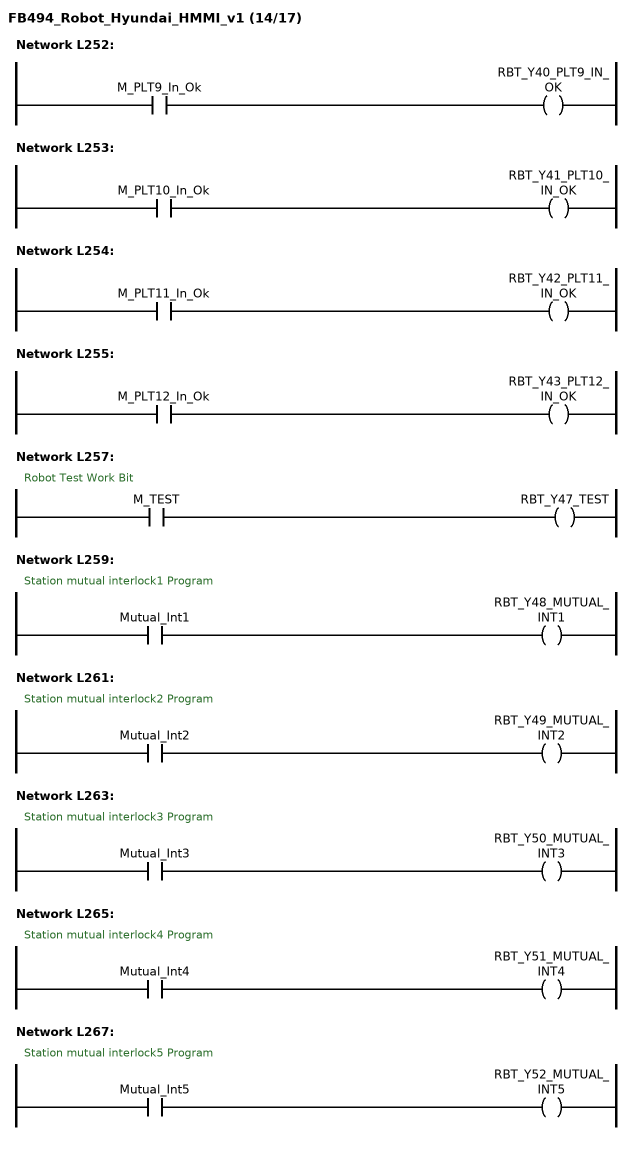
(* Rung L252 *)
RBT_Y40_PLT9_IN_OK := M_PLT9_In_Ok;
(* Rung L253 *)
RBT_Y41_PLT10_IN_OK := M_PLT10_In_Ok;
(* Rung L254 *)
RBT_Y42_PLT11_IN_OK := M_PLT11_In_Ok;
(* Rung L255 *)
RBT_Y43_PLT12_IN_OK := M_PLT12_In_Ok;
(* Robot Test Work Bit *)
(* Rung L257 *)
RBT_Y47_TEST := M_TEST;
(* Station mutual interlock1 Program *)
(* Rung L259 *)
RBT_Y48_MUTUAL_INT1 := Mutual_Int1;
(* Station mutual interlock2 Program *)
(* Rung L261 *)
RBT_Y49_MUTUAL_INT2 := Mutual_Int2;
(* Station mutual interlock3 Program *)
(* Rung L263 *)
RBT_Y50_MUTUAL_INT3 := Mutual_Int3;
(* Station mutual interlock4 Program *)
(* Rung L265 *)
RBT_Y51_MUTUAL_INT4 := Mutual_Int4;
(* Station mutual interlock5 Program *)
(* Rung L267 *)
RBT_Y52_MUTUAL_INT5 := Mutual_Int5;

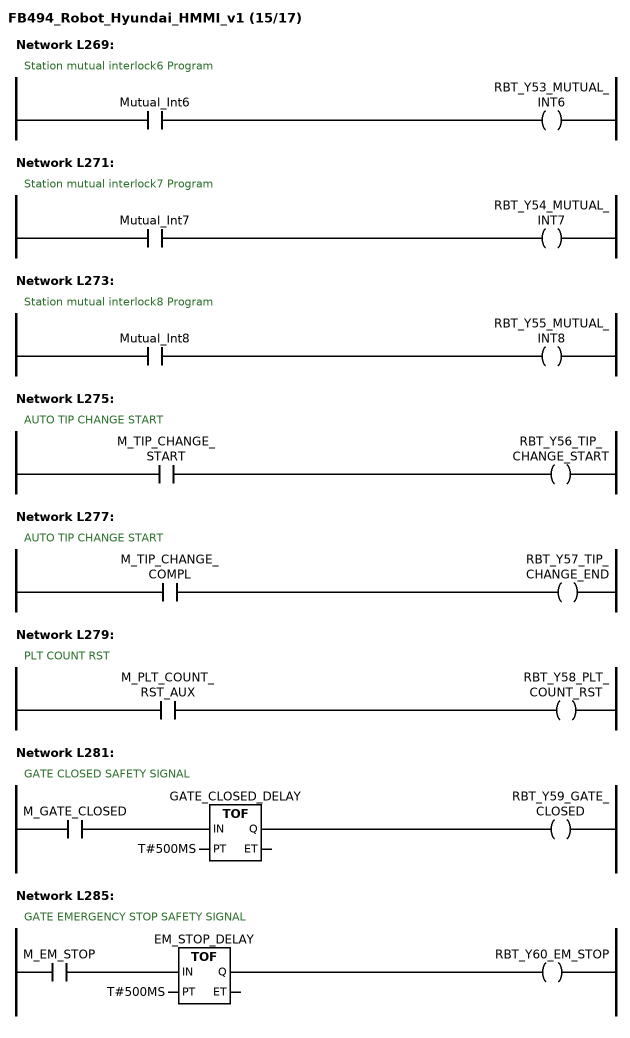
(* Station mutual interlock6 Program *)
(* Rung L269 *)
RBT_Y53_MUTUAL_INT6 := Mutual_Int6;
(* Station mutual interlock7 Program *)
(* Rung L271 *)
RBT_Y54_MUTUAL_INT7 := Mutual_Int7;
(* Station mutual interlock8 Program *)
(* Rung L273 *)
RBT_Y55_MUTUAL_INT8 := Mutual_Int8;
(* AUTO TIP CHANGE START *)
(* Rung L275 *)
RBT_Y56_TIP_CHANGE_START := M_TIP_CHANGE_START;
(* AUTO TIP CHANGE START *)
(* Rung L277 *)
RBT_Y57_TIP_CHANGE_END := M_TIP_CHANGE_COMPL;
(* PLT COUNT RST *)
(* Rung L279 *)
RBT_Y58_PLT_COUNT_RST := M_PLT_COUNT_RST_AUX;
(* GATE CLOSED SAFETY SIGNAL *)
(* Rung L281 *)
GATE_CLOSED_DELAY(IN := M_GATE_CLOSED, PT := T#500MS);
RBT_Y59_GATE_CLOSED := GATE_CLOSED_DELAY.Q;
(* GATE EMERGENCY STOP SAFETY SIGNAL *)
(* Rung L285 *)
EM_STOP_DELAY(IN := M_EM_STOP, PT := T#500MS);
RBT_Y60_EM_STOP := EM_STOP_DELAY.Q;

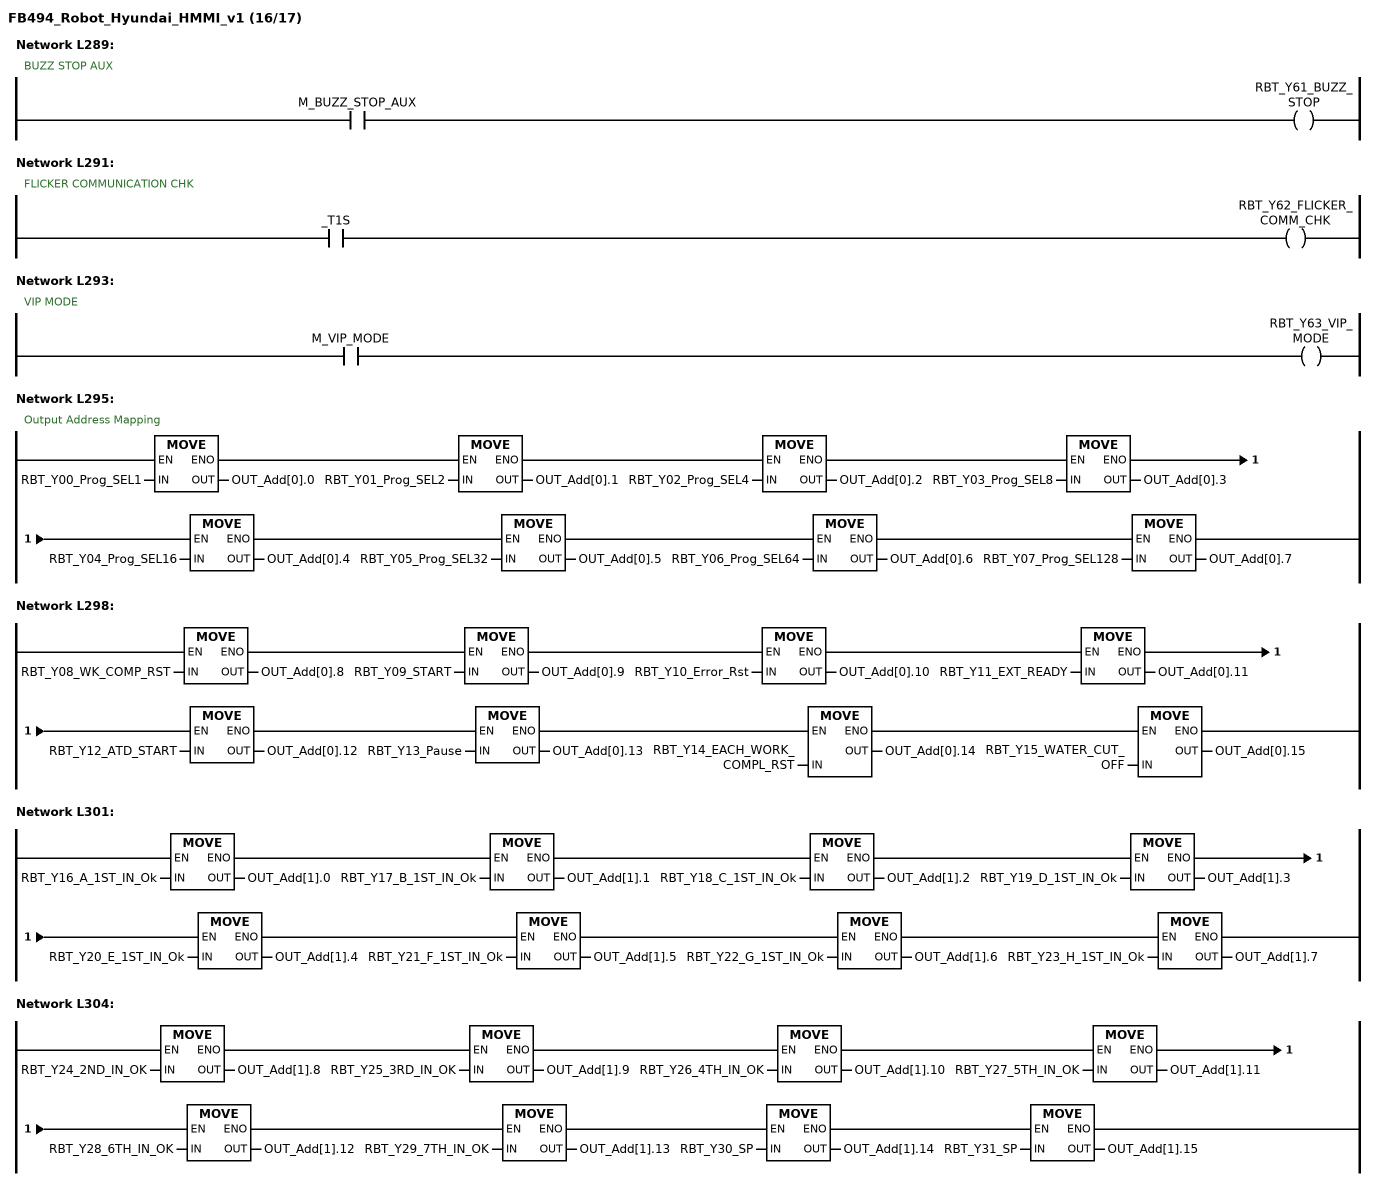
(* BUZZ STOP AUX *)
(* Rung L289 *)
RBT_Y61_BUZZ_STOP := M_BUZZ_STOP_AUX;
(* FLICKER COMMUNICATION CHK *)
(* Rung L291 *)
RBT_Y62_FLICKER_COMM_CHK := _T1S;
(* VIP MODE *)
(* Rung L293 *)
RBT_Y63_VIP_MODE := M_VIP_MODE;
(* Output Address Mapping *)
(* Rung L295 *)
OUT_Add[0].0 := RBT_Y00_Prog_SEL1;
OUT_Add[0].1 := RBT_Y01_Prog_SEL2;
OUT_Add[0].2 := RBT_Y02_Prog_SEL4;
OUT_Add[0].3 := RBT_Y03_Prog_SEL8;
OUT_Add[0].4 := RBT_Y04_Prog_SEL16;
OUT_Add[0].5 := RBT_Y05_Prog_SEL32;
OUT_Add[0].6 := RBT_Y06_Prog_SEL64;
OUT_Add[0].7 := RBT_Y07_Prog_SEL128;
(* Rung L298 *)
OUT_Add[0].8 := RBT_Y08_WK_COMP_RST;
OUT_Add[0].9 := RBT_Y09_START;
OUT_Add[0].10 := RBT_Y10_Error_Rst;
OUT_Add[0].11 := RBT_Y11_EXT_READY;
OUT_Add[0].12 := RBT_Y12_ATD_START;
OUT_Add[0].13 := RBT_Y13_Pause;
OUT_Add[0].14 := RBT_Y14_EACH_WORK_COMPL_RST;
OUT_Add[0].15 := RBT_Y15_WATER_CUT_OFF;
(* Rung L301 *)
OUT_Add[1].0 := RBT_Y16_A_1ST_IN_Ok;
OUT_Add[1].1 := RBT_Y17_B_1ST_IN_Ok;
OUT_Add[1].2 := RBT_Y18_C_1ST_IN_Ok;
OUT_Add[1].3 := RBT_Y19_D_1ST_IN_Ok;
OUT_Add[1].4 := RBT_Y20_E_1ST_IN_Ok;
OUT_Add[1].5 := RBT_Y21_F_1ST_IN_Ok;
OUT_Add[1].6 := RBT_Y22_G_1ST_IN_Ok;
OUT_Add[1].7 := RBT_Y23_H_1ST_IN_Ok;
(* Rung L304 *)
OUT_Add[1].8 := RBT_Y24_2ND_IN_OK;
OUT_Add[1].9 := RBT_Y25_3RD_IN_OK;
OUT_Add[1].10 := RBT_Y26_4TH_IN_OK;
OUT_Add[1].11 := RBT_Y27_5TH_IN_OK;
OUT_Add[1].12 := RBT_Y28_6TH_IN_OK;
OUT_Add[1].13 := RBT_Y29_7TH_IN_OK;
OUT_Add[1].14 := RBT_Y30_SP;
OUT_Add[1].15 := RBT_Y31_SP;

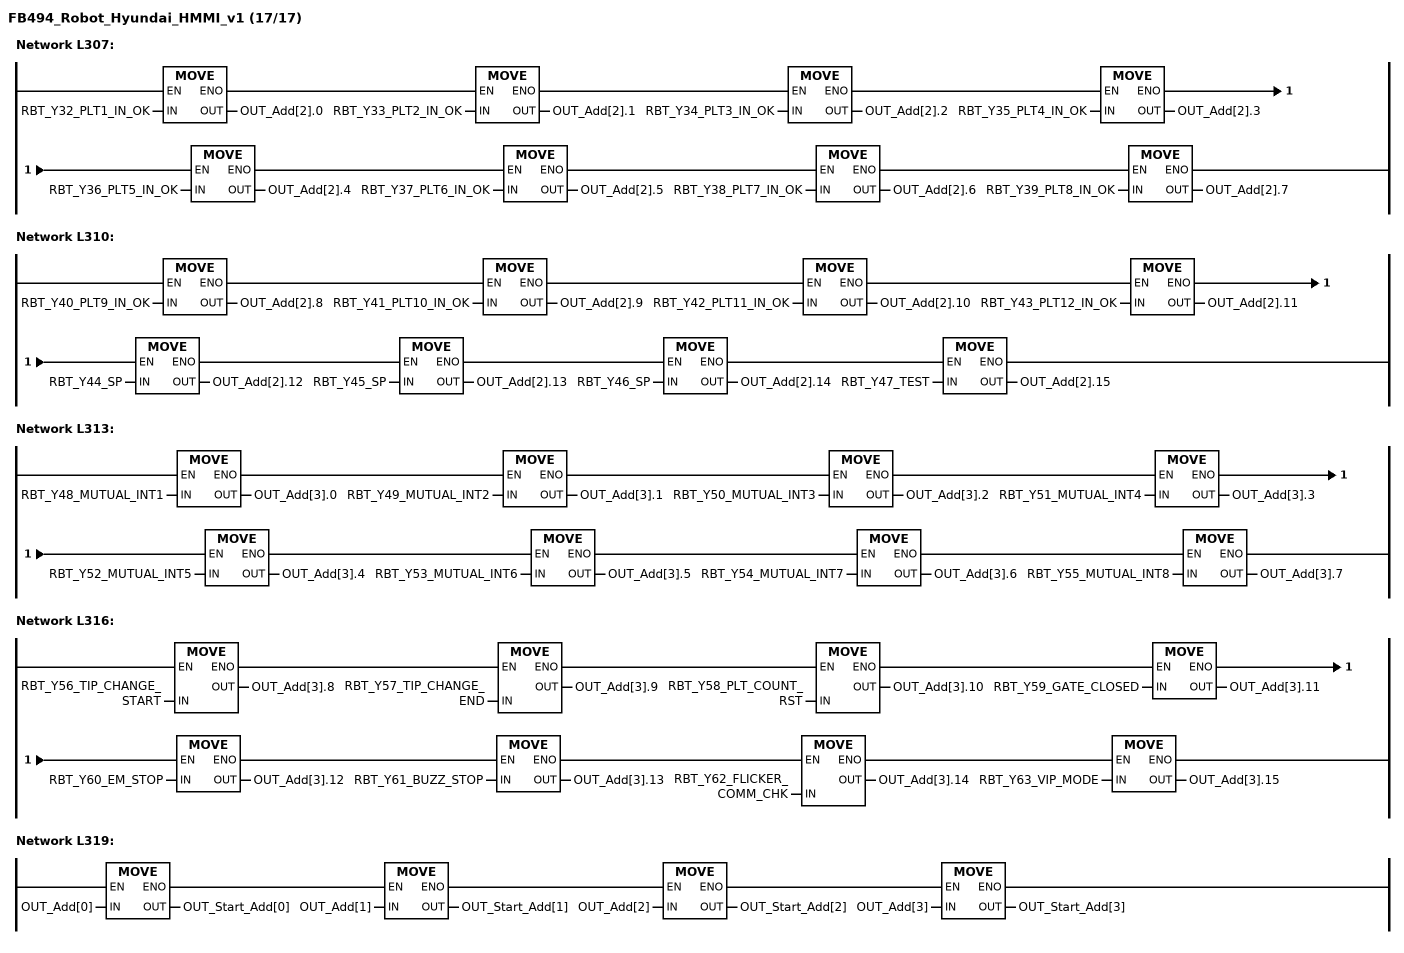
(* Rung L307 *)
OUT_Add[2].0 := RBT_Y32_PLT1_IN_OK;
OUT_Add[2].1 := RBT_Y33_PLT2_IN_OK;
OUT_Add[2].2 := RBT_Y34_PLT3_IN_OK;
OUT_Add[2].3 := RBT_Y35_PLT4_IN_OK;
OUT_Add[2].4 := RBT_Y36_PLT5_IN_OK;
OUT_Add[2].5 := RBT_Y37_PLT6_IN_OK;
OUT_Add[2].6 := RBT_Y38_PLT7_IN_OK;
OUT_Add[2].7 := RBT_Y39_PLT8_IN_OK;
(* Rung L310 *)
OUT_Add[2].8 := RBT_Y40_PLT9_IN_OK;
OUT_Add[2].9 := RBT_Y41_PLT10_IN_OK;
OUT_Add[2].10 := RBT_Y42_PLT11_IN_OK;
OUT_Add[2].11 := RBT_Y43_PLT12_IN_OK;
OUT_Add[2].12 := RBT_Y44_SP;
OUT_Add[2].13 := RBT_Y45_SP;
OUT_Add[2].14 := RBT_Y46_SP;
OUT_Add[2].15 := RBT_Y47_TEST;
(* Rung L313 *)
OUT_Add[3].0 := RBT_Y48_MUTUAL_INT1;
OUT_Add[3].1 := RBT_Y49_MUTUAL_INT2;
OUT_Add[3].2 := RBT_Y50_MUTUAL_INT3;
OUT_Add[3].3 := RBT_Y51_MUTUAL_INT4;
OUT_Add[3].4 := RBT_Y52_MUTUAL_INT5;
OUT_Add[3].5 := RBT_Y53_MUTUAL_INT6;
OUT_Add[3].6 := RBT_Y54_MUTUAL_INT7;
OUT_Add[3].7 := RBT_Y55_MUTUAL_INT8;
(* Rung L316 *)
OUT_Add[3].8 := RBT_Y56_TIP_CHANGE_START;
OUT_Add[3].9 := RBT_Y57_TIP_CHANGE_END;
OUT_Add[3].10 := RBT_Y58_PLT_COUNT_RST;
OUT_Add[3].11 := RBT_Y59_GATE_CLOSED;
OUT_Add[3].12 := RBT_Y60_EM_STOP;
OUT_Add[3].13 := RBT_Y61_BUZZ_STOP;
OUT_Add[3].14 := RBT_Y62_FLICKER_COMM_CHK;
OUT_Add[3].15 := RBT_Y63_VIP_MODE;
(* Rung L319 *)
OUT_Start_Add[0] := OUT_Add[0];
OUT_Start_Add[1] := OUT_Add[1];
OUT_Start_Add[2] := OUT_Add[2];
OUT_Start_Add[3] := OUT_Add[3];
END_FUNCTION_BLOCK

FUNCTION_BLOCK ACT_6_CYL
VAR_INPUT
    사용유무 : BOOL;
    운전준비 : BOOL;
    전진보조 : BOOL;
    후진보조 : BOOL;
    전진단수량 : UINT;
    후진단수량 : UINT;
    전진단1 : BOOL;
    후진단1 : BOOL;
    전진단2 : BOOL;
    후진단2 : BOOL;
    전진단3 : BOOL;
    후진단3 : BOOL;
    전진단4 : BOOL;
    후진단4 : BOOL;
    전진단5 : BOOL;
    후진단5 : BOOL;
    전진단6 : BOOL;
    후진단6 : BOOL;
    전진단_지연시간 : TIME;
    후진단_지연시간 : TIME;
    LS_ERR1_지연시간 : TIME;
    LS_ERR2_지연시간 : TIME;
    이상리셋 : BOOL;
END_VAR
VAR_OUTPUT
    SOL_ADV_출력 : BOOL;
    SOL_RET_출력 : BOOL;
    M_전진단 : BOOL;
    M_후진단 : BOOL;
    M_전진에러 : BOOL;
    M_후진에러 : BOOL;
    ADV_LAMP : WORD;
    RET_LAMP : WORD;
END_VAR
VAR
    ACT_USE : BOOL;
    ADV_END_TIME : TON;
    ADV_SOL_MEMO : BOOL;
    ERR_TIME1 : TON;
    LP_ADV_1 : BOOL;
    LP_ADV_2 : BOOL;
    LP_ADV_3 : BOOL;
    LP_ADV_4 : BOOL;
    LP_ADV_5 : BOOL;
    LP_ADV_6 : BOOL;
    LP_RET_1 : BOOL;
    LP_RET_2 : BOOL;
    LP_RET_3 : BOOL;
    LP_RET_4 : BOOL;
    LP_RET_5 : BOOL;
    LP_RET_6 : BOOL;
    LS_ERR_1 : BOOL;
    LS_ERR_2 : BOOL;
    RET_END_TIME : TON;
    RET_ERR_TIME : TON;
    RET_SOL_MEMO : BOOL;
    ZERO_BYTE : BYTE;
    전진단2_PASS : BOOL;
    전진단3_PASS : BOOL;
    전진단4_PASS : BOOL;
    전진단5_PASS : BOOL;
    전진단6_PASS : BOOL;
    전진단LAMP_AUX : BYTE;
    후진단2_PASS : BOOL;
    후진단3_PASS : BOOL;
    후진단4_PASS : BOOL;
    후진단5_PASS : BOOL;
    후진단6_PASS : BOOL;
    후진단LAMP_AUX : BYTE;
END_VAR

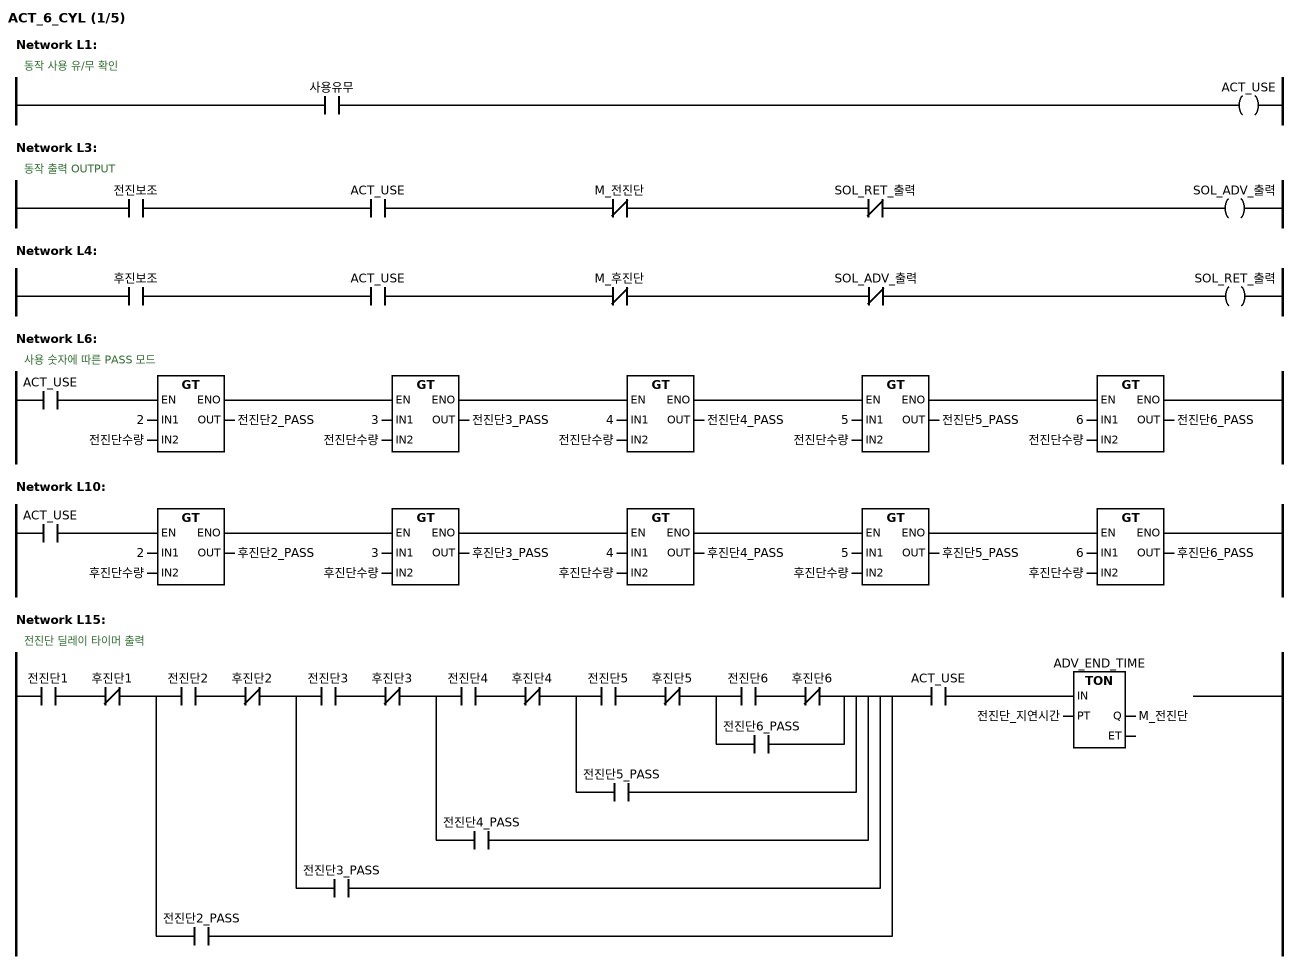
(* 동작 사용 유/무 확인 *)
(* Rung L1 *)
ACT_USE := 사용유무;
(* 동작 출력 OUTPUT *)
(* Rung L3 *)
SOL_ADV_출력 := 전진보조 AND ACT_USE AND NOT M_전진단 AND NOT SOL_RET_출력;
(* Rung L4 *)
SOL_RET_출력 := 후진보조 AND ACT_USE AND NOT M_후진단 AND NOT SOL_ADV_출력;
(* 사용 숫자에 따른 PASS 모드 *)
(* Rung L6 *)
IF ACT_USE THEN
    전진단2_PASS := 2 > 전진단수량;
    전진단3_PASS := 3 > 전진단수량;
    전진단4_PASS := 4 > 전진단수량;
    전진단5_PASS := 5 > 전진단수량;
    전진단6_PASS := 6 > 전진단수량;
END_IF;
(* Rung L10 *)
IF ACT_USE THEN
    후진단2_PASS := 2 > 후진단수량;
    후진단3_PASS := 3 > 후진단수량;
    후진단4_PASS := 4 > 후진단수량;
    후진단5_PASS := 5 > 후진단수량;
    후진단6_PASS := 6 > 후진단수량;
END_IF;
(* 전진단 딜레이 타이머 출력 *)
(* Rung L15 *)
ADV_END_TIME(IN := 전진단1 AND NOT 후진단1 AND ((전진단2 AND NOT 후진단2 AND ((전진단3 AND NOT 후진단3 AND ((전진단4 AND NOT 후진단4 AND ((전진단5 AND NOT 후진단5 AND ((전진단6 AND NOT 후진단6) OR 전진단6_PASS)) OR 전진단5_PASS)) OR 전진단4_PASS)) OR 전진단3_PASS)) OR 전진단2_PASS) AND ACT_USE, PT := 전진단_지연시간, Q => M_전진단);

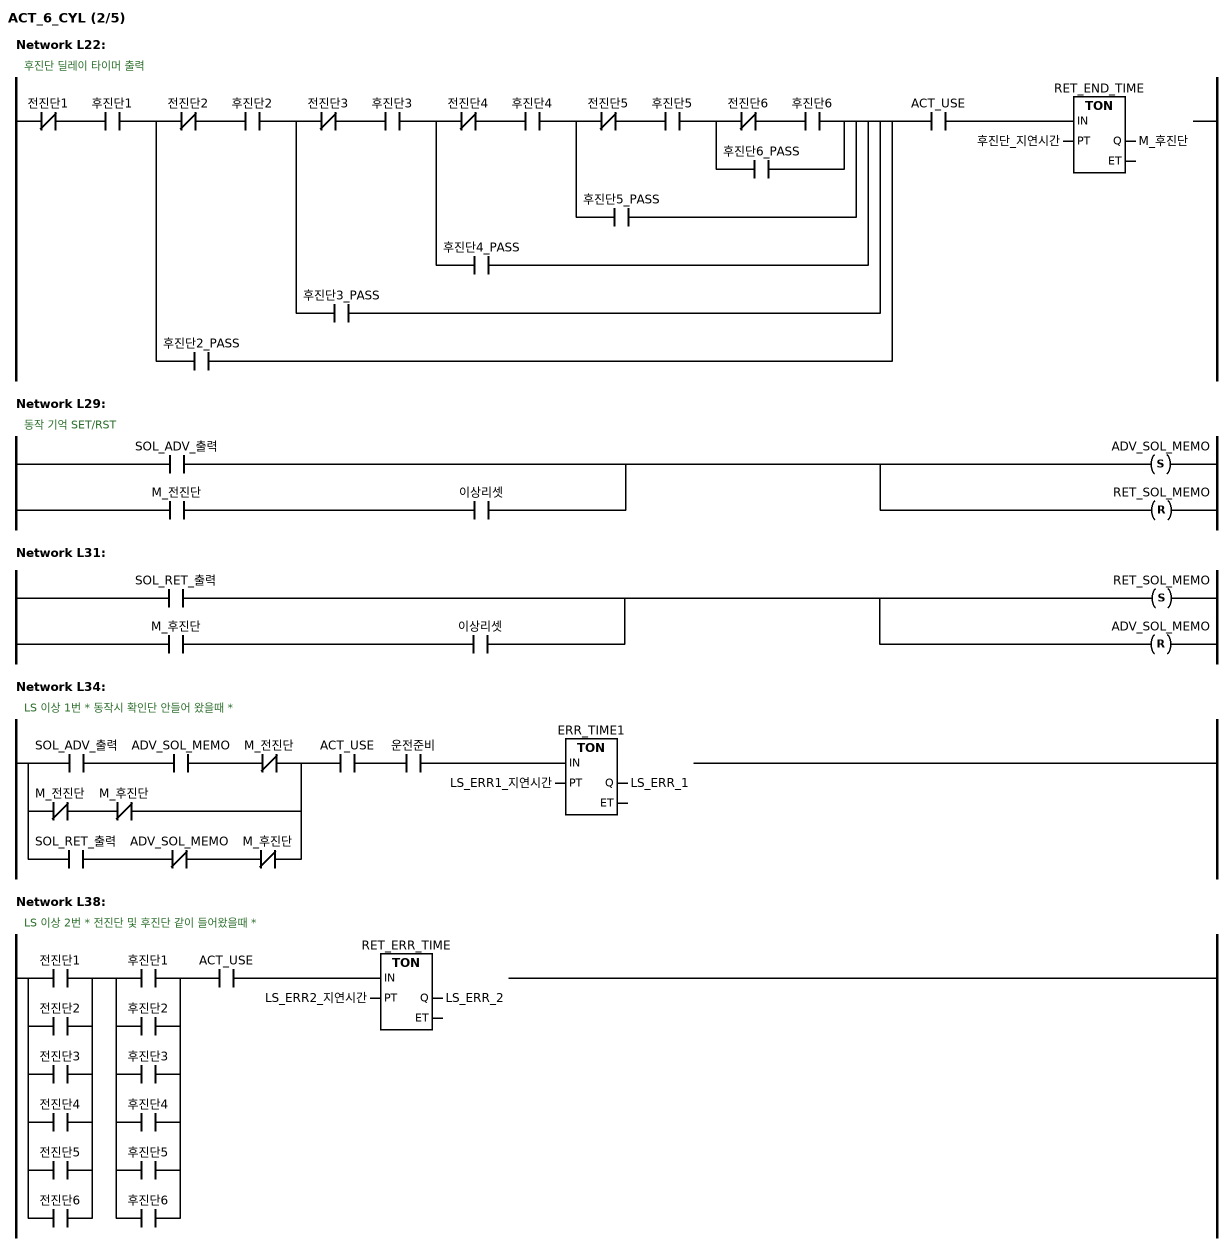
(* 후진단 딜레이 타이머 출력 *)
(* Rung L22 *)
RET_END_TIME(IN := NOT 전진단1 AND 후진단1 AND ((NOT 전진단2 AND 후진단2 AND ((NOT 전진단3 AND 후진단3 AND ((NOT 전진단4 AND 후진단4 AND ((NOT 전진단5 AND 후진단5 AND ((NOT 전진단6 AND 후진단6) OR 후진단6_PASS)) OR 후진단5_PASS)) OR 후진단4_PASS)) OR 후진단3_PASS)) OR 후진단2_PASS) AND ACT_USE, PT := 후진단_지연시간, Q => M_후진단);
(* 동작 기억 SET/RST *)
(* Rung L29 *)
IF SOL_ADV_출력 OR (M_전진단 AND 이상리셋) THEN
    ADV_SOL_MEMO := TRUE;
    RET_SOL_MEMO := FALSE;
END_IF;
(* Rung L31 *)
IF SOL_RET_출력 OR (M_후진단 AND 이상리셋) THEN
    RET_SOL_MEMO := TRUE;
    ADV_SOL_MEMO := FALSE;
END_IF;
(* LS 이상 1번 * 동작시 확인단 안들어 왔을때 * *)
(* Rung L34 *)
ERR_TIME1(IN := ((SOL_ADV_출력 AND ADV_SOL_MEMO AND NOT M_전진단) OR (NOT M_전진단 AND NOT M_후진단) OR (SOL_RET_출력 AND NOT ADV_SOL_MEMO AND NOT M_후진단)) AND ACT_USE AND 운전준비, PT := LS_ERR1_지연시간, Q => LS_ERR_1);
(* LS 이상 2번 * 전진단 및 후진단 같이 들어왔을때 * *)
(* Rung L38 *)
RET_ERR_TIME(IN := (전진단1 OR 전진단2 OR 전진단3 OR 전진단4 OR 전진단5 OR 전진단6) AND (후진단1 OR 후진단2 OR 후진단3 OR 후진단4 OR 후진단5 OR 후진단6) AND ACT_USE, PT := LS_ERR2_지연시간, Q => LS_ERR_2);

